// NETWORK 20
//   fb_gearinPos_el: add 2011 06 09 to delete 1sec delay
//   v_elevation: Virtual axis "v_elevation" with axis number 8
//   drive3: Real axis "Drive3" with axis number 3
// label: (*add ton between gearin and AF 2011_03_24*)
fb_gearinPos_el(
    Execute := test2 AND b_M_el_done,
    RatioNumerator := 1,
    RatioDenominator := 1,
    MasterFineadjust := 0,
    SyncMode := 0,
    StartMode := 0,
    Master := v_elevation,
    Slave := drive3); // MB_GearInPos
b_gearin_3_done := fb_gearinPos_el.InSync;

// NETWORK 21 (disabled)
//   v_elevation: Virtual axis "v_elevation" with axis number 8
//   drive4: Real axis "Drive4" with axis number 4
//   b_gearin_4_done: drive 3 and 4 are synchronous with v_elevation
// fb_gearin_4(
//     Execute := b_gearin_3_done,
//     RatioNumerator := 1,
//     RatioDenominator := 1,
//     MasterFineadjust := 0,
//     SyncMode := 0,
//     StartMode := 1,
//     Master := v_elevation,
//     Slave := drive4); // MB_GearInPos
// b_gearin_4_done := fb_gearin_4.InSync;

// NETWORK 22
//   b_local_on: in the local mode
//   axisdata[6].Axis_InAb: A-0-0021.14 -RD- Axis is ready for power to the engine (Ab)
//   axisdata[5].Axis_InAb: A-0-0021.14 -RD- Axis is ready for power to the engine (Ab)
//   b_enable_FI_6: the enable of drive 6
//   b_enable_FI_5: the enable of drive 5
// label: (*enable FeedIndexer axis with panel*)
fb_rtrig_FI(CLK := (b_local_on AND b_enable_FI OR b_remote_on AND b_activate_FI) AND axisdata[6].Axis_InAb AND axisdata[5].Axis_InAb); // R_TRIG
b_enable_FI_6 S= fb_rtrig_FI.Q;
b_enable_FI_5 S= fb_rtrig_FI.Q;

// NETWORK 23 (disabled)
//   b_enable_FI_5: the enable of drive 5
//   axisdata[5].Axis_InAb: A-0-0021.14 -RD- Axis is ready for power to the engine (Ab)
//   axisdata[5].Axis_Error: A-0-0021.09 -RD- Axis reports error
//   drive5: Real axis "Drive5" with axis number 5
// ton_en_5(IN := b_enable_FI_5 AND axisdata[5].Axis_InAb AND NOT axisdata[5].Axis_Error, PT := t#500ms); // TON
// fb_5_power(Enable := ton_en_5.Q, Axis := drive5); // MC_Power
// b_5_enable_on := fb_5_power.Status;

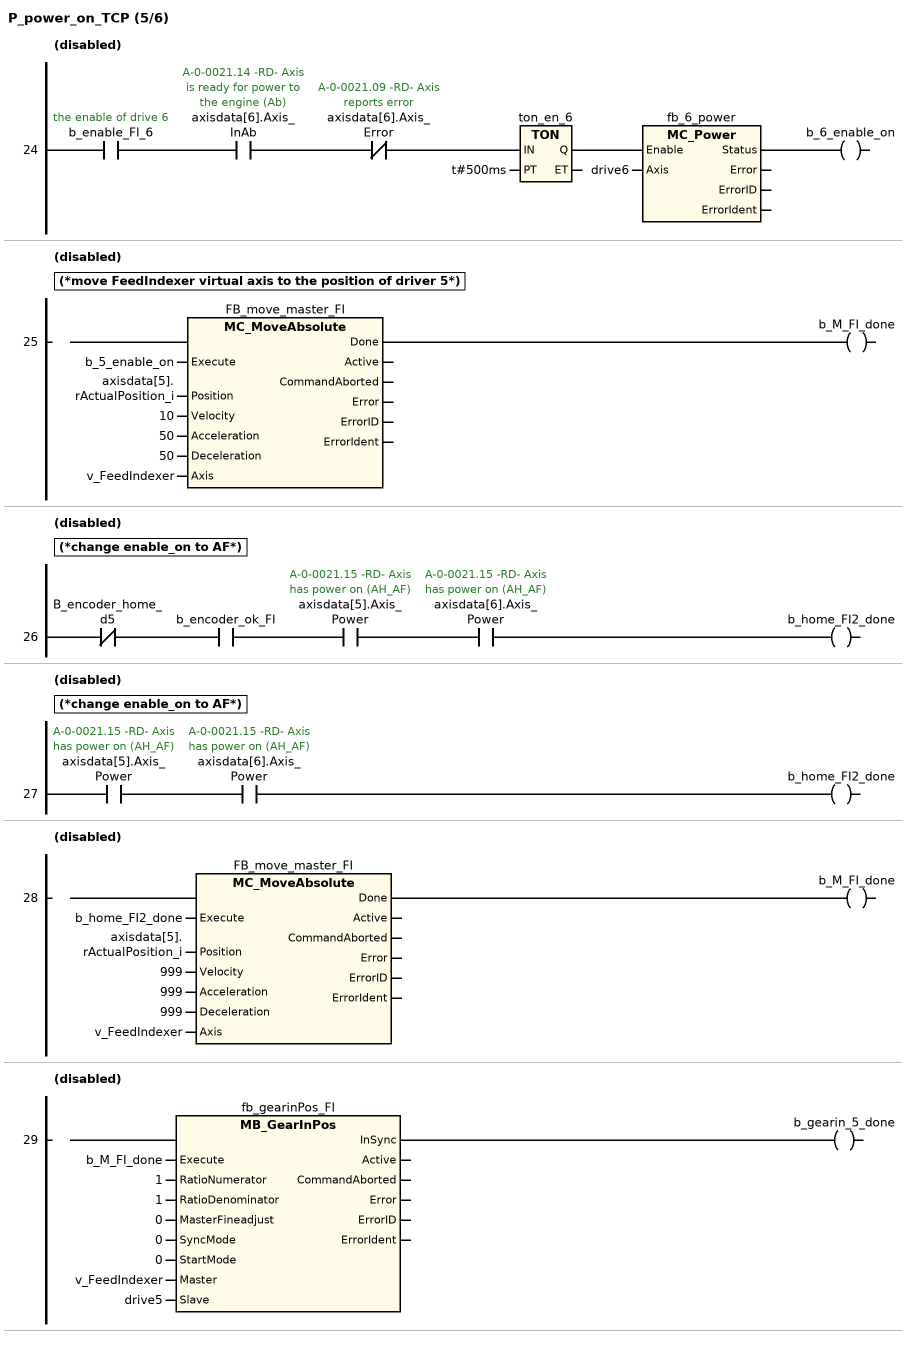
// NETWORK 24 (disabled)
//   b_enable_FI_6: the enable of drive 6
//   axisdata[6].Axis_InAb: A-0-0021.14 -RD- Axis is ready for power to the engine (Ab)
//   axisdata[6].Axis_Error: A-0-0021.09 -RD- Axis reports error
//   drive6: Real axis "Drive6" with axis number 6
// ton_en_6(IN := b_enable_FI_6 AND axisdata[6].Axis_InAb AND NOT axisdata[6].Axis_Error, PT := t#500ms); // TON
// fb_6_power(Enable := ton_en_6.Q, Axis := drive6); // MC_Power
// b_6_enable_on := fb_6_power.Status;

// NETWORK 25 (disabled)
//   axisdata[5].rActualPosition_i: A-0-0100 -RD- Actual position
//   v_FeedIndexer: Virtual axis "v_polarization" with axis number 9
// label: (*move FeedIndexer virtual axis to the position of driver 5*)
// FB_move_master_FI(
//     Execute := b_5_enable_on,
//     Position := axisdata[5].rActualPosition_i,
//     Velocity := 10,
//     Acceleration := 50,
//     Deceleration := 50,
//     Axis := v_FeedIndexer); // MC_MoveAbsolute
// b_M_FI_done := FB_move_master_FI.Done;

// NETWORK 26 (disabled)
//   axisdata[5].Axis_Power: A-0-0021.15 -RD- Axis has power on (AH_AF)
//   axisdata[6].Axis_Power: A-0-0021.15 -RD- Axis has power on (AH_AF)
// label: (*change enable_on to AF*)
// b_home_FI2_done := NOT B_encoder_home_d5 AND b_encoder_ok_FI AND axisdata[5].Axis_Power AND axisdata[6].Axis_Power;

// NETWORK 27 (disabled)
//   axisdata[5].Axis_Power: A-0-0021.15 -RD- Axis has power on (AH_AF)
//   axisdata[6].Axis_Power: A-0-0021.15 -RD- Axis has power on (AH_AF)
// label: (*change enable_on to AF*)
// b_home_FI2_done := axisdata[5].Axis_Power AND axisdata[6].Axis_Power;

// NETWORK 28 (disabled)
//   axisdata[5].rActualPosition_i: A-0-0100 -RD- Actual position
//   v_FeedIndexer: Virtual axis "v_polarization" with axis number 9
// FB_move_master_FI(
//     Execute := b_home_FI2_done,
//     Position := axisdata[5].rActualPosition_i,
//     Velocity := 999,
//     Acceleration := 999,
//     Deceleration := 999,
//     Axis := v_FeedIndexer); // MC_MoveAbsolute
// b_M_FI_done := FB_move_master_FI.Done;

// NETWORK 29 (disabled)
//   v_FeedIndexer: Virtual axis "v_polarization" with axis number 9
//   drive5: Real axis "Drive5" with axis number 5
// fb_gearinPos_FI(
//     Execute := b_M_FI_done,
//     RatioNumerator := 1,
//     RatioDenominator := 1,
//     MasterFineadjust := 0,
//     SyncMode := 0,
//     StartMode := 0,
//     Master := v_FeedIndexer,
//     Slave := drive5); // MB_GearInPos
// b_gearin_5_done := fb_gearinPos_FI.InSync;

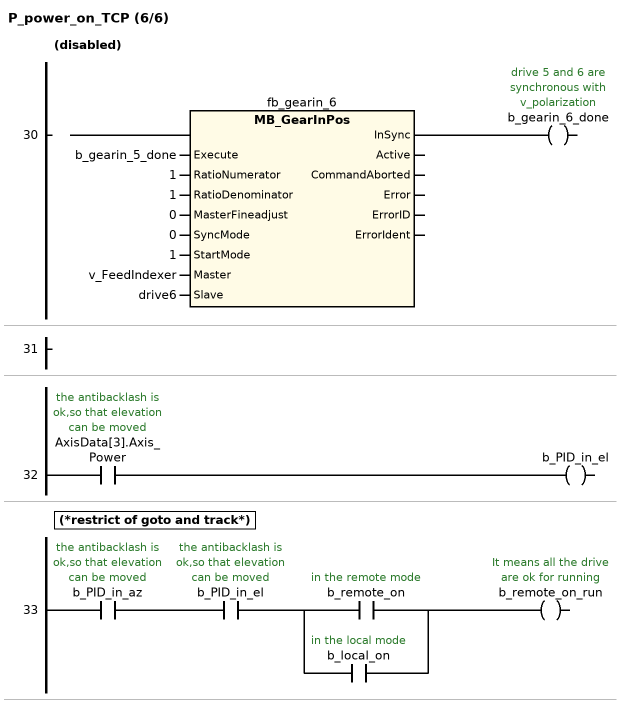
// NETWORK 30 (disabled)
//   v_FeedIndexer: Virtual axis "v_polarization" with axis number 9
//   drive6: Real axis "Drive6" with axis number 6
//   b_gearin_6_done: drive 5 and 6 are synchronous with v_polarization
// fb_gearin_6(
//     Execute := b_gearin_5_done,
//     RatioNumerator := 1,
//     RatioDenominator := 1,
//     MasterFineadjust := 0,
//     SyncMode := 0,
//     StartMode := 1,
//     Master := v_FeedIndexer,
//     Slave := drive6); // MB_GearInPos
// b_gearin_6_done := fb_gearin_6.InSync;

// NETWORK 31

// NETWORK 32
//   AxisData[3].Axis_Power: the antibacklash is ok,so that elevation can be moved
b_PID_in_el := AxisData[3].Axis_Power;

// NETWORK 33
//   b_PID_in_az: the antibacklash is ok,so that elevation can be moved
//   b_PID_in_el: the antibacklash is ok,so that elevation can be moved
//   b_remote_on: in the remote mode
//   b_local_on: in the local mode
//   b_remote_on_run: It means all the drive are ok for running
// label: (*restrict of goto and track*)
b_remote_on_run := b_PID_in_az AND b_PID_in_el AND (b_remote_on OR b_local_on);

END_PROGRAM

// IndraMotionMlc1/Application/POUs/Simulation/P_Simulation
PROGRAM P_Simulation
VAR
	//b_zone_az_sim:BOOL;  // simulate the zone switch 
	
	sim_HMV_warning : BOOL;(*the warning of HMV*)     
	sim_HMV_UD : BOOL;(*the UD of HMV*)              
	sim_stow_pin_limit_lock: BOOL:=1;(*locked*) // Stow pin deployed limit active
	sim_stow_pin_limit_unlock : BOOL;(*unlocked*) // Stow pin retracted limit active
	fb_rtrig_sim_stow_pin_retract: R_TRIG;
	fb_rtrig_sim_stow_pin_deploy: R_TRIG;
	sim_DriveCabinetDoor_Estop :BOOL;(*the estop of DriveCabinetDoor*)
	
	sim_PedDoor_Switch  :BOOL;(*the estop of DSDoor*)
	sim_PSCDoor_Switch :BOOL;(*the estop of DPSCDoor*)
	sim_EMISCDoor_Switch  :BOOL; (*the estop of EMISCDoor*)
	
	sim_AZ_Hatch  :BOOL;(*the estop of AZ_Hatch*)
	sim_Turnhead_Hatch  :BOOL;(*the estop of Turnhead_Hatch*)
	sim_DS_Estop  :BOOL;(*the estop of DS*)
	sim_Turnhead_Estop  :BOOL;(*the estop of Turnhead*)
	sim_FI_Estop  :BOOL;(*the estop of FI*)

	sim_HHP_Connected : BOOL;      
	sim_HHP_AZ : BOOL;
	sim_HHP_EL : BOOL;
	sim_HHP_Interlock : BOOL;
	sim_HHP_move_cw_slow : BOOL;
	sim_HHP_move_ccw_slow : BOOL;
	sim_HHP_move_cw_fast : BOOL;
	sim_HHP_move_ccw_fast : BOOL;
	
	sim_HHP_ENABLE  :BOOL;
	sim_HHP_STOW  :BOOL;
	sim_HHP_Motor_UNLOCK  :BOOL;
	sim_HHP_Disable  :BOOL;
	sim_HHP_Estop :BOOL;(*the estop of HHP*)
	sim_MAIN_PD_Compressor_breaker_on  :BOOL;
	sim_MAIN_PD_MAIN_lighting_on  :BOOL;
	
	sim_MAIN_PD_FI_Breaker_on :BOOL;
	sim_MAIN_PD_spare :BOOL;
	sim_PSC_PD_Light_Breaker_on :BOOL;
	sim_PSC_PD_EMISC_Breaker_on :BOOL;
	sim_PSC_PD_FAN_Breaker_on  :BOOL;
	sim_PSC_PD_spare :BOOL;
	
	sim_FI_PD_FI1_Breaker_on :BOOL;
	sim_FI_PD_FI2_Breaker_on  :BOOL;
	
	sim_Lock_Out_Az: BOOL;
	sim_Lock_Out_El: BOOL;
	sim_Lock_Out_Fi: BOOL;
	b_aztest: REAL;
	b_sector_sw: BOOL;
	
	
	
	b_escape: Bool;
	Az_lim_off: BOOL:=FALSE;
	El_lim_off: BOOL:=FALSE;
	Fi_lim_off: BOOL:=FALSE;
END_VAR

(* This piece of code is used to simulate the digital IO and drive IO when virtual axes are used *)
(*	r_limit_cw_az_sim:REAL:= 270 ;
	r_limit_ccw_az_sim:REAL:= -270;
	r_limit_final_cw_az_sim:REAL:= 271 ;
	r_limit_final_ccw_az_sim:REAL:=-271 ;
	// Elevation Limits
	r_limit_cw_az_sim:REAL:= 90;
	r_limit_ccw_az_sim:REAL:= 13.5 ;
	r_limit_final_cw_az_sim:REAL:=90.5 ;
	r_limit_final_ccw_az_sim:REAL:=13 ;
	// Feed Indexer Limits
	r_limit_cw_az_sim:REAL:= 110;
	r_limit_ccw_az_sim:REAL:= -140;
	r_limit_final_cw_az_sim:REAL:= 111 ;
	r_limit_final_ccw_az_sim:REAL:= -141; *)
	
IF gc_b_sim_on=1 THEN 
// Initial position 
    	

// Zone switch 
     b_aztest:=axisdata[1].rActualPosition_i;
	// There is a flash of llimits as AZ crosses over 0. I don't think this will be fixed in the simulator. 
	IF (axisdata[1].rActualPosition_i > 0.0 AND axisdata[1].rActualPosition_i < 90) THEN 
		b_zone_az_sim:=1;
	ELSIF axisdata[1].rActualPosition_i > 270 THEN
        b_zone_az_sim:=0;
	ELSE 
		b_zone_az_sim:=1;
	END_IF

// Azimuth limits
 IF NOT Az_lim_off THEN 
	IF r_pos_az_v >= gc_r_limit_cw_az_sim THEN 
		b_limit_cw_az:=1;
		b_stop_Az:=1;
	ELSE
		b_limit_cw_az:=0;
	END_IF
	
	IF r_pos_az_v <= gc_r_limit_ccw_az_sim THEN 
		b_limit_ccw_az:=1;
		b_stop_Az:=1;
		ELSE
		b_limit_ccw_az:=0;
	END_IF
	IF r_pos_az_v >= gc_r_limit_final_cw_az_sim THEN 
		b_limit_final_cw_az:=1;
		b_stop_Az:=1;
		ELSE
		b_limit_final_cw_az:=0;
	END_IF
	IF r_pos_az_v <= gc_r_limit_final_ccw_az_sim THEN 
		b_limit_final_ccw_az:=1;
		b_stop_Az:=1;
		ELSE
		b_limit_final_ccw_az:=0;
	END_IF
 ELSE
   b_limit_final_ccw_az:=0;
   b_limit_final_cw_az:=0;
	b_limit_ccw_az:=0;
	b_limit_cw_az:=0;
 END_IF;
	
	
	// Elevation limits
 IF NOT El_lim_off THEN
	IF r_pos_el_v >= gc_r_limit_cw_el_sim THEN 
		b_limit_cw_el:=1;
		
		IF b_enable_el_3=TRUE AND NOT(b_escape) THEN
			b_stop_El:=1;
			b_deactivate_el:=1;
			b_escape:=1;
		END_IF
	ELSE
		b_limit_cw_el:=0;
		b_escape:=0;
	END_IF
	IF r_pos_el_v <= gc_r_limit_ccw_el_sim THEN 
		b_limit_ccw_el:=1;
		
		//IF b_enable_el_3 THEN
		//	b_stop_El:=1;
		//	b_deactivate_el:=1;
		//END_IF
	ELSE
		b_limit_ccw_el:=0;
	END_IF
	IF r_pos_el_v >= gc_r_limit_final_cw_el_sim THEN 
		b_limit_final_cw_el:=1;
		//b_stop_El:=1;
		ELSE
		b_limit_final_cw_el:=0;
	END_IF
	IF r_pos_el_v <= gc_r_limit_final_ccw_el_sim THEN 
		b_limit_final_ccw_el:=1;
		//b_stop_El:=1;
		ELSE
		b_limit_final_ccw_el:=0;
	END_IF
 ELSE
	b_limit_final_ccw_el:=0;
	b_limit_final_cw_el:=0;
	b_limit_cw_el:=0;
	b_limit_ccw_el:=0;
 END_IF
 
	// Feed Indexer Limits
 IF NOT Fi_lim_off THEN
	IF r_pos_fi_v >= gc_r_limit_cw_fi_sim THEN 
		b_limit_cw_fi:=1;
		b_stop_Fi:=1;
	ELSE
		b_limit_cw_fi:=0;
	END_IF
	IF r_pos_fi_v <= gc_r_limit_ccw_fi_sim THEN 
		b_limit_ccw_fi:=1;
		b_stop_Fi:=1;
		ELSE
		b_limit_ccw_fi:=0;
	END_IF
	IF r_pos_fi_v >= gc_r_limit_final_cw_fi_sim THEN 
		b_limit_final_cw_fi:=1;
		b_stop_Fi:=1;
		ELSE
		b_limit_final_cw_fi:=0;
	END_IF
	IF r_pos_el_v <= gc_r_limit_final_ccw_fi_sim THEN 
		b_limit_final_ccw_fi:=1;
		b_stop_Fi:=1;
		ELSE
		b_limit_final_ccw_fi:=0;
	END_IF
ELSE 
	b_limit_final_ccw_fi:=0;
	b_limit_final_cw_fi:=0;
	b_limit_ccw_fi:=0;
	b_limit_cw_fi:=0;
END_IF
// Expose inputs to OPCUA

	b_HMV_warning:= sim_HMV_warning; 
	b_HMV_UD:=sim_HMV_UD ;         
	//b_stow_pin_limit_lock:= sim_stow_pin_limit_lock  ;
	fb_rtrig_sim_stow_pin_deploy(CLK:=sim_stow_pin_limit_lock);
	//b_stow_pin_limit_lock:=fb_rtrig_sim_stow_pin_deploy.Q;
	// simulate a retracted stow pin limit
	//fb_rtrig_sim_stow_pin_retract(CLK:=sim_stow_pin_limit_unlock);
	//b_stow_pin_limit_unlock:=fb_rtrig_sim_stow_pin_retract.Q;
	
	
	b_DriveCabinetDoor_Estop:= sim_DriveCabinetDoor_Estop ; 
	b_DSDoor_Estop:= sim_PedDoor_Switch ; 
	b_PSCDoor_Estop:= sim_PSCDoor_Switch ; 
	b_AZ_Hatch:= sim_AZ_Hatch ;  
	b_Turnhead_Hatch:= sim_Turnhead_Hatch ; 
	b_DS_Estop:= sim_DS_Estop;  
	b_Turnhead_Estop:= sim_Turnhead_Estop;  
	b_FI_Estop:=  sim_FI_Estop;

	b_HHP_Connected:=  sim_HHP_Connected; 
	b_HHP_AZ:= sim_HHP_AZ;
	b_HHP_EL:= sim_HHP_EL;
	b_HHP_Interlock:= sim_HHP_Interlock; 
	b_HHP_move_cw_slow:=  sim_HHP_move_cw_slow; 
	b_HHP_move_ccw_slow:= sim_HHP_move_ccw_slow ;
	b_HHP_move_cw_fast:= sim_HHP_move_cw_fast;
	b_HHP_move_ccw_fast:= sim_HHP_move_ccw_fast;
	
	b_HHP_ENABLE:= sim_HHP_ENABLE ;
	b_HHP_STOW:= sim_HHP_STOW ;
	b_HHP_Motor_UNLOCK:=  sim_HHP_Motor_UNLOCK; 
	b_HHP_Disable:=  sim_HHP_Disable;
	b_EMISCDoor_Estop:= sim_EMISCDoor_Switch;  
	b_HHP_Estop:= sim_HHP_Estop;
	b_MAIN_PD_Compressor_breaker_on:= sim_MAIN_PD_Compressor_breaker_on;
	b_MAIN_PD_MAIN_lighting_on:= sim_MAIN_PD_MAIN_lighting_on;  
	
	b_MAIN_PD_FI_Breaker_on:= sim_MAIN_PD_FI_Breaker_on;
	b_MAIN_PD_spare:=  sim_MAIN_PD_spare;
	b_PSC_PD_Light_Breaker_on:= sim_PSC_PD_Light_Breaker_on;
	b_PSC_PD_EMISC_Breaker_on:=  sim_PSC_PD_EMISC_Breaker_on;
	b_PSC_PD_FAN_Breaker_on:= sim_PSC_PD_FAN_Breaker_on ;
    b_PSC_PD_spare:= sim_PSC_PD_spare;
	b_FI_PD_FI1_Breaker_on:= sim_FI_PD_FI1_Breaker_on;
	b_FI_PD_FI2_Breaker_on := sim_FI_PD_FI2_Breaker_on ;
	
	b_Lock_Out_Az:= sim_Lock_Out_Az;
	b_Lock_Out_El:= sim_Lock_Out_El;
	b_Lock_Out_Fi:= sim_Lock_Out_Fi;
	

	
 END_IF //IF b_sim_on=1 THEN

END_PROGRAM

// IndraMotionMlc1/Application/POUs/Panel Function/P_remote_local
(*This program is built for switch the mode between local,remote and off.
In the local mode,the antenna can be controled only by the button on the
panelbox;In the remote mode,the antenna can be controled only by the command
that come from the ACU;In the off mode,all the motion will be stopped.
And every time the switch is off,there is a clear_error action*)
PROGRAM P_remote_local
VAR
(*clear all error when the switch is off*)
	FB_clear_all_error: MB_WriteParameter;
	b_clear_error: BOOL;
	b_clear_all_error: BOOL;
	b_clear_done: BOOL;
	rtrig_clear_error: R_TRIG;
	rtrig_reset_clear: R_TRIG;
	el_encoder_pos: LREAL;
	b_run_once: BOOL;
END_VAR

b_Alarm;
b_Horn;
b_HHP_Interlock;
b_HHP_ENABLE;
b_HHP_STOW;
b_HHP_Motor_UNLOCK;
b_HHP_Disable;
el_encoder_pos:=Motor_to_encoder(axisdata[3].rActualPosition_i);

IF b_HHP_AZ=FALSE AND b_HHP_FI=FALSE THEN
	b_HHP_EL := TRUE;
ELSE
	b_HHP_EL := FALSE;
END_IF

IF b_HHP_connected THEN
	b_remote_on:=FALSE;
	b_local_on:=TRUE;
	CommandArbiter.Status.DscCmdAuthority:= HHP; // Needsome code to change it to No Auth when HHP is dosconnected. 
	IF NOT b_run_once THEN 
     b_Horn_Start:= TRUE; 
	 b_run_once:=TRUE;
	END_IF
ELSE
	b_remote_on:=TRUE;
	b_local_on:=FALSE;
	b_run_once:=FALSE;
END_IF

IF b_local_on OR b_remote_on THEN
	b_clear_error:=FALSE;
END_IF;
(*when the switch is off,reset some command and stop all the motion*)
IF b_remote_on =FALSE AND b_local_on=FALSE THEN
	b_power_Az:=FALSE;
	b_power_el:=FALSE;
	b_power_FI:=FALSE;
	b_stow_pin_deploy:=FALSE;
	b_stow_pin_retract:=FALSE;
	b_scc_enable_on:=FALSE;
	b_scc_enable_off:=FALSE;
	b_scc_stow:=FALSE;
	b_track_on:=FALSE;
	b_clear_error:=TRUE;
	b_scc_goto:=FALSE;
	b_scc_goto_az:=FALSE;
	b_scc_goto_el:=FALSE;
	b_scc_goto_FI:=FALSE;
	b_scc_vel:=FALSE;
END_IF;
(*transfer the sub-program A_clear_error to clear all the error*)
P_remote_local.A_clear_error();

ACTION A_clear_error:
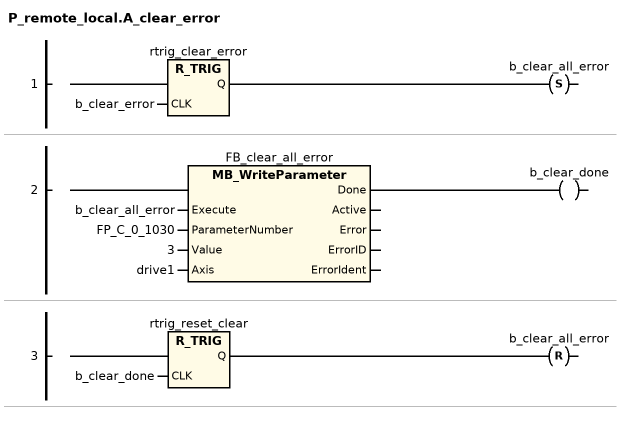
// NETWORK 1
rtrig_clear_error(CLK := b_clear_error); // R_TRIG
b_clear_all_error S= rtrig_clear_error.Q;

// NETWORK 2
FB_clear_all_error(Execute := b_clear_all_error, ParameterNumber := FP_C_0_1030, Value := 3, Axis := drive1); // MB_WriteParameter
b_clear_done := FB_clear_all_error.Done;

// NETWORK 3
rtrig_reset_clear(CLK := b_clear_done); // R_TRIG
b_clear_all_error R= rtrig_reset_clear.Q;
END_ACTION

END_PROGRAM

// IndraMotionMlc1/Application/POUs/TCP/Message/Motor_to_encoder
FUNCTION Motor_to_encoder : LREAL
VAR_INPUT
	motor_input:LREAL;
END_VAR
VAR
END_VAR

IF motor_input < 619748 THEN
	Motor_to_encoder:=AA1*(motor_input)-BB1;	
ELSIF (619748 <= motor_input) AND (motor_input < 676291) THEN
	Motor_to_encoder:=AA2*(motor_input)-BB2;
ELSIF (676291 <= motor_input) AND (motor_input < 735364) THEN
	Motor_to_encoder:=AA3*(motor_input)-BB3;
ELSIF (735364 <= motor_input) AND (motor_input < 796846) THEN
	Motor_to_encoder:=AA4*(motor_input)-BB4;
ELSIF (796846 <= motor_input) AND (motor_input < 860616) THEN
	Motor_to_encoder:=AA5*(motor_input)-BB5;
ELSIF (860616 <= motor_input) AND (motor_input < 926557) THEN
	Motor_to_encoder:=AA6*(motor_input)-BB6;
ELSIF (926557 <= motor_input) AND (motor_input < 994541) THEN
	Motor_to_encoder:=AA7*(motor_input)-BB7;
ELSIF (994541 <= motor_input) AND (motor_input < 1064438) THEN
	Motor_to_encoder:=AA8*(motor_input)-BB8;
ELSIF (1064438 <= motor_input) AND (motor_input < 1136109) THEN
	Motor_to_encoder:=AA9*(motor_input)-BB9;
ELSIF (1136109 <= motor_input) AND (motor_input < 1209420) THEN
	Motor_to_encoder:=AA10*(motor_input)-BB10;
ELSIF (1209420 <= motor_input) AND (motor_input < 1284232) THEN
	Motor_to_encoder:=AA11*(motor_input)-BB11;
ELSIF (1284232 <= motor_input) AND (motor_input < 1360400) THEN
	Motor_to_encoder:=AA12*(motor_input)-BB12;
ELSIF (1360400 <= motor_input) AND (motor_input < 1437759) THEN
	Motor_to_encoder:=AA13*(motor_input)-BB13;
ELSIF (1437759 <= motor_input) AND (motor_input < 1516147) THEN
	Motor_to_encoder:=AA14*(motor_input)-BB14;
ELSE
	Motor_to_encoder:=AA15*(motor_input)-BB15;
END_IF

END_FUNCTION

// IndraMotionMlc1/Application/POUs/Panel Function/P_read_drv_IO
(* The program is built for read the digital input value on X31 and X32,
and FP_P_0_0303 is Digital I/Os status display *)
PROGRAM P_read_drv_IO
VAR
(*With "MB_ReadParameter",it is possible to read the current value of a parameter. The return value is DINT. *)
	FB_1_read_P303: MB_ReadParameter;
	FB_2_read_P303: MB_ReadParameter;
	FB_3_read_P303: MB_ReadParameter;
	FB_4_read_P303: MB_ReadParameter;
	FB_5_read_P303: MB_ReadParameter;
	FB_6_read_P303: MB_ReadParameter;
	Dint_1_P303: DINT;
	Dint_2_P303: DINT;
	Dint_3_P303: DINT;
	Dint_4_P303: DINT;
	Dint_5_P303: DINT;
	Dint_6_P303: DINT;
(*change DINT to DWORD,so that the bit of DWORD can be read*)
	Dword_1_P303: DWORD;
	Dword_2_P303: DWORD;
	Dword_3_P303: DWORD;
	Dword_4_P303: DWORD;
	Dword_5_P303: DWORD;
	Dword_6_P303: DWORD;
	R_TRIG_0: R_TRIG;
	rtrig_stop_az1: R_TRIG;
	b_stop1_done: BOOL;
	b_stop_act_az: BOOL;
	R_TRIG_1: r_trig;
	b_zero_velocity: BOOL;
	fb_zero_velocity: MC_movevelocity;
	b_zero1_done: BOOL;
	b_zero_act_az: BOOL;
	TON_0: ton;
	FB_move_master_az1: MC_MoveAbsolute;
	fb_stop_AZ: MC_STOP;
END_VAR
VAR // added by the converter: edge detectors and wires of the graphical bodies
    _w1, _w2, _w3, _w4, _w5, _w6 : ANY;
    _w7 : BOOL;
END_VAR

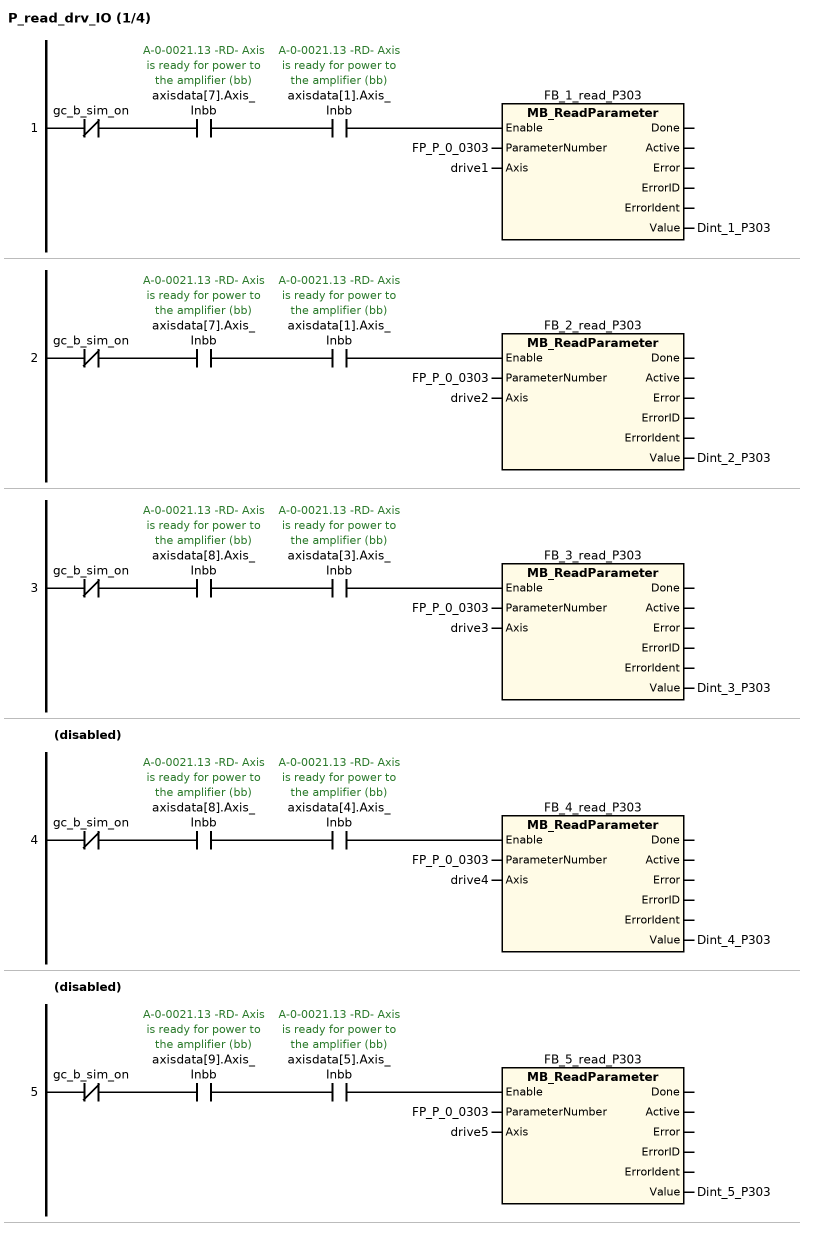
// NETWORK 1
//   FB_1_read_P303: With "MB_ReadParameter",it is possible to read the current value of a parameter. The return value is DINT.
//   axisdata[7].Axis_Inbb: A-0-0021.13 -RD- Axis is ready for power to the amplifier (bb)
//   axisdata[1].Axis_Inbb: A-0-0021.13 -RD- Axis is ready for power to the amplifier (bb)
//   FP_P_0_0303: Digital inputs, input image of device
//   drive1: Real axis "Drive1" with axis number 1
FB_1_read_P303(
    Enable := NOT gc_b_sim_on AND axisdata[7].Axis_Inbb AND axisdata[1].Axis_Inbb,
    ParameterNumber := FP_P_0_0303,
    Axis := drive1,
    Value => Dint_1_P303); // MB_ReadParameter

// NETWORK 2
//   axisdata[7].Axis_Inbb: A-0-0021.13 -RD- Axis is ready for power to the amplifier (bb)
//   axisdata[1].Axis_Inbb: A-0-0021.13 -RD- Axis is ready for power to the amplifier (bb)
//   FP_P_0_0303: Digital inputs, input image of device
//   drive2: Real axis "Drive2" with axis number 2
FB_2_read_P303(
    Enable := NOT gc_b_sim_on AND axisdata[7].Axis_Inbb AND axisdata[1].Axis_Inbb,
    ParameterNumber := FP_P_0_0303,
    Axis := drive2,
    Value => Dint_2_P303); // MB_ReadParameter

// NETWORK 3
//   axisdata[8].Axis_Inbb: A-0-0021.13 -RD- Axis is ready for power to the amplifier (bb)
//   axisdata[3].Axis_Inbb: A-0-0021.13 -RD- Axis is ready for power to the amplifier (bb)
//   FP_P_0_0303: Digital inputs, input image of device
//   drive3: Real axis "Drive3" with axis number 3
FB_3_read_P303(
    Enable := NOT gc_b_sim_on AND axisdata[8].Axis_Inbb AND axisdata[3].Axis_Inbb,
    ParameterNumber := FP_P_0_0303,
    Axis := drive3,
    Value => Dint_3_P303); // MB_ReadParameter

// NETWORK 4 (disabled)
//   axisdata[8].Axis_Inbb: A-0-0021.13 -RD- Axis is ready for power to the amplifier (bb)
//   axisdata[4].Axis_Inbb: A-0-0021.13 -RD- Axis is ready for power to the amplifier (bb)
//   FP_P_0_0303: Digital inputs, input image of device
//   drive4: Real axis "Drive4" with axis number 4
// FB_4_read_P303(
//     Enable := NOT gc_b_sim_on AND axisdata[8].Axis_Inbb AND axisdata[4].Axis_Inbb,
//     ParameterNumber := FP_P_0_0303,
//     Axis := drive4,
//     Value => Dint_4_P303); // MB_ReadParameter

// NETWORK 5 (disabled)
//   axisdata[9].Axis_Inbb: A-0-0021.13 -RD- Axis is ready for power to the amplifier (bb)
//   axisdata[5].Axis_Inbb: A-0-0021.13 -RD- Axis is ready for power to the amplifier (bb)
//   FP_P_0_0303: Digital inputs, input image of device
//   drive5: Real axis "Drive5" with axis number 5
// FB_5_read_P303(
//     Enable := NOT gc_b_sim_on AND axisdata[9].Axis_Inbb AND axisdata[5].Axis_Inbb,
//     ParameterNumber := FP_P_0_0303,
//     Axis := drive5,
//     Value => Dint_5_P303); // MB_ReadParameter

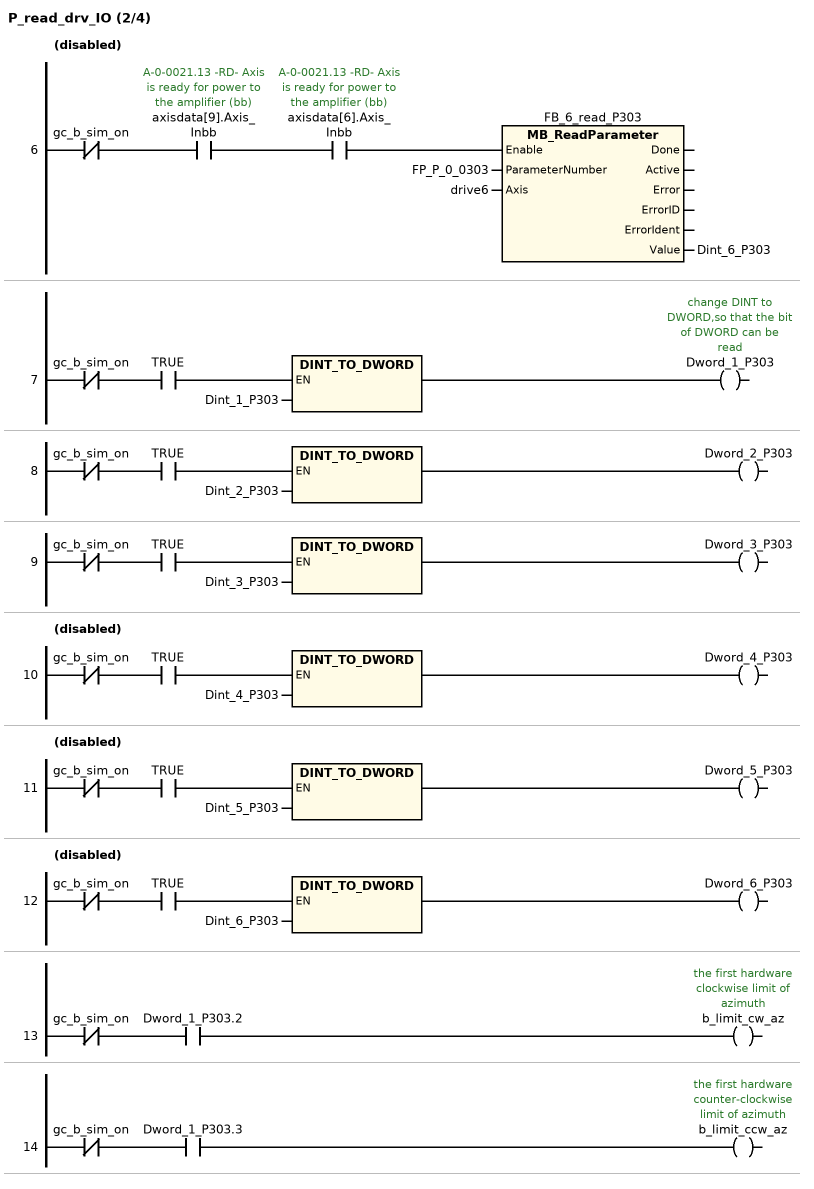
// NETWORK 6 (disabled)
//   axisdata[9].Axis_Inbb: A-0-0021.13 -RD- Axis is ready for power to the amplifier (bb)
//   axisdata[6].Axis_Inbb: A-0-0021.13 -RD- Axis is ready for power to the amplifier (bb)
//   FP_P_0_0303: Digital inputs, input image of device
//   drive6: Real axis "Drive6" with axis number 6
// FB_6_read_P303(
//     Enable := NOT gc_b_sim_on AND axisdata[9].Axis_Inbb AND axisdata[6].Axis_Inbb,
//     ParameterNumber := FP_P_0_0303,
//     Axis := drive6,
//     Value => Dint_6_P303); // MB_ReadParameter

// NETWORK 7
//   Dword_1_P303: change DINT to DWORD,so that the bit of DWORD can be read
IF NOT gc_b_sim_on AND TRUE THEN _w1 := DINT_TO_DWORD(Dint_1_P303); END_IF
Dword_1_P303 := _w1;

// NETWORK 8
IF NOT gc_b_sim_on AND TRUE THEN _w2 := DINT_TO_DWORD(Dint_2_P303); END_IF
Dword_2_P303 := _w2;

// NETWORK 9
IF NOT gc_b_sim_on AND TRUE THEN _w3 := DINT_TO_DWORD(Dint_3_P303); END_IF
Dword_3_P303 := _w3;

// NETWORK 10 (disabled)
// IF NOT gc_b_sim_on AND TRUE THEN _w4 := DINT_TO_DWORD(Dint_4_P303); END_IF
// Dword_4_P303 := _w4;

// NETWORK 11 (disabled)
// IF NOT gc_b_sim_on AND TRUE THEN _w5 := DINT_TO_DWORD(Dint_5_P303); END_IF
// Dword_5_P303 := _w5;

// NETWORK 12 (disabled)
// IF NOT gc_b_sim_on AND TRUE THEN _w6 := DINT_TO_DWORD(Dint_6_P303); END_IF
// Dword_6_P303 := _w6;

// NETWORK 13
//   b_limit_cw_az: the first hardware clockwise limit of azimuth
b_limit_cw_az := NOT gc_b_sim_on AND Dword_1_P303.2;

// NETWORK 14
//   b_limit_ccw_az: the first hardware counter-clockwise limit of azimuth
b_limit_ccw_az := NOT gc_b_sim_on AND Dword_1_P303.3;

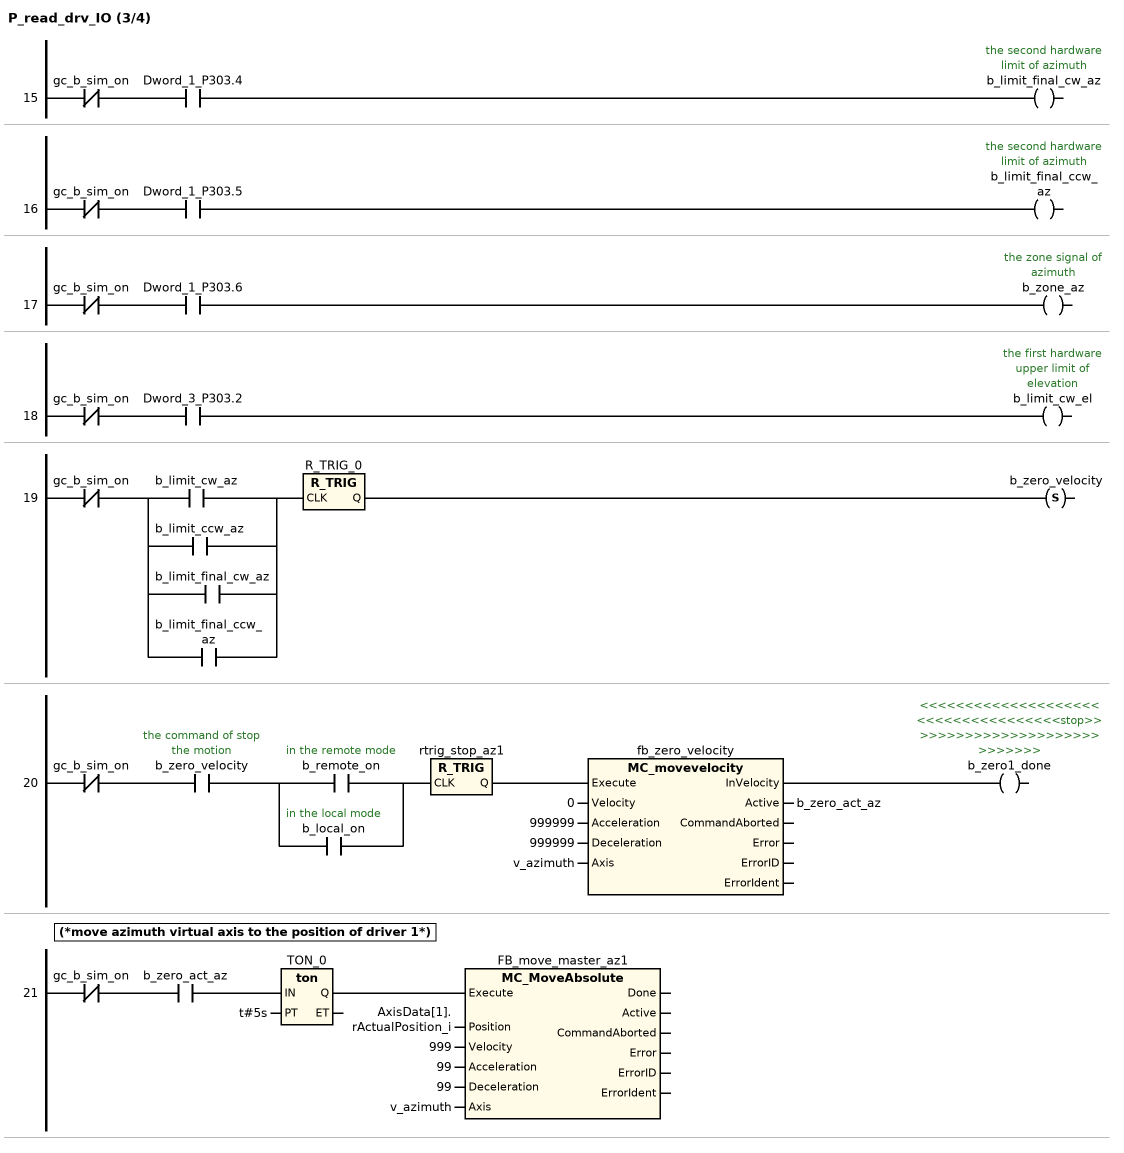
// NETWORK 15
//   b_limit_final_cw_az: the second hardware limit of azimuth
b_limit_final_cw_az := NOT gc_b_sim_on AND Dword_1_P303.4;

// NETWORK 16
//   b_limit_final_ccw_az: the second hardware limit of azimuth
b_limit_final_ccw_az := NOT gc_b_sim_on AND Dword_1_P303.5;

// NETWORK 17
//   b_zone_az: the zone signal of azimuth
b_zone_az := NOT gc_b_sim_on AND Dword_1_P303.6;

// NETWORK 18
//   b_limit_cw_el: the first hardware upper limit of elevation
b_limit_cw_el := NOT gc_b_sim_on AND Dword_3_P303.2;

// NETWORK 19
_w7 := NOT gc_b_sim_on;
R_TRIG_0(CLK := _w7 AND b_limit_cw_az OR _w7 AND b_limit_ccw_az OR _w7 AND b_limit_final_cw_az OR _w7 AND b_limit_final_ccw_az); // R_TRIG
b_zero_velocity S= R_TRIG_0.Q;

// NETWORK 20
//   b_zero_velocity: the command of stop the motion
//   b_remote_on: in the remote mode
//   b_local_on: in the local mode
//   999999: Virtual axis "v_azimuth" with axis number 7
//   b_zero1_done: <<<<<<<<<<<<<<<<<<<<<<<<<<<<<<<<<<<<stop>>>>>>>>>>>>>>>>>>>>>>>>>>>>>
rtrig_stop_az1(CLK := NOT gc_b_sim_on AND b_zero_velocity AND (b_remote_on OR b_local_on)); // R_TRIG
fb_zero_velocity(
    Execute := rtrig_stop_az1.Q,
    Velocity := 0,
    Acceleration := 999999,
    Deceleration := 999999,
    Axis := v_azimuth,
    Active => b_zero_act_az); // MC_movevelocity
b_zero1_done := fb_zero_velocity.InVelocity;

// NETWORK 21
//   FB_move_master_az1: "MC_MoveAbsolute" is used to move the drive to a preset absolute position.
//   AxisData[1].rActualPosition_i: A-0-0100 -RD- Actual position
//   v_azimuth: Virtual axis "v_azimuth" with axis number 7
// label: (*move azimuth virtual axis to the position of driver 1*)
TON_0(IN := NOT gc_b_sim_on AND b_zero_act_az, PT := t#5s); // ton
FB_move_master_az1(
    Execute := TON_0.Q,
    Position := AxisData[1].rActualPosition_i,
    Velocity := 999,
    Acceleration := 99,
    Deceleration := 99,
    Axis := v_azimuth); // MC_MoveAbsolute

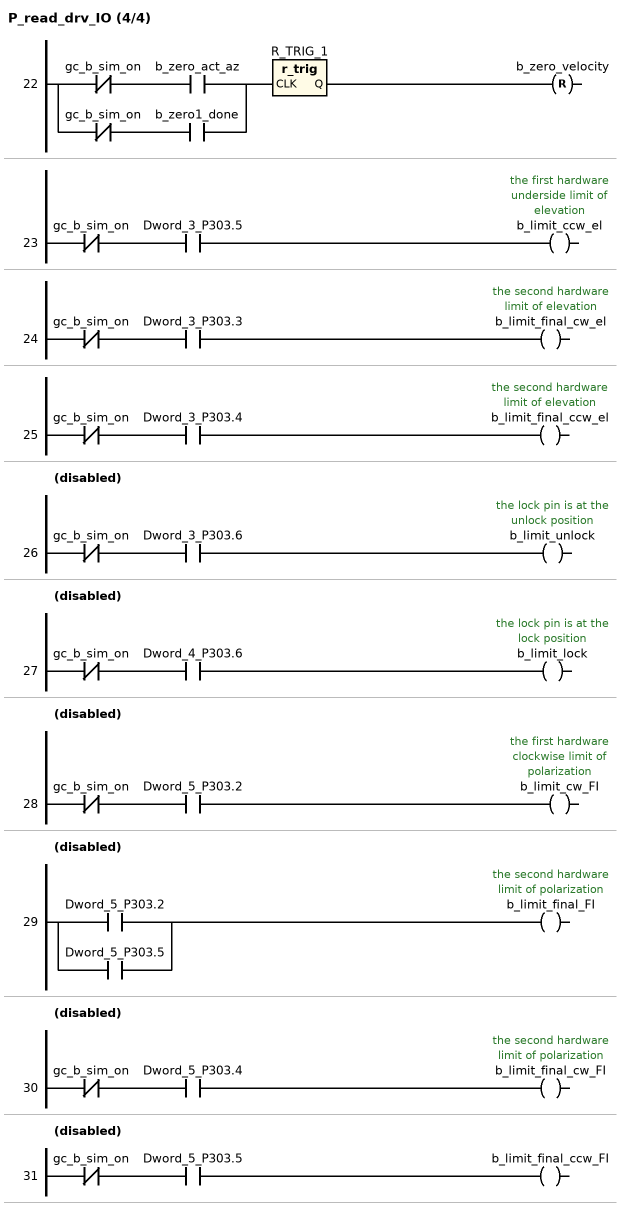
// NETWORK 22
R_TRIG_1(CLK := NOT gc_b_sim_on AND b_zero_act_az OR NOT gc_b_sim_on AND b_zero1_done); // r_trig
b_zero_velocity R= R_TRIG_1.Q;

// NETWORK 23
//   b_limit_ccw_el: the first hardware underside limit of elevation
b_limit_ccw_el := NOT gc_b_sim_on AND Dword_3_P303.5;

// NETWORK 24
//   b_limit_final_cw_el: the second hardware limit of elevation
b_limit_final_cw_el := NOT gc_b_sim_on AND Dword_3_P303.3;

// NETWORK 25
//   b_limit_final_ccw_el: the second hardware limit of elevation
b_limit_final_ccw_el := NOT gc_b_sim_on AND Dword_3_P303.4;

// NETWORK 26 (disabled)
//   b_limit_unlock: the lock pin is at the unlock position
// b_limit_unlock := NOT gc_b_sim_on AND Dword_3_P303.6;

// NETWORK 27 (disabled)
//   b_limit_lock: the lock pin is at the lock position
// b_limit_lock := NOT gc_b_sim_on AND Dword_4_P303.6;

// NETWORK 28 (disabled)
//   b_limit_cw_FI: the first hardware clockwise limit of polarization
// b_limit_cw_FI := NOT gc_b_sim_on AND Dword_5_P303.2;

// NETWORK 29 (disabled)
//   b_limit_final_FI: the second hardware limit of polarization
// b_limit_final_FI := Dword_5_P303.2 OR Dword_5_P303.5;

// NETWORK 30 (disabled)
//   b_limit_final_cw_FI: the second hardware limit of polarization
// b_limit_final_cw_FI := NOT gc_b_sim_on AND Dword_5_P303.4;

// NETWORK 31 (disabled)
// b_limit_final_ccw_FI := NOT gc_b_sim_on AND Dword_5_P303.5;

END_PROGRAM

// IndraMotionMlc1/Application/POUs/Motion/P_power_off_TCP
(*the program is built for power off the 3 axis under the contol of remote or local.
the elevation axis is the similar with the azimuth*)
PROGRAM P_power_off_TCP
VAR
(*The firmware function block "MC_Stop" is used to bring the drive to the status STOP.*)
	fb_stop_v_az: MC_Stop;
	fb_stop_d1: MC_Stop;
	fb_stop_d2: MC_Stop;
	fb_stop_v_el: MC_Stop;
	fb_stop_d3: MC_Stop;
	fb_stop_d4: MC_Stop;
	fb_stop_v_FI: MC_Stop;
	fb_stop_d5: MC_Stop;
	fb_stop_d6: MC_Stop;
(*The firmware function block "MC_GearOut" is used to terminate an active synchronization function block.*)
	fb_gearout_d1: MC_GearOut;
	fb_gearout_d2: MC_GearOut;
	fb_gearout_d3: MC_GearOut;
	fb_gearout_d4: MC_GearOut;
	fb_gearout_d5: MC_GearOut;
	fb_gearout_d6: MC_GearOut;
(*The function block R_TRIG detects a rising edge*)
	rtrig_stop_az: R_TRIG;
	rtrig_stop_el: R_TRIG;
	rtrig_stop_FI: R_TRIG;
	rtrig_stop_d1: R_TRIG;
	rtrig_stop_d2: R_TRIG;
	rtrig_stop_d3: R_TRIG;
	rtrig_stop_d4: R_TRIG;
	rtrig_stop_d5: R_TRIG;
	rtrig_stop_d6: R_TRIG;
	rtrig_d1: R_TRIG;
	rtrig_d2: R_TRIG;
	rtrig_d3: R_TRIG;
	rtrig_d4: R_TRIG;
	rtrig_d5: R_TRIG;
	rtrig_d6: R_TRIG;
	rtrig_en_off: R_TRIG;
(*The function block F_TRIG a falling edge*)
	ftrig_reset_az: F_TRIG;
	ftrig_reset_el: F_TRIG;
	ftrig_reset_FI: F_TRIG;
(*The function block Timer On Delay implements a turn-on delay..*)
	fb_ton_powoff_az: TON;
	fb_ton_powoff_el: TON;
	fb_ton_powoff_FI: TON;
	fb_ton_en_off: TON;
	fb_ton_error: TON;
	FB_clear_all_error: MB_WriteParameter;
	fb_f_enable_off: F_TRIG;
	fb_R_enable_off: R_TRIG;
	fb_ton_enable_off: TON;
	b_enable_start: BOOL;
	fb_blink_reset: BLINK;
	b_clear_error: BOOL;
	fb_r_clear_error: R_TRIG;
	FB_clear_error_1: MB_WriteParameter;
	rtrig_clr_deactivate: R_TRIG;
	rtrig_el_deactivate_clear: R_TRIG;
	rtrig_deactivate_clear_el: R_TRIG;
	rtrig_clr_deactivate_az: R_TRIG;
	rtrig_clr_deactivate_fi: R_TRIG;
	b_execute_goto_Az: INT;
	b_start_goto_Az: BOOL;
END_VAR

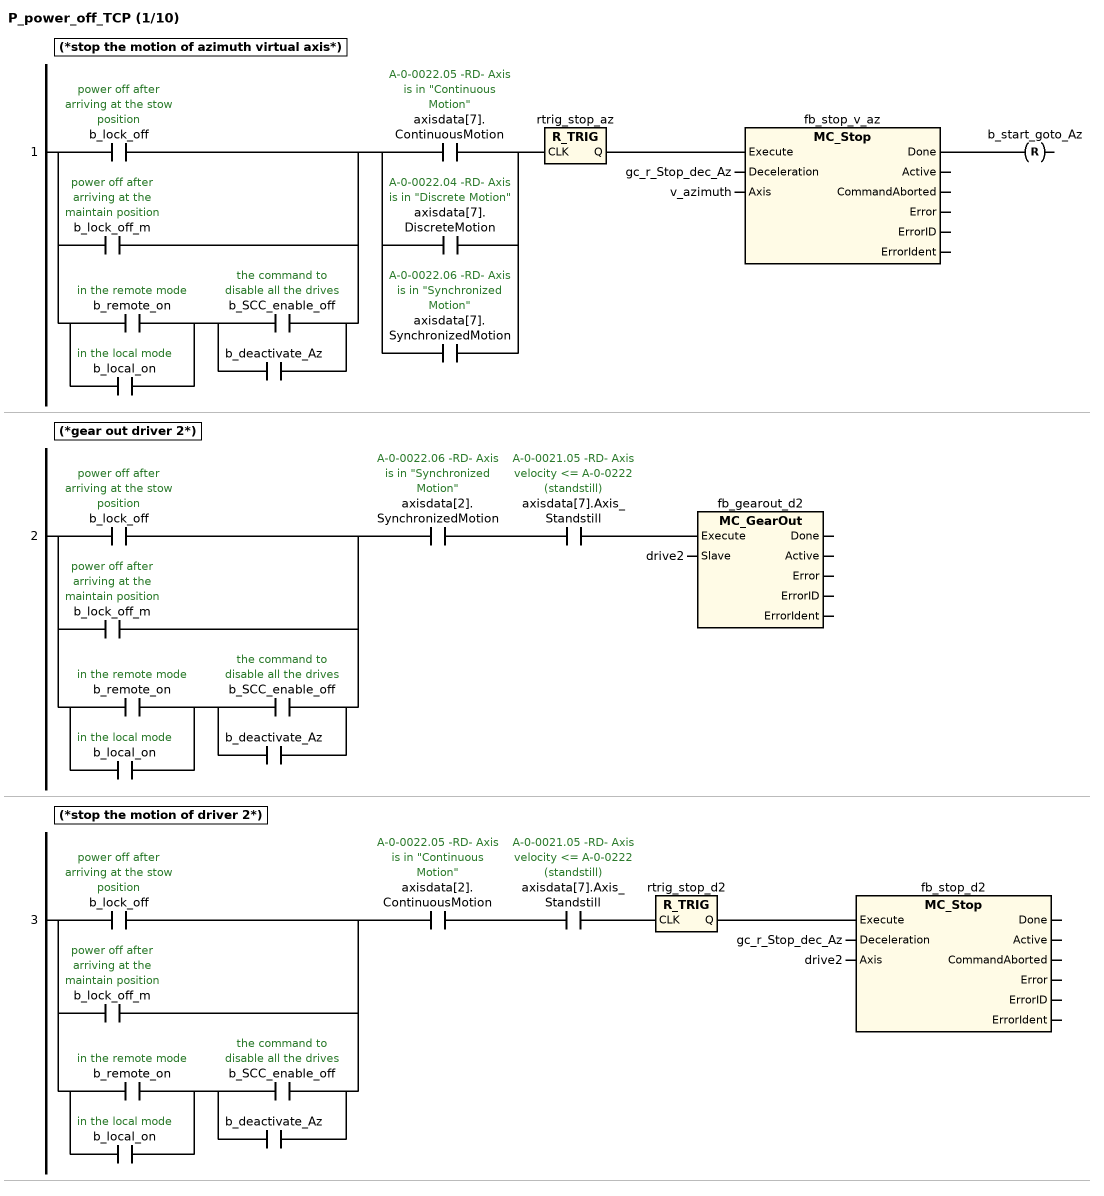
// NETWORK 1
//   fb_stop_v_az: The firmware function block "MC_Stop" is used to bring the drive to the status STOP.
//   rtrig_stop_az: The function block R_TRIG detects a rising edge
//   b_lock_off: power off after arriving at the stow position
//   b_lock_off_m: power off after arriving at the maintain position
//   b_remote_on: in the remote mode
//   b_local_on: in the local mode
//   b_SCC_enable_off: the command to disable all the drives
//   axisdata[7].ContinuousMotion: A-0-0022.05 -RD- Axis is in "Continuous Motion"
//   axisdata[7].DiscreteMotion: A-0-0022.04 -RD- Axis is in "Discrete Motion"
//   axisdata[7].SynchronizedMotion: A-0-0022.06 -RD- Axis is in "Synchronized Motion"
//   v_azimuth: Virtual axis "v_azimuth" with axis number 7
// label: (*stop the motion of azimuth virtual axis*)
rtrig_stop_az(CLK := (b_lock_off OR b_lock_off_m OR (b_remote_on OR b_local_on) AND (b_SCC_enable_off OR b_deactivate_Az)) AND (axisdata[7].ContinuousMotion OR axisdata[7].DiscreteMotion OR axisdata[7].SynchronizedMotion)); // R_TRIG
fb_stop_v_az(Execute := rtrig_stop_az.Q, Deceleration := gc_r_Stop_dec_Az, Axis := v_azimuth); // MC_Stop
b_start_goto_Az R= fb_stop_v_az.Done;

// NETWORK 2
//   b_lock_off: power off after arriving at the stow position
//   b_lock_off_m: power off after arriving at the maintain position
//   b_remote_on: in the remote mode
//   b_local_on: in the local mode
//   b_SCC_enable_off: the command to disable all the drives
//   axisdata[2].SynchronizedMotion: A-0-0022.06 -RD- Axis is in "Synchronized Motion"
//   axisdata[7].Axis_Standstill: A-0-0021.05 -RD- Axis velocity <= A-0-0222 (standstill)
//   drive2: Real axis "Drive2" with axis number 2
// label: (*gear out driver 2*)
fb_gearout_d2(Execute := (b_lock_off OR b_lock_off_m OR (b_remote_on OR b_local_on) AND (b_SCC_enable_off OR b_deactivate_Az)) AND axisdata[2].SynchronizedMotion AND axisdata[7].Axis_Standstill, Slave := drive2); // MC_GearOut

// NETWORK 3
//   b_lock_off: power off after arriving at the stow position
//   b_lock_off_m: power off after arriving at the maintain position
//   b_remote_on: in the remote mode
//   b_local_on: in the local mode
//   b_SCC_enable_off: the command to disable all the drives
//   axisdata[2].ContinuousMotion: A-0-0022.05 -RD- Axis is in "Continuous Motion"
//   axisdata[7].Axis_Standstill: A-0-0021.05 -RD- Axis velocity <= A-0-0222 (standstill)
//   drive2: Real axis "Drive2" with axis number 2
// label: (*stop the motion of driver 2*)
rtrig_stop_d2(CLK := (b_lock_off OR b_lock_off_m OR (b_remote_on OR b_local_on) AND (b_SCC_enable_off OR b_deactivate_Az)) AND axisdata[2].ContinuousMotion AND axisdata[7].Axis_Standstill); // R_TRIG
fb_stop_d2(Execute := rtrig_stop_d2.Q, Deceleration := gc_r_Stop_dec_Az, Axis := drive2); // MC_Stop

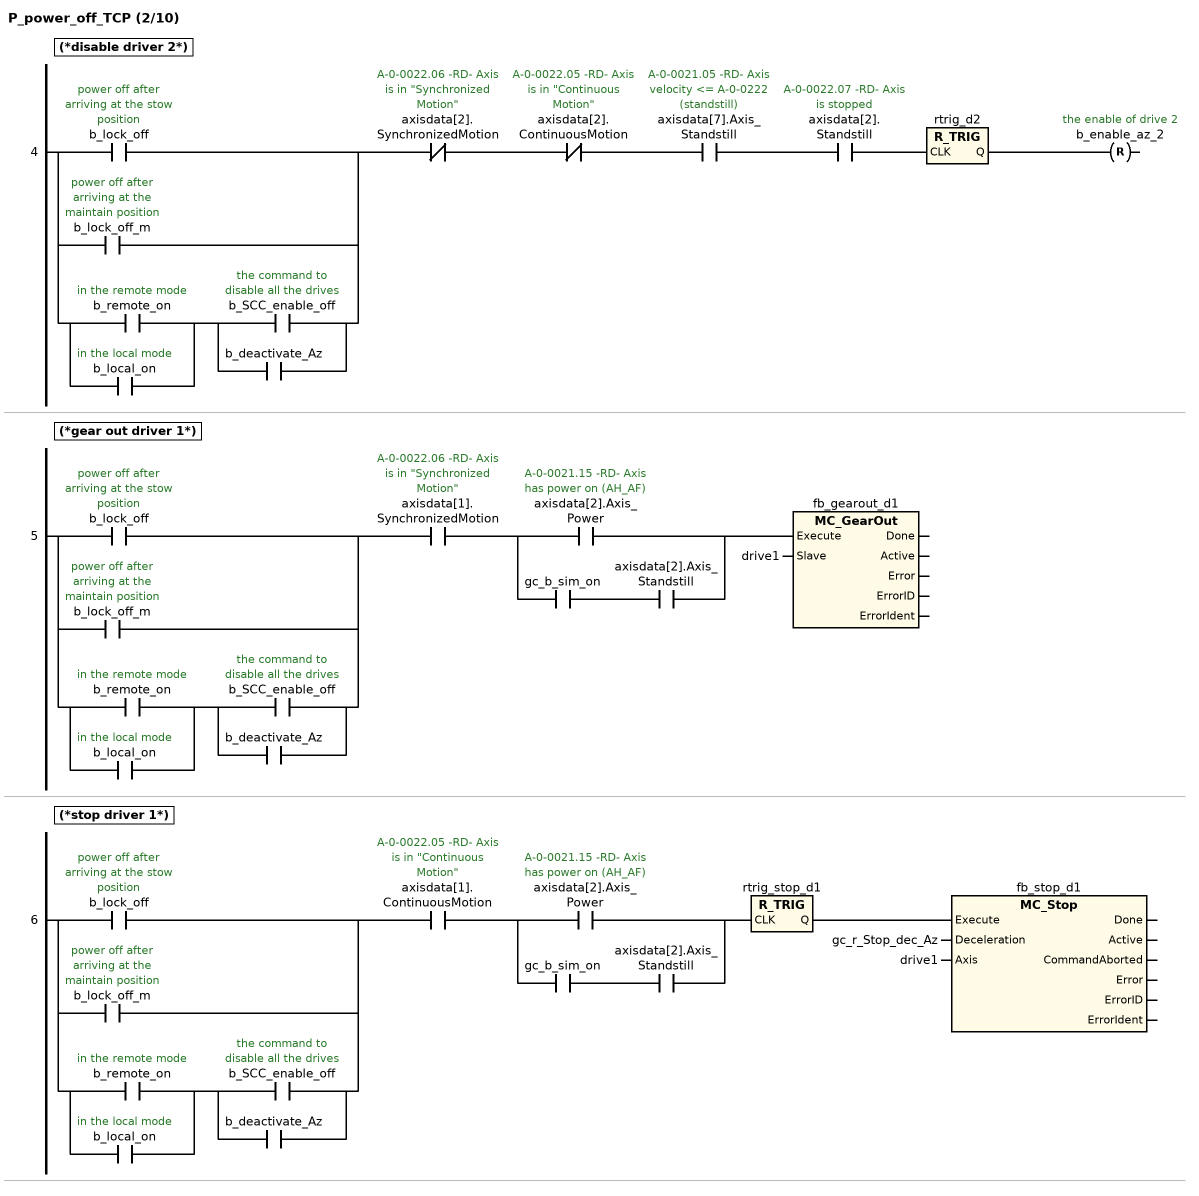
// NETWORK 4
//   b_lock_off: power off after arriving at the stow position
//   b_lock_off_m: power off after arriving at the maintain position
//   b_remote_on: in the remote mode
//   b_local_on: in the local mode
//   b_SCC_enable_off: the command to disable all the drives
//   axisdata[2].SynchronizedMotion: A-0-0022.06 -RD- Axis is in "Synchronized Motion"
//   axisdata[2].ContinuousMotion: A-0-0022.05 -RD- Axis is in "Continuous Motion"
//   axisdata[7].Axis_Standstill: A-0-0021.05 -RD- Axis velocity <= A-0-0222 (standstill)
//   axisdata[2].Standstill: A-0-0022.07 -RD- Axis is stopped
//   b_enable_az_2: the enable of drive 2
// label: (*disable driver 2*)
rtrig_d2(CLK := (b_lock_off OR b_lock_off_m OR (b_remote_on OR b_local_on) AND (b_SCC_enable_off OR b_deactivate_Az)) AND NOT axisdata[2].SynchronizedMotion AND NOT axisdata[2].ContinuousMotion AND axisdata[7].Axis_Standstill AND axisdata[2].Standstill); // R_TRIG
b_enable_az_2 R= rtrig_d2.Q;

// NETWORK 5
//   fb_gearout_d1: The firmware function block "MC_GearOut" is used to terminate an active synchronization function block.
//   b_lock_off: power off after arriving at the stow position
//   b_lock_off_m: power off after arriving at the maintain position
//   b_remote_on: in the remote mode
//   b_local_on: in the local mode
//   b_SCC_enable_off: the command to disable all the drives
//   axisdata[1].SynchronizedMotion: A-0-0022.06 -RD- Axis is in "Synchronized Motion"
//   axisdata[2].Axis_Power: A-0-0021.15 -RD- Axis has power on (AH_AF)
//   drive1: Real axis "Drive1" with axis number 1
// label: (*gear out driver 1*)
fb_gearout_d1(Execute := (b_lock_off OR b_lock_off_m OR (b_remote_on OR b_local_on) AND (b_SCC_enable_off OR b_deactivate_Az)) AND axisdata[1].SynchronizedMotion AND (axisdata[2].Axis_Power OR gc_b_sim_on AND axisdata[2].Axis_Standstill), Slave := drive1); // MC_GearOut

// NETWORK 6
//   b_lock_off: power off after arriving at the stow position
//   b_lock_off_m: power off after arriving at the maintain position
//   b_remote_on: in the remote mode
//   b_local_on: in the local mode
//   b_SCC_enable_off: the command to disable all the drives
//   axisdata[1].ContinuousMotion: A-0-0022.05 -RD- Axis is in "Continuous Motion"
//   axisdata[2].Axis_Power: A-0-0021.15 -RD- Axis has power on (AH_AF)
//   drive1: Real axis "Drive1" with axis number 1
// label: (*stop driver 1*)
rtrig_stop_d1(CLK := (b_lock_off OR b_lock_off_m OR (b_remote_on OR b_local_on) AND (b_SCC_enable_off OR b_deactivate_Az)) AND axisdata[1].ContinuousMotion AND (axisdata[2].Axis_Power OR gc_b_sim_on AND axisdata[2].Axis_Standstill)); // R_TRIG
fb_stop_d1(Execute := rtrig_stop_d1.Q, Deceleration := gc_r_Stop_dec_Az, Axis := drive1); // MC_Stop

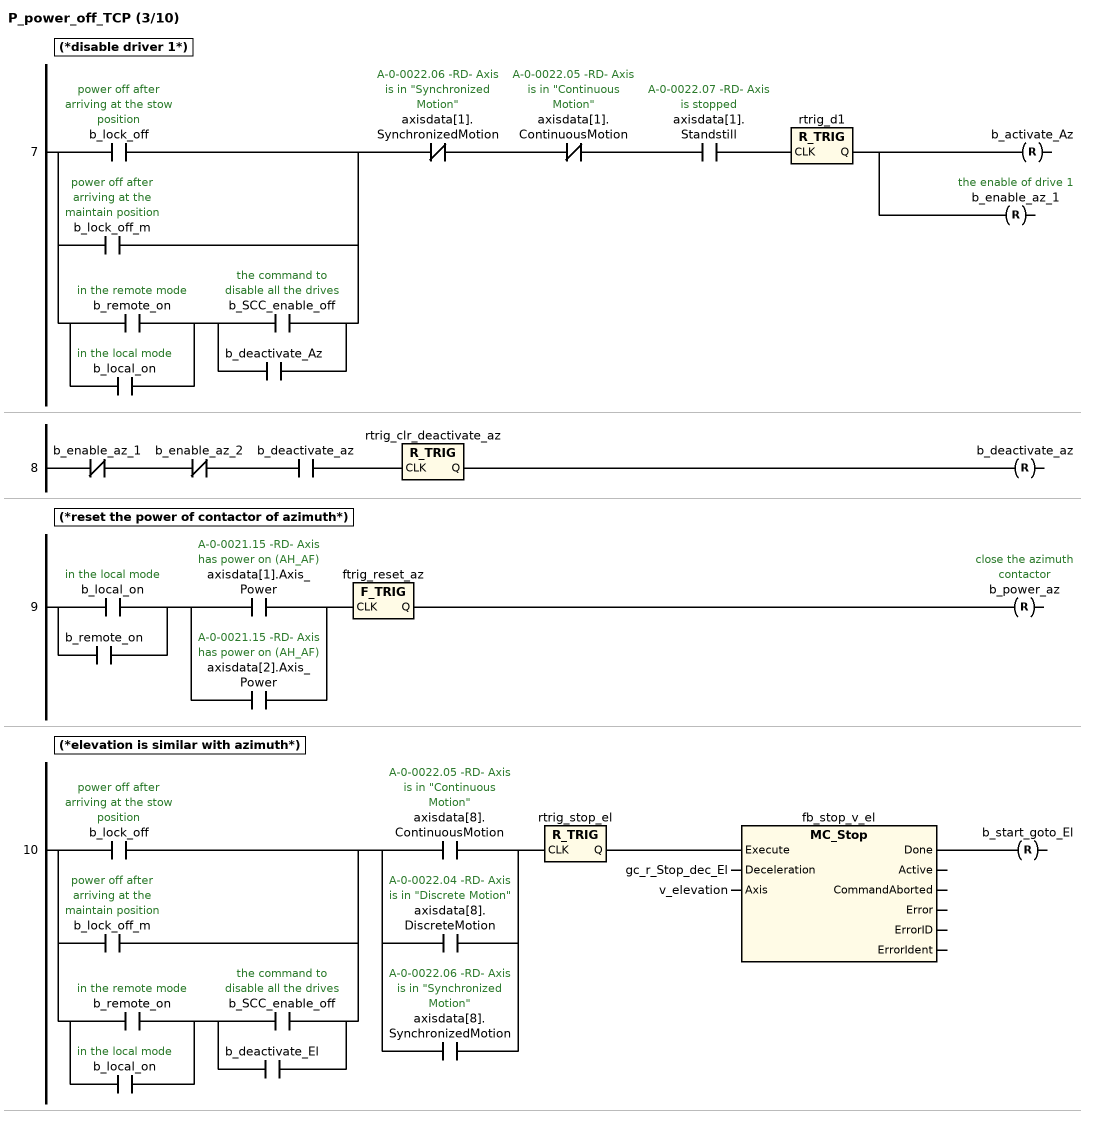
// NETWORK 7
//   b_lock_off: power off after arriving at the stow position
//   b_lock_off_m: power off after arriving at the maintain position
//   b_remote_on: in the remote mode
//   b_local_on: in the local mode
//   b_SCC_enable_off: the command to disable all the drives
//   axisdata[1].SynchronizedMotion: A-0-0022.06 -RD- Axis is in "Synchronized Motion"
//   axisdata[1].ContinuousMotion: A-0-0022.05 -RD- Axis is in "Continuous Motion"
//   axisdata[1].Standstill: A-0-0022.07 -RD- Axis is stopped
//   b_enable_az_1: the enable of drive 1
// label: (*disable driver 1*)
rtrig_d1(CLK := (b_lock_off OR b_lock_off_m OR (b_remote_on OR b_local_on) AND (b_SCC_enable_off OR b_deactivate_Az)) AND NOT axisdata[1].SynchronizedMotion AND NOT axisdata[1].ContinuousMotion AND axisdata[1].Standstill); // R_TRIG
b_activate_Az R= rtrig_d1.Q;
b_enable_az_1 R= rtrig_d1.Q;

// NETWORK 8
rtrig_clr_deactivate_az(CLK := NOT b_enable_az_1 AND NOT b_enable_az_2 AND b_deactivate_az); // R_TRIG
b_deactivate_az R= rtrig_clr_deactivate_az.Q;

// NETWORK 9
//   ftrig_reset_az: The function block F_TRIG a falling edge
//   b_local_on: in the local mode
//   axisdata[1].Axis_Power: A-0-0021.15 -RD- Axis has power on (AH_AF)
//   axisdata[2].Axis_Power: A-0-0021.15 -RD- Axis has power on (AH_AF)
//   b_power_az: close the azimuth contactor
// label: (*reset the power of contactor of azimuth*)
ftrig_reset_az(CLK := (b_local_on OR b_remote_on) AND (axisdata[1].Axis_Power OR axisdata[2].Axis_Power)); // F_TRIG
b_power_az R= ftrig_reset_az.Q;

// NETWORK 10
//   b_lock_off: power off after arriving at the stow position
//   b_lock_off_m: power off after arriving at the maintain position
//   b_remote_on: in the remote mode
//   b_local_on: in the local mode
//   b_SCC_enable_off: the command to disable all the drives
//   axisdata[8].ContinuousMotion: A-0-0022.05 -RD- Axis is in "Continuous Motion"
//   axisdata[8].DiscreteMotion: A-0-0022.04 -RD- Axis is in "Discrete Motion"
//   axisdata[8].SynchronizedMotion: A-0-0022.06 -RD- Axis is in "Synchronized Motion"
//   v_elevation: Virtual axis "v_elevation" with axis number 8
// label: (*elevation is similar with azimuth*)
rtrig_stop_el(CLK := (b_lock_off OR b_lock_off_m OR (b_remote_on OR b_local_on) AND (b_SCC_enable_off OR b_deactivate_El)) AND (axisdata[8].ContinuousMotion OR axisdata[8].DiscreteMotion OR axisdata[8].SynchronizedMotion)); // R_TRIG
fb_stop_v_el(Execute := rtrig_stop_el.Q, Deceleration := gc_r_Stop_dec_El, Axis := v_elevation); // MC_Stop
b_start_goto_El R= fb_stop_v_el.Done;

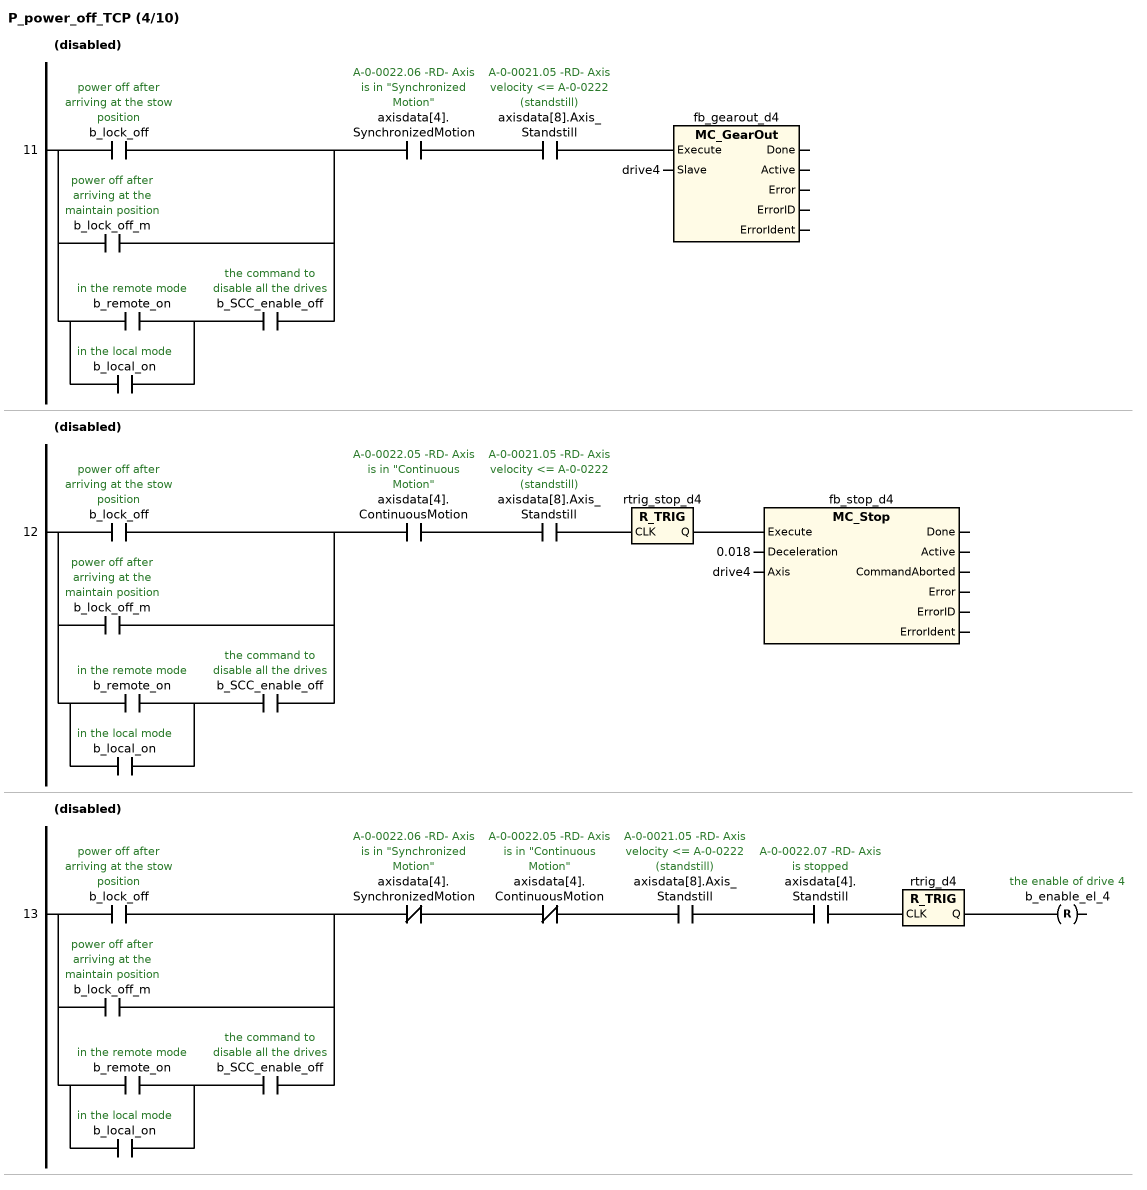
// NETWORK 11 (disabled)
//   b_lock_off: power off after arriving at the stow position
//   b_lock_off_m: power off after arriving at the maintain position
//   b_remote_on: in the remote mode
//   b_local_on: in the local mode
//   b_SCC_enable_off: the command to disable all the drives
//   axisdata[4].SynchronizedMotion: A-0-0022.06 -RD- Axis is in "Synchronized Motion"
//   axisdata[8].Axis_Standstill: A-0-0021.05 -RD- Axis velocity <= A-0-0222 (standstill)
//   drive4: Real axis "Drive4" with axis number 4
// fb_gearout_d4(Execute := (b_lock_off OR b_lock_off_m OR (b_remote_on OR b_local_on) AND b_SCC_enable_off) AND axisdata[4].SynchronizedMotion AND axisdata[8].Axis_Standstill, Slave := drive4); // MC_GearOut

// NETWORK 12 (disabled)
//   b_lock_off: power off after arriving at the stow position
//   b_lock_off_m: power off after arriving at the maintain position
//   b_remote_on: in the remote mode
//   b_local_on: in the local mode
//   b_SCC_enable_off: the command to disable all the drives
//   axisdata[4].ContinuousMotion: A-0-0022.05 -RD- Axis is in "Continuous Motion"
//   axisdata[8].Axis_Standstill: A-0-0021.05 -RD- Axis velocity <= A-0-0222 (standstill)
//   drive4: Real axis "Drive4" with axis number 4
// rtrig_stop_d4(CLK := (b_lock_off OR b_lock_off_m OR (b_remote_on OR b_local_on) AND b_SCC_enable_off) AND axisdata[4].ContinuousMotion AND axisdata[8].Axis_Standstill); // R_TRIG
// fb_stop_d4(Execute := rtrig_stop_d4.Q, Deceleration := 0.018, Axis := drive4); // MC_Stop

// NETWORK 13 (disabled)
//   b_lock_off: power off after arriving at the stow position
//   b_lock_off_m: power off after arriving at the maintain position
//   b_remote_on: in the remote mode
//   b_local_on: in the local mode
//   b_SCC_enable_off: the command to disable all the drives
//   axisdata[4].SynchronizedMotion: A-0-0022.06 -RD- Axis is in "Synchronized Motion"
//   axisdata[4].ContinuousMotion: A-0-0022.05 -RD- Axis is in "Continuous Motion"
//   axisdata[8].Axis_Standstill: A-0-0021.05 -RD- Axis velocity <= A-0-0222 (standstill)
//   axisdata[4].Standstill: A-0-0022.07 -RD- Axis is stopped
//   b_enable_el_4: the enable of drive 4
// rtrig_d4(CLK := (b_lock_off OR b_lock_off_m OR (b_remote_on OR b_local_on) AND b_SCC_enable_off) AND NOT axisdata[4].SynchronizedMotion AND NOT axisdata[4].ContinuousMotion AND axisdata[8].Axis_Standstill AND axisdata[4].Standstill); // R_TRIG
// b_enable_el_4 R= rtrig_d4.Q;

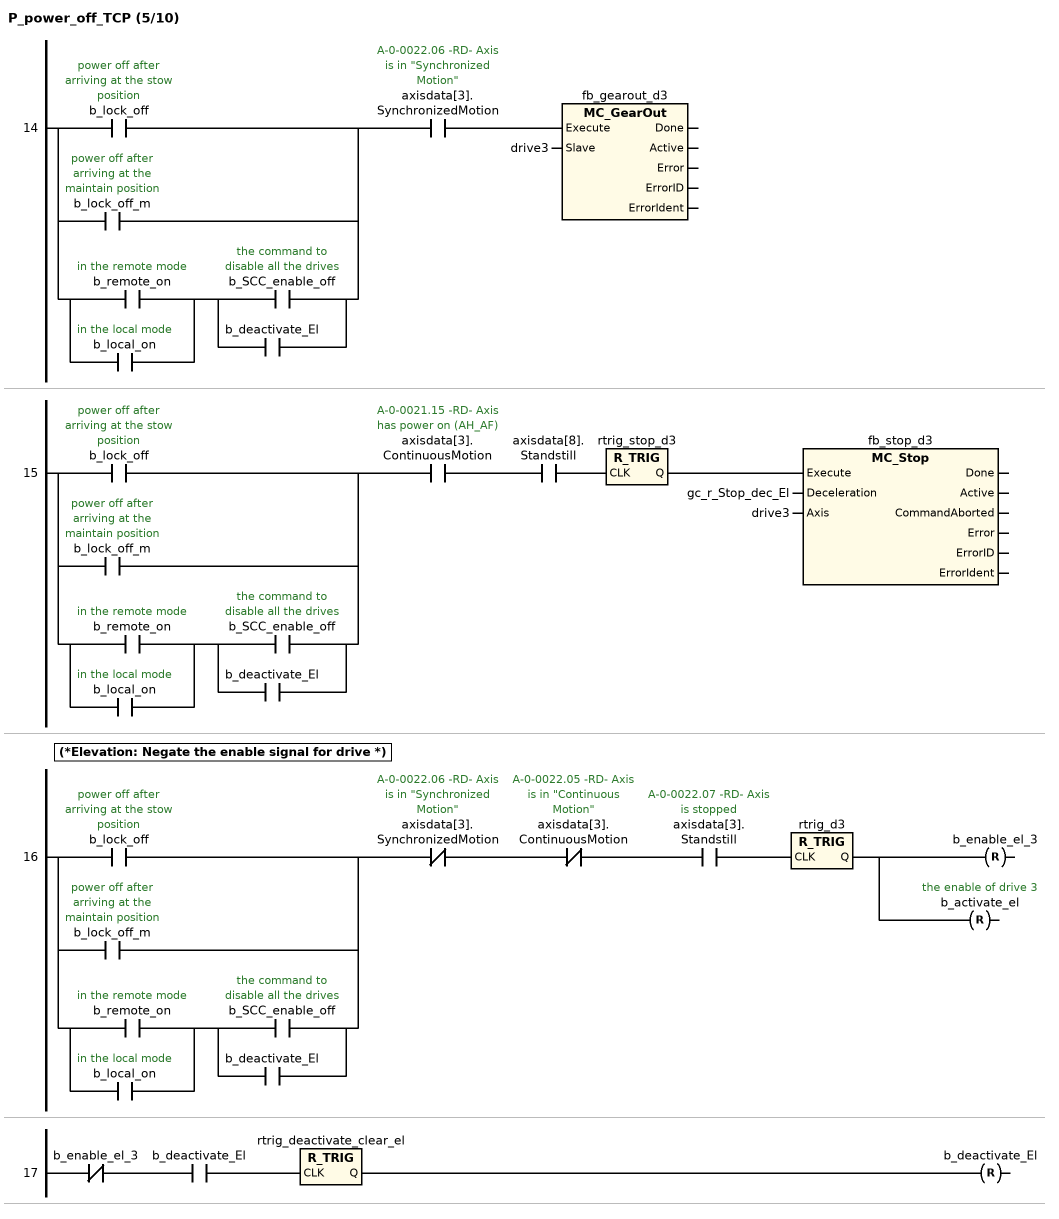
// NETWORK 14
//   b_lock_off: power off after arriving at the stow position
//   b_lock_off_m: power off after arriving at the maintain position
//   b_remote_on: in the remote mode
//   b_local_on: in the local mode
//   b_SCC_enable_off: the command to disable all the drives
//   axisdata[3].SynchronizedMotion: A-0-0022.06 -RD- Axis is in "Synchronized Motion"
//   drive3: Real axis "Drive3" with axis number 3
fb_gearout_d3(Execute := (b_lock_off OR b_lock_off_m OR (b_remote_on OR b_local_on) AND (b_SCC_enable_off OR b_deactivate_El)) AND axisdata[3].SynchronizedMotion, Slave := drive3); // MC_GearOut

// NETWORK 15
//   b_lock_off: power off after arriving at the stow position
//   b_lock_off_m: power off after arriving at the maintain position
//   b_remote_on: in the remote mode
//   b_local_on: in the local mode
//   b_SCC_enable_off: the command to disable all the drives
//   axisdata[3].ContinuousMotion: A-0-0021.15 -RD- Axis has power on (AH_AF)
//   drive3: Real axis "Drive3" with axis number 3
rtrig_stop_d3(CLK := (b_lock_off OR b_lock_off_m OR (b_remote_on OR b_local_on) AND (b_SCC_enable_off OR b_deactivate_El)) AND axisdata[3].ContinuousMotion AND axisdata[8].Standstill); // R_TRIG
fb_stop_d3(Execute := rtrig_stop_d3.Q, Deceleration := gc_r_Stop_dec_El, Axis := drive3); // MC_Stop

// NETWORK 16
//   b_lock_off: power off after arriving at the stow position
//   b_lock_off_m: power off after arriving at the maintain position
//   b_remote_on: in the remote mode
//   b_local_on: in the local mode
//   b_SCC_enable_off: the command to disable all the drives
//   axisdata[3].SynchronizedMotion: A-0-0022.06 -RD- Axis is in "Synchronized Motion"
//   axisdata[3].ContinuousMotion: A-0-0022.05 -RD- Axis is in "Continuous Motion"
//   axisdata[3].Standstill: A-0-0022.07 -RD- Axis is stopped
//   b_activate_el: the enable of drive 3
// label: (*Elevation: Negate the enable signal for drive *)
rtrig_d3(CLK := (b_lock_off OR b_lock_off_m OR (b_remote_on OR b_local_on) AND (b_SCC_enable_off OR b_deactivate_El)) AND NOT axisdata[3].SynchronizedMotion AND NOT axisdata[3].ContinuousMotion AND axisdata[3].Standstill); // R_TRIG
b_enable_el_3 R= rtrig_d3.Q;
b_activate_el R= rtrig_d3.Q;

// NETWORK 17
rtrig_deactivate_clear_el(CLK := NOT b_enable_el_3 AND b_deactivate_El); // R_TRIG
b_deactivate_El R= rtrig_deactivate_clear_el.Q;

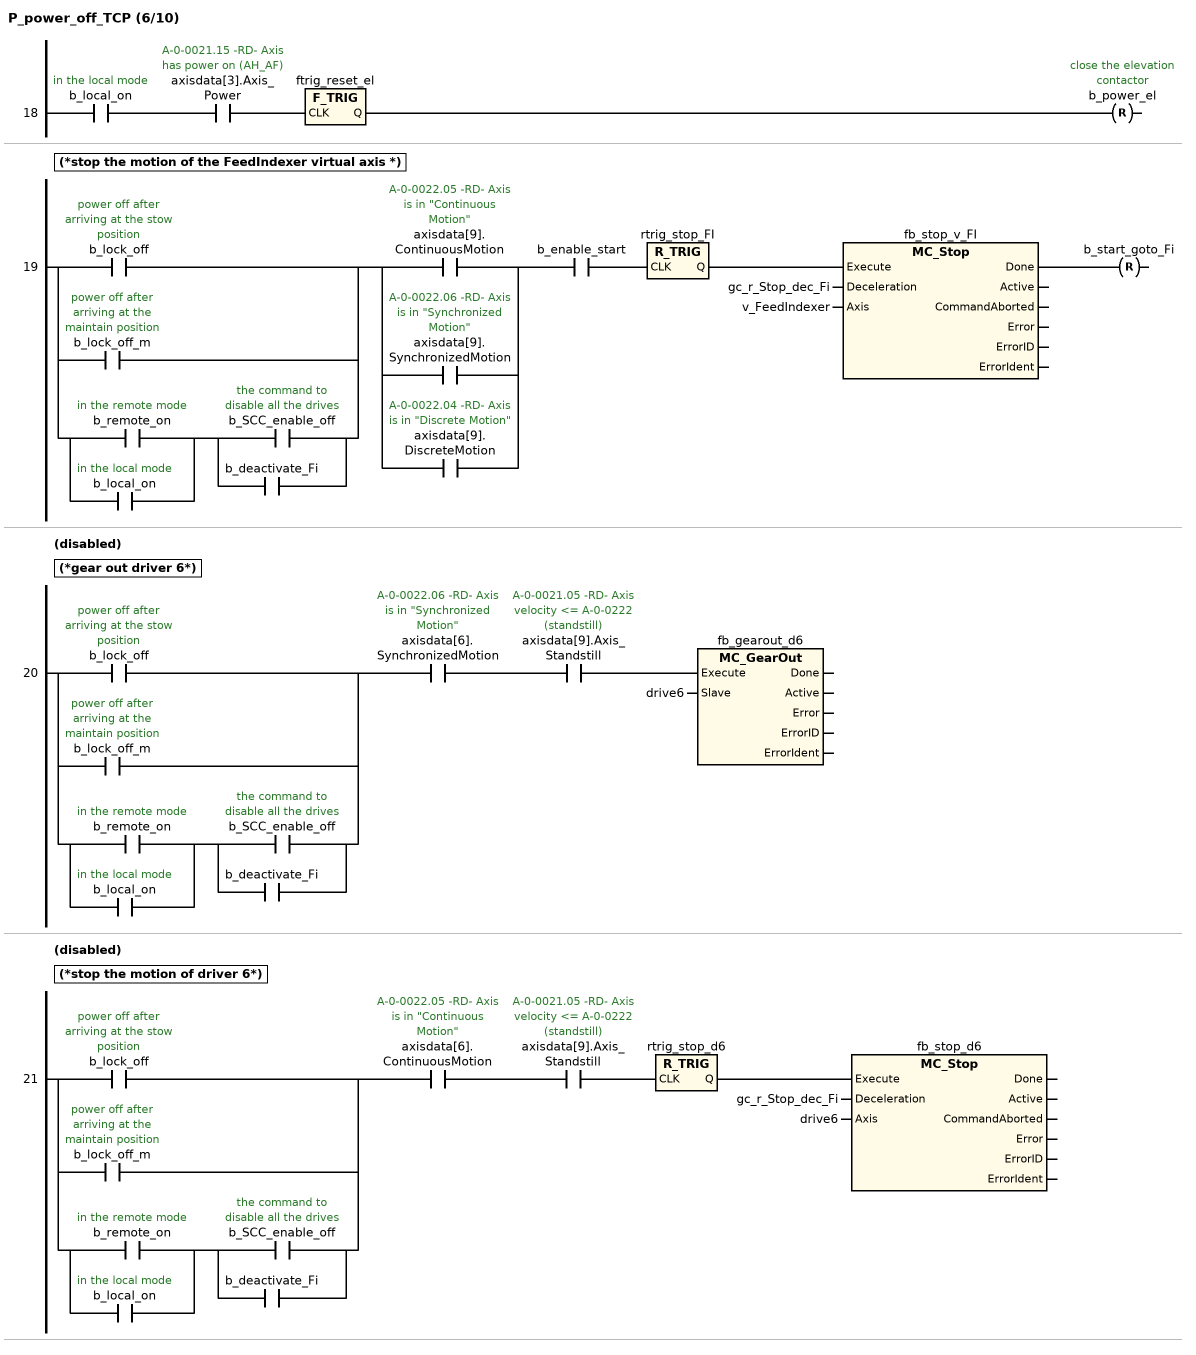
// NETWORK 18
//   b_local_on: in the local mode
//   axisdata[3].Axis_Power: A-0-0021.15 -RD- Axis has power on (AH_AF)
//   b_power_el: close the elevation contactor
ftrig_reset_el(CLK := b_local_on AND axisdata[3].Axis_Power); // F_TRIG
b_power_el R= ftrig_reset_el.Q;

// NETWORK 19
//   b_lock_off: power off after arriving at the stow position
//   b_lock_off_m: power off after arriving at the maintain position
//   b_remote_on: in the remote mode
//   b_local_on: in the local mode
//   b_SCC_enable_off: the command to disable all the drives
//   axisdata[9].ContinuousMotion: A-0-0022.05 -RD- Axis is in "Continuous Motion"
//   axisdata[9].SynchronizedMotion: A-0-0022.06 -RD- Axis is in "Synchronized Motion"
//   axisdata[9].DiscreteMotion: A-0-0022.04 -RD- Axis is in "Discrete Motion"
//   v_FeedIndexer: Virtual axis "v_polarization" with axis number 9
// label: (*stop the motion of the FeedIndexer virtual axis *)
rtrig_stop_FI(CLK := (b_lock_off OR b_lock_off_m OR (b_remote_on OR b_local_on) AND (b_SCC_enable_off OR b_deactivate_Fi)) AND (axisdata[9].ContinuousMotion OR axisdata[9].SynchronizedMotion OR axisdata[9].DiscreteMotion) AND b_enable_start); // R_TRIG
fb_stop_v_FI(Execute := rtrig_stop_FI.Q, Deceleration := gc_r_Stop_dec_Fi, Axis := v_FeedIndexer); // MC_Stop
b_start_goto_Fi R= fb_stop_v_FI.Done;

// NETWORK 20 (disabled)
//   b_lock_off: power off after arriving at the stow position
//   b_lock_off_m: power off after arriving at the maintain position
//   b_remote_on: in the remote mode
//   b_local_on: in the local mode
//   b_SCC_enable_off: the command to disable all the drives
//   axisdata[6].SynchronizedMotion: A-0-0022.06 -RD- Axis is in "Synchronized Motion"
//   axisdata[9].Axis_Standstill: A-0-0021.05 -RD- Axis velocity <= A-0-0222 (standstill)
//   drive6: Real axis "Drive6" with axis number 6
// label: (*gear out driver 6*)
// fb_gearout_d6(Execute := (b_lock_off OR b_lock_off_m OR (b_remote_on OR b_local_on) AND (b_SCC_enable_off OR b_deactivate_Fi)) AND axisdata[6].SynchronizedMotion AND axisdata[9].Axis_Standstill, Slave := drive6); // MC_GearOut

// NETWORK 21 (disabled)
//   b_lock_off: power off after arriving at the stow position
//   b_lock_off_m: power off after arriving at the maintain position
//   b_remote_on: in the remote mode
//   b_local_on: in the local mode
//   b_SCC_enable_off: the command to disable all the drives
//   axisdata[6].ContinuousMotion: A-0-0022.05 -RD- Axis is in "Continuous Motion"
//   axisdata[9].Axis_Standstill: A-0-0021.05 -RD- Axis velocity <= A-0-0222 (standstill)
//   drive6: Real axis "Drive6" with axis number 6
// label: (*stop the motion of driver 6*)
// rtrig_stop_d6(CLK := (b_lock_off OR b_lock_off_m OR (b_remote_on OR b_local_on) AND (b_SCC_enable_off OR b_deactivate_Fi)) AND axisdata[6].ContinuousMotion AND axisdata[9].Axis_Standstill); // R_TRIG
// fb_stop_d6(Execute := rtrig_stop_d6.Q, Deceleration := gc_r_Stop_dec_Fi, Axis := drive6); // MC_Stop

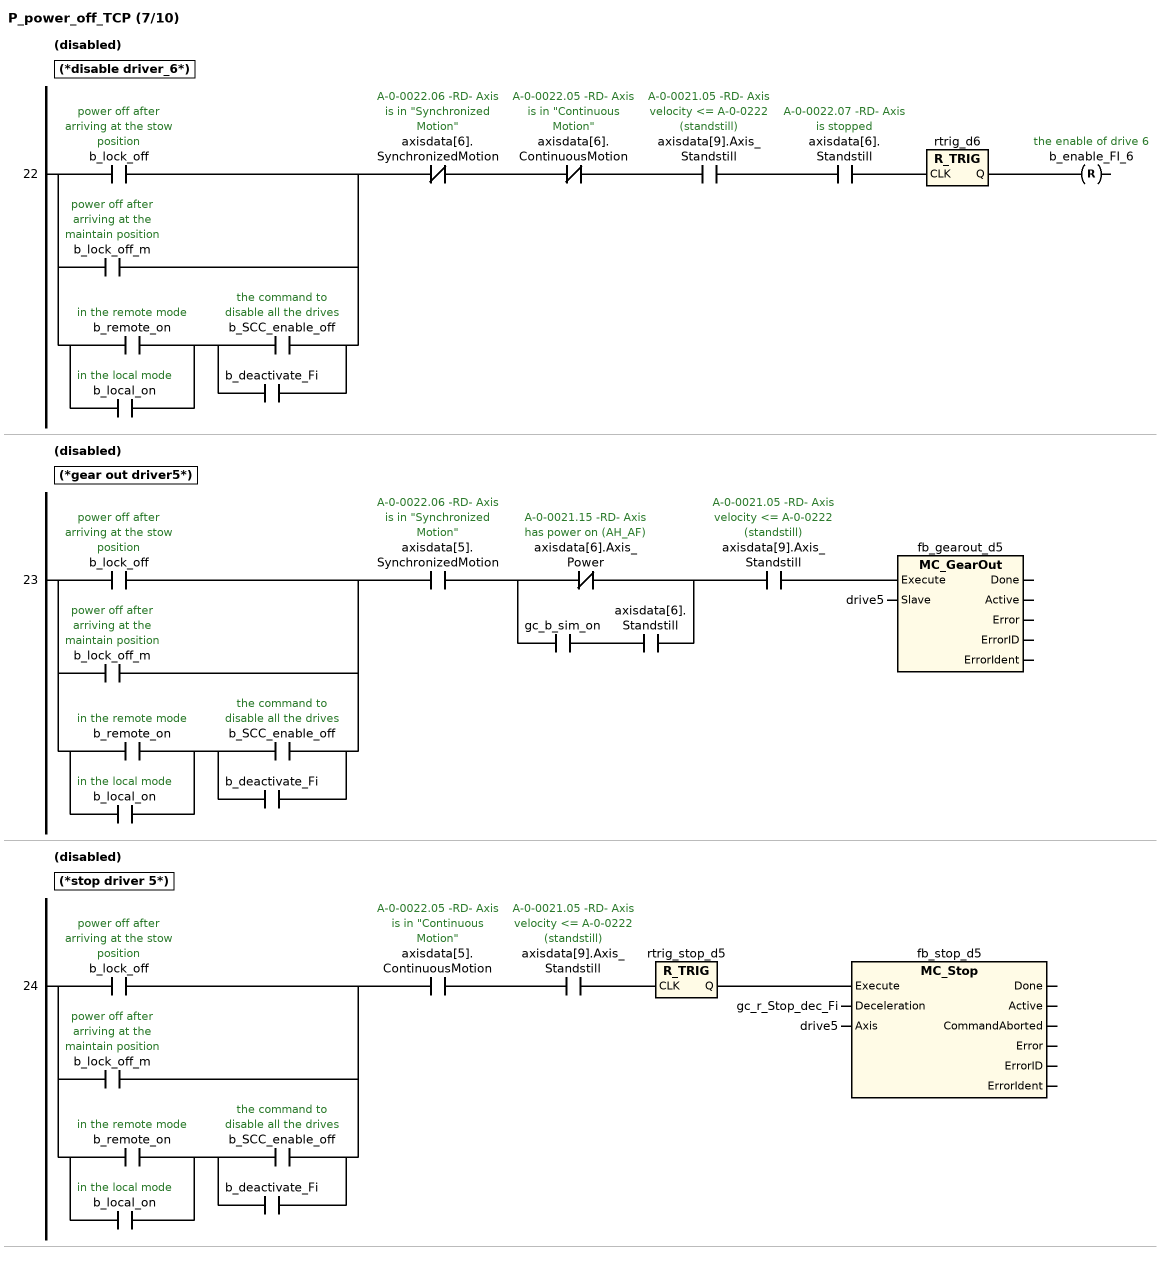
// NETWORK 22 (disabled)
//   b_lock_off: power off after arriving at the stow position
//   b_lock_off_m: power off after arriving at the maintain position
//   b_remote_on: in the remote mode
//   b_local_on: in the local mode
//   b_SCC_enable_off: the command to disable all the drives
//   axisdata[6].SynchronizedMotion: A-0-0022.06 -RD- Axis is in "Synchronized Motion"
//   axisdata[6].ContinuousMotion: A-0-0022.05 -RD- Axis is in "Continuous Motion"
//   axisdata[9].Axis_Standstill: A-0-0021.05 -RD- Axis velocity <= A-0-0222 (standstill)
//   axisdata[6].Standstill: A-0-0022.07 -RD- Axis is stopped
//   b_enable_FI_6: the enable of drive 6
// label: (*disable driver_6*)
// rtrig_d6(CLK := (b_lock_off OR b_lock_off_m OR (b_remote_on OR b_local_on) AND (b_SCC_enable_off OR b_deactivate_Fi)) AND NOT axisdata[6].SynchronizedMotion AND NOT axisdata[6].ContinuousMotion AND axisdata[9].Axis_Standstill AND axisdata[6].Standstill); // R_TRIG
// b_enable_FI_6 R= rtrig_d6.Q;

// NETWORK 23 (disabled)
//   b_lock_off: power off after arriving at the stow position
//   b_lock_off_m: power off after arriving at the maintain position
//   b_remote_on: in the remote mode
//   b_local_on: in the local mode
//   b_SCC_enable_off: the command to disable all the drives
//   axisdata[5].SynchronizedMotion: A-0-0022.06 -RD- Axis is in "Synchronized Motion"
//   axisdata[6].Axis_Power: A-0-0021.15 -RD- Axis has power on (AH_AF)
//   axisdata[9].Axis_Standstill: A-0-0021.05 -RD- Axis velocity <= A-0-0222 (standstill)
//   drive5: Real axis "Drive5" with axis number 5
// label: (*gear out driver5*)
// fb_gearout_d5(Execute := (b_lock_off OR b_lock_off_m OR (b_remote_on OR b_local_on) AND (b_SCC_enable_off OR b_deactivate_Fi)) AND axisdata[5].SynchronizedMotion AND (NOT axisdata[6].Axis_Power OR gc_b_sim_on AND axisdata[6].Standstill) AND axisdata[9].Axis_Standstill, Slave := drive5); // MC_GearOut

// NETWORK 24 (disabled)
//   b_lock_off: power off after arriving at the stow position
//   b_lock_off_m: power off after arriving at the maintain position
//   b_remote_on: in the remote mode
//   b_local_on: in the local mode
//   b_SCC_enable_off: the command to disable all the drives
//   axisdata[5].ContinuousMotion: A-0-0022.05 -RD- Axis is in "Continuous Motion"
//   axisdata[9].Axis_Standstill: A-0-0021.05 -RD- Axis velocity <= A-0-0222 (standstill)
//   drive5: Real axis "Drive5" with axis number 5
// label: (*stop driver 5*)
// rtrig_stop_d5(CLK := (b_lock_off OR b_lock_off_m OR (b_remote_on OR b_local_on) AND (b_SCC_enable_off OR b_deactivate_Fi)) AND axisdata[5].ContinuousMotion AND axisdata[9].Axis_Standstill); // R_TRIG
// fb_stop_d5(Execute := rtrig_stop_d5.Q, Deceleration := gc_r_Stop_dec_Fi, Axis := drive5); // MC_Stop

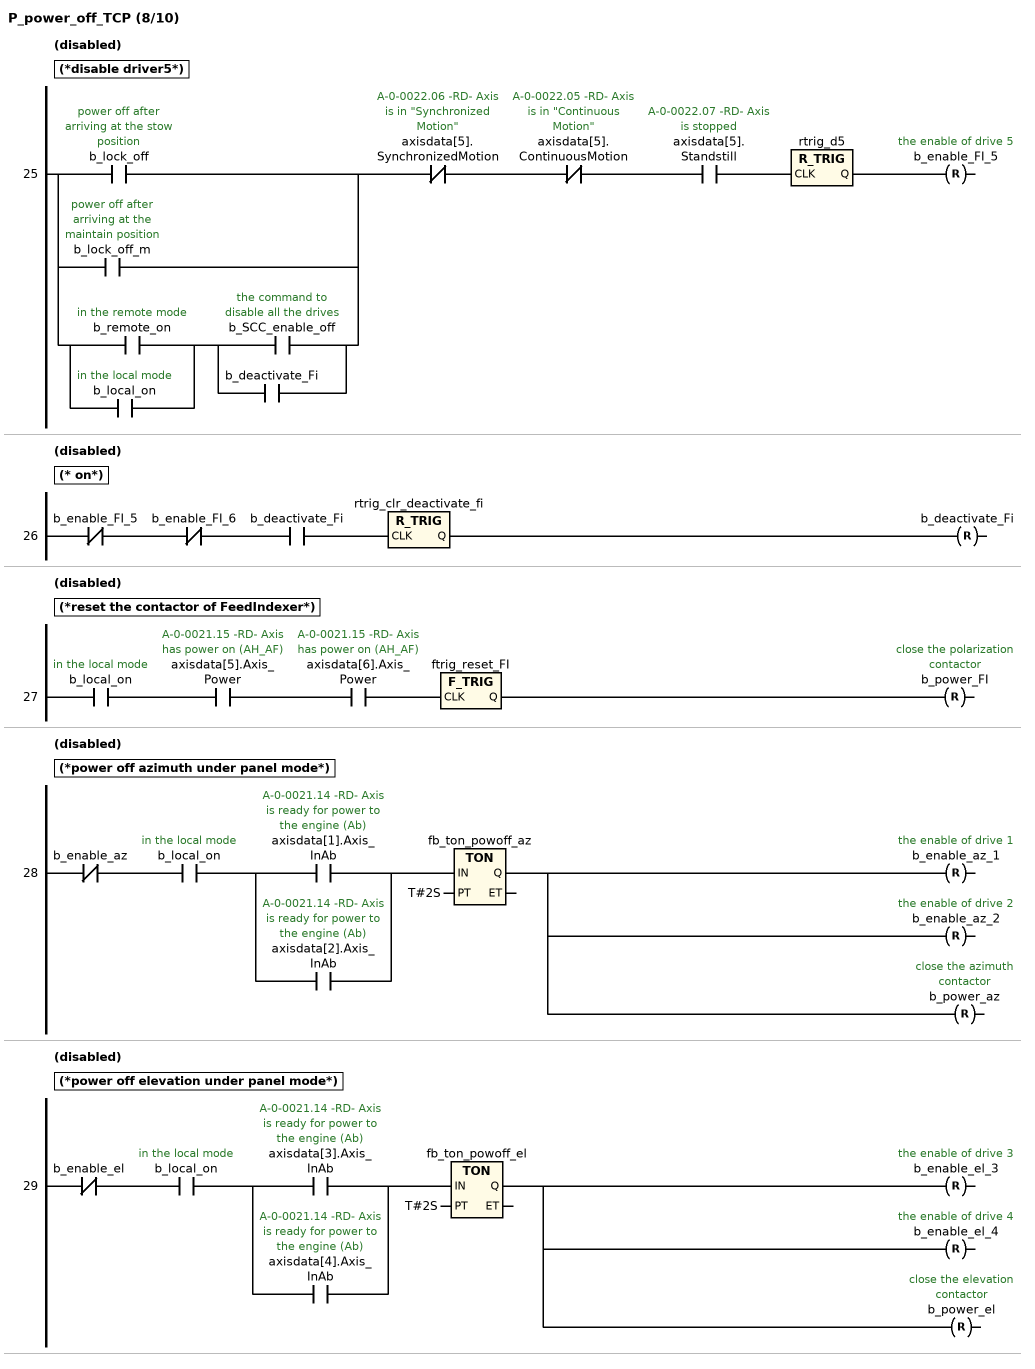
// NETWORK 25 (disabled)
//   b_lock_off: power off after arriving at the stow position
//   b_lock_off_m: power off after arriving at the maintain position
//   b_remote_on: in the remote mode
//   b_local_on: in the local mode
//   b_SCC_enable_off: the command to disable all the drives
//   axisdata[5].SynchronizedMotion: A-0-0022.06 -RD- Axis is in "Synchronized Motion"
//   axisdata[5].ContinuousMotion: A-0-0022.05 -RD- Axis is in "Continuous Motion"
//   axisdata[5].Standstill: A-0-0022.07 -RD- Axis is stopped
//   b_enable_FI_5: the enable of drive 5
// label: (*disable driver5*)
// rtrig_d5(CLK := (b_lock_off OR b_lock_off_m OR (b_remote_on OR b_local_on) AND (b_SCC_enable_off OR b_deactivate_Fi)) AND NOT axisdata[5].SynchronizedMotion AND NOT axisdata[5].ContinuousMotion AND axisdata[5].Standstill); // R_TRIG
// b_enable_FI_5 R= rtrig_d5.Q;

// NETWORK 26 (disabled)
// label: (* on*)
// rtrig_clr_deactivate_fi(CLK := NOT b_enable_FI_5 AND NOT b_enable_FI_6 AND b_deactivate_Fi); // R_TRIG
// b_deactivate_Fi R= rtrig_clr_deactivate_fi.Q;

// NETWORK 27 (disabled)
//   b_local_on: in the local mode
//   axisdata[5].Axis_Power: A-0-0021.15 -RD- Axis has power on (AH_AF)
//   axisdata[6].Axis_Power: A-0-0021.15 -RD- Axis has power on (AH_AF)
//   b_power_FI: close the polarization contactor
// label: (*reset the contactor of FeedIndexer*)
// ftrig_reset_FI(CLK := b_local_on AND axisdata[5].Axis_Power AND axisdata[6].Axis_Power); // F_TRIG
// b_power_FI R= ftrig_reset_FI.Q;

// NETWORK 28 (disabled)
//   fb_ton_powoff_az: The function block Timer On Delay implements a turn-on delay..
//   b_local_on: in the local mode
//   axisdata[1].Axis_InAb: A-0-0021.14 -RD- Axis is ready for power to the engine (Ab)
//   axisdata[2].Axis_InAb: A-0-0021.14 -RD- Axis is ready for power to the engine (Ab)
//   b_enable_az_1: the enable of drive 1
//   b_enable_az_2: the enable of drive 2
//   b_power_az: close the azimuth contactor
// label: (*power off azimuth under panel mode*)
// fb_ton_powoff_az(IN := NOT b_enable_az AND b_local_on AND (axisdata[1].Axis_InAb OR axisdata[2].Axis_InAb), PT := T#2S); // TON
// b_enable_az_1 R= fb_ton_powoff_az.Q;
// b_enable_az_2 R= fb_ton_powoff_az.Q;
// b_power_az R= fb_ton_powoff_az.Q;

// NETWORK 29 (disabled)
//   b_local_on: in the local mode
//   axisdata[3].Axis_InAb: A-0-0021.14 -RD- Axis is ready for power to the engine (Ab)
//   axisdata[4].Axis_InAb: A-0-0021.14 -RD- Axis is ready for power to the engine (Ab)
//   b_enable_el_3: the enable of drive 3
//   b_enable_el_4: the enable of drive 4
//   b_power_el: close the elevation contactor
// label: (*power off elevation under panel mode*)
// fb_ton_powoff_el(IN := NOT b_enable_el AND b_local_on AND (axisdata[3].Axis_InAb OR axisdata[4].Axis_InAb), PT := T#2S); // TON
// b_enable_el_3 R= fb_ton_powoff_el.Q;
// b_enable_el_4 R= fb_ton_powoff_el.Q;
// b_power_el R= fb_ton_powoff_el.Q;

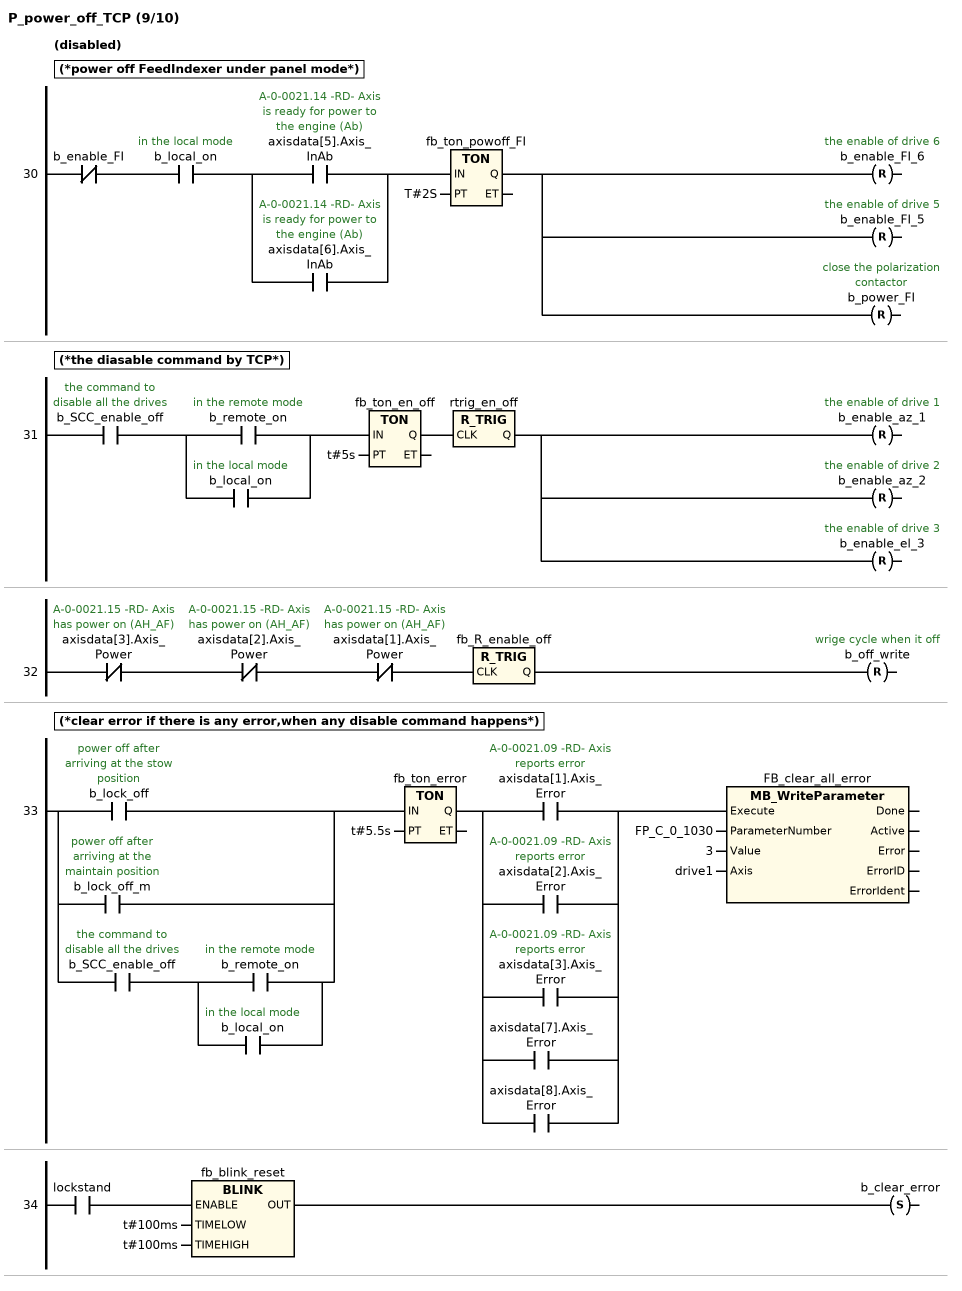
// NETWORK 30 (disabled)
//   b_local_on: in the local mode
//   axisdata[5].Axis_InAb: A-0-0021.14 -RD- Axis is ready for power to the engine (Ab)
//   axisdata[6].Axis_InAb: A-0-0021.14 -RD- Axis is ready for power to the engine (Ab)
//   b_enable_FI_6: the enable of drive 6
//   b_enable_FI_5: the enable of drive 5
//   b_power_FI: close the polarization contactor
// label: (*power off FeedIndexer under panel mode*)
// fb_ton_powoff_FI(IN := NOT b_enable_FI AND b_local_on AND (axisdata[5].Axis_InAb OR axisdata[6].Axis_InAb), PT := T#2S); // TON
// b_enable_FI_6 R= fb_ton_powoff_FI.Q;
// b_enable_FI_5 R= fb_ton_powoff_FI.Q;
// b_power_FI R= fb_ton_powoff_FI.Q;

// NETWORK 31
//   b_SCC_enable_off: the command to disable all the drives
//   b_remote_on: in the remote mode
//   b_local_on: in the local mode
//   b_enable_az_1: the enable of drive 1
//   b_enable_az_2: the enable of drive 2
//   b_enable_el_3: the enable of drive 3
// label: (*the diasable command by TCP*)
fb_ton_en_off(IN := b_SCC_enable_off AND (b_remote_on OR b_local_on), PT := t#5s); // TON
rtrig_en_off(CLK := fb_ton_en_off.Q); // R_TRIG
b_enable_az_1 R= rtrig_en_off.Q;
b_enable_az_2 R= rtrig_en_off.Q;
b_enable_el_3 R= rtrig_en_off.Q;

// NETWORK 32
//   axisdata[3].Axis_Power: A-0-0021.15 -RD- Axis has power on (AH_AF)
//   axisdata[2].Axis_Power: A-0-0021.15 -RD- Axis has power on (AH_AF)
//   axisdata[1].Axis_Power: A-0-0021.15 -RD- Axis has power on (AH_AF)
//   b_off_write: wrige cycle when it off
fb_R_enable_off(CLK := NOT axisdata[3].Axis_Power AND NOT axisdata[2].Axis_Power AND NOT axisdata[1].Axis_Power); // R_TRIG
b_off_write R= fb_R_enable_off.Q;

// NETWORK 33
//   b_lock_off: power off after arriving at the stow position
//   b_lock_off_m: power off after arriving at the maintain position
//   b_SCC_enable_off: the command to disable all the drives
//   b_remote_on: in the remote mode
//   b_local_on: in the local mode
//   axisdata[1].Axis_Error: A-0-0021.09 -RD- Axis reports error
//   axisdata[2].Axis_Error: A-0-0021.09 -RD- Axis reports error
//   axisdata[3].Axis_Error: A-0-0021.09 -RD- Axis reports error
//   FP_C_0_1030: Command: Clear all control errors
//   drive1: Real axis "Drive1" with axis number 1
// label: (*clear error if there is any error,when any disable command happens*)
fb_ton_error(IN := b_lock_off OR b_lock_off_m OR b_SCC_enable_off AND (b_remote_on OR b_local_on), PT := t#5.5s); // TON
FB_clear_all_error(
    Execute := fb_ton_error.Q AND (axisdata[1].Axis_Error OR axisdata[2].Axis_Error OR axisdata[3].Axis_Error OR axisdata[7].Axis_Error OR axisdata[8].Axis_Error),
    ParameterNumber := FP_C_0_1030,
    Value := 3,
    Axis := drive1); // MB_WriteParameter

// NETWORK 34
fb_blink_reset(ENABLE := lockstand, TIMELOW := t#100ms, TIMEHIGH := t#100ms); // BLINK
b_clear_error S= fb_blink_reset.OUT;

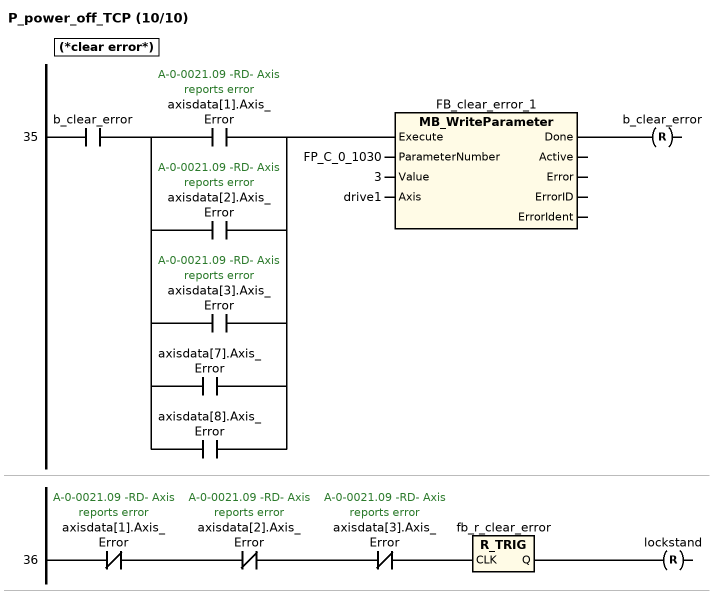
// NETWORK 35
//   axisdata[1].Axis_Error: A-0-0021.09 -RD- Axis reports error
//   axisdata[2].Axis_Error: A-0-0021.09 -RD- Axis reports error
//   axisdata[3].Axis_Error: A-0-0021.09 -RD- Axis reports error
//   FP_C_0_1030: Command: Clear all control errors
//   drive1: Real axis "Drive1" with axis number 1
// label: (*clear error*)
FB_clear_error_1(
    Execute := b_clear_error AND (axisdata[1].Axis_Error OR axisdata[2].Axis_Error OR axisdata[3].Axis_Error OR axisdata[7].Axis_Error OR axisdata[8].Axis_Error),
    ParameterNumber := FP_C_0_1030,
    Value := 3,
    Axis := drive1); // MB_WriteParameter
b_clear_error R= FB_clear_error_1.Done;

// NETWORK 36
//   axisdata[1].Axis_Error: A-0-0021.09 -RD- Axis reports error
//   axisdata[2].Axis_Error: A-0-0021.09 -RD- Axis reports error
//   axisdata[3].Axis_Error: A-0-0021.09 -RD- Axis reports error
fb_r_clear_error(CLK := NOT axisdata[1].Axis_Error AND NOT axisdata[2].Axis_Error AND NOT axisdata[3].Axis_Error); // R_TRIG
lockstand R= fb_r_clear_error.Q;

END_PROGRAM

// IndraMotionMlc1/Application/POUs/TCP/P_UDP_with_DAM
(*This program is built for UDP communication, receive the message from CSIRO,deal with the commands,and send the reply to CSIRO*)
PROGRAM P_UDP_with_DAM
VAR
(*<<<<<<<<<<<<<<<<<<<<<<<<<<<<<<<<<<<<<<<<<<<>>>>>>>>>>>>>>>>>>>>>>>>>>>>>>>>>>>>>*)
	b_receiving :BOOL;
	b_receiving_1 :BOOL;
	b_receiving_2 :BOOL;
	b_receiving_3 :BOOL;
	b_commanding: BOOL;
	b_commanding_1: BOOL;
	b_commanding_2: BOOL;
	b_commanding_3: BOOL;
	b_sending: BOOL;
	b_sending_1: BOOL;
	b_sending_2: BOOL;
	b_sending_3: BOOL;
	
(*<<<<<<<<<<<<<<<<<<<<<<<<<<<<<<<<<<<<<<<<<<<CONNECTION>>>>>>>>>>>>>>>>>>>>>>>>>>>>>>>>>>>>>*)
	UDPConnection_1: IL_UDPSocketAsync;
	UDPConnection_2: IL_UDPSocketAsync;
	UDPConnection_3: IL_UDPSocketAsync;
	b_Server_Enable: BOOL:=TRUE;(*the enable of IL_TCPConnectionAsync*)
	b_Server_Enable_1: BOOL:=TRUE;(*the enable of IL_TCPConnectionAsync*)
	b_Server_Enable_2: BOOL:=TRUE;(*the enable of IL_TCPConnectionAsync*)
	b_Server_Enable_3: BOOL:=TRUE;(*the enable of IL_TCPConnectionAsync*)
	di_Socket: DINT;(*the socket number*)
	di_Socket_1: DINT;(*the socket number*)
	di_Socket_2: DINT;(*the socket number*)
	di_Socket_3: DINT;(*the socket number*)
	strIP: STRING;
	b_Connection_done: BOOL;
	b_Connection_done_1: BOOL;
	b_Connection_done_2: BOOL;
	b_Connection_done_3: BOOL;
(*<<<<<<<<<<<<<<<<<<<<<<<<<<<<<<<<<<<<<<<<<<<RECEIVE>>>>>>>>>>>>>>>>>>>>>>>>>>>>>>>>>>>>>*)
	UDPRecv_1: IL_UDPRecvfromAsync;
	UDPRecv_2: IL_UDPRecvfromAsync;
	UDPRecv_3: IL_UDPRecvfromAsync;
	b_Recv_enable: BOOL;
	b_Recv_enable_1: BOOL;
	b_Recv_enable_2: BOOL;
	b_Recv_enable_3: BOOL;
	b_Recv_done: BOOL;
	b_Recv_done_1: BOOL;
	b_Recv_done_2: BOOL;
	b_Recv_done_3: BOOL;
	str_Recv: STRING(255);
	str_Recv_1: ARRAY [1..200] OF BYTE;
	str_Recv_2: ARRAY [1..200] OF BYTE;
	str_Recv_3: ARRAY [1..200] OF BYTE;
	//fb_crc16 : CRC16_MODBUS;
	di_ReceivedBytes: DINT;
	di_ReceivedBytes_1: DINT;
	di_ReceivedBytes_2: DINT;
	di_ReceivedBytes_3: DINT;
(*<<<<<<<<<<<<<<<<<<<<<<<<<<<<<<<<<<<<<<<<<<<<SEND>>>>>>>>>>>>>>>>>>>>>>>>>>>>>>>>>>>>>*)
	UDPSend_1: IL_UDPSendtoAsync;
	UDPSend_2: IL_UDPSendtoAsync;
	UDPSend_3: IL_UDPSendtoAsync;
	b_Send_enable: BOOL;
	b_Send_enable_1: BOOL;
	b_Send_enable_2: BOOL;
	b_Send_enable_3: BOOL;
	b_Send_done: BOOL;
	b_Send_done_1: BOOL;
	b_Send_done_2: BOOL;
	b_Send_done_3: BOOL;
	str_Send: STRING(1000);
	str_Send_1: ARRAY [1..8] OF BYTE;
	str_Send_2: ARRAY [1..8] OF BYTE;
	str_Send_3: ARRAY [1..8] OF BYTE;
	di_SentBytes: DINT;
	di_SentBytes_1: DINT;
	di_SentBytes_2: DINT;
	di_SentBytes_3: DINT;
	
	di_SentBytesLen_1: UINT;
	di_SentBytesLen_2: UINT;
	di_SentBytesLen_3: UINT;

(*add the function of close TCP function*)
	fb_tcp_close: IL_UDPCloseAsync;
	fb_udp_close_1: IL_UDPCloseAsync;
	fb_udp_close_2: IL_UDPCloseAsync;
	fb_udp_close_3: IL_UDPCloseAsync;
	B_TCP_close: BOOL;
	B_TCP_close_1: BOOL;
	B_TCP_close_2: BOOL;
	B_TCP_close_3: BOOL;
	b_TCP_close_done: BOOL;
	b_TCP_close_done_1: BOOL;
	b_TCP_close_done_2: BOOL;
	b_TCP_close_done_3: BOOL;
	b_Recv_active: BOOL;
	b_Recv_active_1: BOOL;
	b_Recv_active_2: BOOL;
	b_Recv_active_3: BOOL;
	i_counter_udp1:INT;
	i_counter_udp2:INT;
	i_counter_udp3:INT;

	str_concat: ARRAY[1..40] OF STRING(1000);(*数组及其类型的定义*)	
	str_concat_1: ARRAY[1..40] OF BYTE;(*数组及其类型的定义*)
	str_concat_2: ARRAY[1..40] OF BYTE;(*数组及其类型的定义*)
	str_concat_3: ARRAY[1..40] OF BYTE;(*数组及其类型的定义*)
	Counter: INT;
	bWaiting4Connection: BOOL;
	bWaiting4Connection_1: BOOL;
	bWaiting4Connection_2: BOOL;
	bWaiting4Connection_3: BOOL;
	bConnError: BOOL;
	bConnError_1: BOOL;
	bConnError_2: BOOL;
	bConnError_3: BOOL;
	diConnError: ERROR_CODE;
	diConnError_1: ERROR_CODE;
	diConnError_2: ERROR_CODE;
	diConnError_3: ERROR_CODE;
	ConnectError: ERROR_STRUCT;
	ConnectError_1: ERROR_STRUCT;
	ConnectError_2: ERROR_STRUCT;
	ConnectError_3: ERROR_STRUCT;
	i_counter_1s: INT:=0;	
	i_count:INT;
	
	reply_count: DINT;
	index: BYTE;
	
	dam1_data1 : LREAL;
	dam1_data2 : LREAL;
	dam1_data3 : LREAL;
	dam1_data4 : LREAL;
	dam1_data5 : LREAL;
	dam1_data6 : LREAL;
	dam1_data7 : LREAL;
	dam1_data8 : LREAL;
	dam1_data9 : LREAL;
	dam1_data10 : LREAL;
	dam1_data11 : LREAL;
	dam1_data12 : LREAL;
	

	
	dam3_data1 : REAL;
	dam3_data2 : REAL;
	dam3_data3 : REAL;
	dam3_data4 : REAL;
	dam3_data5 : REAL;
	dam3_data6 : REAL;
	dam3_data7 : REAL;
	dam3_data8 : REAL;
	dam3_data9 : REAL;
	dam3_data10 : REAL;
	dam3_data11 : REAL;
	dam3_data12 : REAL;
	dam3_data13 : REAL;
	dam3_data14 : REAL;
	dam3_data15 : REAL;
	dam3_data16 : REAL;
	dam3_data17 : REAL;
	dam3_data18 : REAL;
	dam3_data19 : REAL;
	dam3_data20 : REAL;
	dam3_data21 : REAL;
	dam3_data22 : REAL;
	dam3_data23 : REAL;
	dam3_data24 : REAL;
	dam3_data25 : REAL;
	dam3_data26 : REAL;
	dam3_data27 : REAL;
	dam3_data28 : REAL;
	fb_crc16_modbus: CRC16_MODBUS;
	
	a_phase_current : REAL;
	b_phase_current : REAL;
	c_phase_current : REAL;
	a_phase_voltage : REAL;
	b_phase_voltage : REAL;
	c_phase_voltage : REAL;
	ab_line_voltage : REAL;
	bc_line_voltage : REAL;
	ca_line_voltage : REAL;
	a_phase_activepower : REAL;
	b_phase_activepower : REAL;
	c_phase_activepower : REAL;
	a_phase_reactivepower : REAL;
	b_phase_reactivepower : REAL;
	c_phase_reactivepower : REAL;
	a_phase_apparentpower : REAL;
	b_phase_apparentpower : REAL;
	c_phase_apparentpower : REAL;
	a_phase_powerfactor : REAL;
	b_phase_powerfactor : REAL;
	c_phase_powerfactor : REAL;
	a_phase_frequency : REAL;
	b_phase_frequency : REAL;
	c_phase_frequency : REAL;
	total_activepower : REAL;
	total_reactivepower : REAL;
	total_apparentpower : REAL;
	total_powerfactor : REAL;
	
	
	X_Axis_Tile_Monitor : LREAL;
	Y_Axis_Tile_Monitor : LREAL;
	Temp_Tile_Monitor : LREAL;
	
	HumidEMISC_Outlet: LREAL;
END_VAR


reply_count:=reply_count+1;

IF reply_count < 0 OR reply_count >= 40 THEN	
	reply_count:=0;
END_IF

IF reply_count >= 0 AND reply_count < 10 THEN 
(*<<<<<<<<<<<<<<<<<<<<<<<<<<<<<concatenate STR_DAM1>>>>>>>>>>>>>>>>>>>>>>>>>>>>>>>>>>>>>>>>>>>>>>>>>>>>>>>*)
	str_concat_1[1] := 16#01;	//设备地址1
	str_concat_1[2] := 16#04;	//功能码
	str_concat_1[3] := 16#00;	//寄存器地址1
	str_concat_1[4] := 16#00;	//寄存器地址2
	str_concat_1[5] := 16#00;	//寄存器数量1
	str_concat_1[6] := 16#10;	//寄存器地址2
	fb_crc16_modbus(str_Message:= str_concat_1, str_Len:= 6, crc16=> );		//计算CRC校验
	str_concat_1[7] := WORD_TO_BYTE(fb_crc16_modbus.crc16 AND 16#00FF);
	str_concat_1[8] := WORD_TO_BYTE(SHR(fb_crc16_modbus.crc16,8) AND 16#00FF);
	FOR index:=1 TO 8 BY 1 DO
		str_send_1[index] := 16#00;
	END_FOR
	FOR index:=1 TO 8 BY 1 DO
		str_send_1[index] := str_concat_1[index];
	END_FOR
	di_SentBytesLen_1 := 8;
ELSIF reply_count >= 10 AND reply_count < 20 THEN
(*<<<<<<<<<<<<<<<<<<<<<<<<<<<<<concatenate STR_DAM2>>>>>>>>>>>>>>>>>>>>>>>>>>>>>>>>>>>>>>>>>>>>>>>>>>>>>>>*)
	str_concat_1[1] := 16#02;	//设备地址1
	str_concat_1[2] := 16#04;	//功能码
	str_concat_1[3] := 16#00;	//寄存器地址1
	str_concat_1[4] := 16#00;	//寄存器地址2
	str_concat_1[5] := 16#00;	//寄存器数量1
	str_concat_1[6] := 16#03;	//寄存器地址2
	fb_crc16_modbus(str_Message:= str_concat_1, str_Len:= 6, crc16=> );		//计算CRC校验
	str_concat_1[7] := WORD_TO_BYTE(fb_crc16_modbus.crc16 AND 16#00FF);
	str_concat_1[8] := WORD_TO_BYTE(SHR(fb_crc16_modbus.crc16,8) AND 16#00FF);
	FOR index:=1 TO 8 BY 1 DO
		str_send_1[index] := 16#00;
	END_FOR
	FOR index:=1 TO 8 BY 1 DO
		str_send_1[index] := str_concat_1[index];
	END_FOR
	di_SentBytesLen_1 := 8;
ELSIF reply_count >= 20 AND reply_count < 30 THEN
(*<<<<<<<<<<<<<<<<<<<<<<<<<<<<<concatenate STR_DAM2>>>>>>>>>>>>>>>>>>>>>>>>>>>>>>>>>>>>>>>>>>>>>>>>>>>>>>>*)
	str_concat_1[1] := 16#03;	//设备地址1
	str_concat_1[2] := 16#04;	//功能码
	str_concat_1[3] := 16#00;	//寄存器地址1
	str_concat_1[4] := 16#00;	//寄存器地址2
	str_concat_1[5] := 16#00;	//寄存器数量1
	str_concat_1[6] := 16#06;	//寄存器地址2
	fb_crc16_modbus(str_Message:= str_concat_1, str_Len:= 6, crc16=> );		//计算CRC校验
	str_concat_1[7] := WORD_TO_BYTE(fb_crc16_modbus.crc16 AND 16#00FF);
	str_concat_1[8] := WORD_TO_BYTE(SHR(fb_crc16_modbus.crc16,8) AND 16#00FF);
	FOR index:=1 TO 8 BY 1 DO
		str_send_1[index] := 16#00;
	END_FOR
	FOR index:=1 TO 8 BY 1 DO
		str_send_1[index] := str_concat_1[index];
	END_FOR
	di_SentBytesLen_1 := 8;
ELSE
(*<<<<<<<<<<<<<<<<<<<<<<<<<<<<<concatenate STR_DAM3>>>>>>>>>>>>>>>>>>>>>>>>>>>>>>>>>>>>>>>>>>>>>>>>>>>>>>>*)
	str_concat_1[1] := 16#03;	//设备地址1
	str_concat_1[2] := 16#04;	//功能码
	str_concat_1[3] := 16#00;	//寄存器地址1
	str_concat_1[4] := 16#27;	//寄存器地址2
	str_concat_1[5] := 16#00;	//寄存器数量1
	str_concat_1[6] := 16#0D;	//寄存器地址2
	fb_crc16_modbus(str_Message:= str_concat_1, str_Len:= 6, crc16=> );		//计算CRC校验
	str_concat_1[7] := WORD_TO_BYTE(fb_crc16_modbus.crc16 AND 16#00FF);
	str_concat_1[8] := WORD_TO_BYTE(SHR(fb_crc16_modbus.crc16,8) AND 16#00FF);
	FOR index:=1 TO 8 BY 1 DO
		str_send_1[index] := 16#00;
	END_FOR
	FOR index:=1 TO 8 BY 1 DO
		str_send_1[index] := str_concat_1[index];
	END_FOR	
	di_SentBytesLen_1 := 8;
END_IF
				
(*<<<<<<<<<<<<<<<<<<<<<<<<<<<if TCP is wrong,reset the TCP serve>>>>>>>>>>>>>>>>>>>>>>>>>>>>*)
IF UDPConnection_1.Error=TRUE OR UDPRecv_1.Error=TRUE OR UDPSend_1.Error=TRUE THEN
	b_Server_Enable_1:=FALSE;
	b_Recv_enable_1:=FALSE;
	b_Send_enable_1:=FALSE;
ELSE
	b_Server_Enable_1:=TRUE;
END_IF

IF UDPConnection_2.Error=TRUE OR UDPRecv_2.Error=TRUE OR UDPSend_2.Error=TRUE THEN
	b_Server_Enable_2:=FALSE;
	b_Recv_enable_2:=FALSE;
	b_Send_enable_2:=FALSE;
ELSE
	b_Server_Enable_2:=TRUE;
END_IF

P_UDP_with_DAM.Async_TCP();
P_UDP_with_DAM.A_RECV();
P_UDP_with_DAM.A_SEND();
(*<<<<<<<<<<<<<<<<<<<<<<<<<<<if TCP server is connected,a cycle is executed>>>>>>>>>>>>>>>>>>>>>>>>>>>>>>>>>>>>>>>>>>>>>*)
IF b_Connection_done_1=TRUE THEN
	IF  b_receiving_1=FALSE AND b_sending_1=FALSE AND b_Send_enable_1=FALSE THEN
		b_Send_enable_1:=TRUE;(*open send fuction*)
		P_UDP_with_DAM.A_SEND();
		b_sending_1:=TRUE;
	END_IF;
	
(*<<<<<<<<<<<<<<<<<<<<<<<<<<<send message>>>>>>>>>>>>>>>>>>>>>>>>>>>>>>>>>>>>>>>>>>>>>>>>>*)
	IF b_Send_done_1=TRUE AND b_sending_1=TRUE AND b_receiving_1=FALSE THEN
		b_Send_enable_1:=FALSE;
		P_UDP_with_DAM.A_SEND();
		b_sending_1:=FALSE;
		b_receiving_1:=TRUE;
		i_counter_udp1 := 0;
	END_IF;
	
(*<<<<<<<<<<<<<<<<<<<<<<<<<<<<<<<<<<<<<<<<<<<<<<<<<receive message>>>>>>>>>>>>>>>>>>>>>>>>>>>>>>>>>>>>>>>>>>>>>>>>>>>>>>>*)
	IF b_sending_1=FALSE AND b_receiving_1=TRUE THEN
		b_Recv_enable_1:=TRUE;
		P_UDP_with_DAM.A_RECV();
		i_counter_udp1 := i_counter_udp1 + 1;
	END_IF;
	
(*<<<<<<<<<<<<<<<<<<<<<<<<<<<<<<<<<<<<<<<<<<<<<<<<<not receive message>>>>>>>>>>>>>>>>>>>>>>>>>>>>>>>>>>>>>>>>>>>>>>>>>>>>>>>*)	
	IF b_sending_1=FALSE AND b_receiving_1=TRUE AND i_counter_udp1>10 THEN
		b_Recv_enable_1:=FALSE;
		b_receiving_1:=FALSE;
		i_counter_udp1 := 0;
	END_IF;
	
(*<<<<<<<<<<<<<<<<<<<<<<<<<<<recieveing message>>>>>>>>>>>>>>>>>>>>>>>>>>>>>>>>>>>>>>>>>>>>>>>>>*)
	IF b_Recv_done_1=TRUE AND b_receiving_1=TRUE THEN
		
		IF str_Recv_1[1] = 16#01 AND str_Recv_1[3] = 16#20 THEN
			
			TempEMISC_Outlet := WORD_TO_LREAL(BYTE_TO_WORD(str_Recv_1[16]) * 256 + BYTE_TO_WORD(str_Recv_1[17])) / 65535 * 165 - 40;
			HumidEMISC_Outlet := WORD_TO_LREAL(BYTE_TO_WORD(str_Recv_1[18]) * 256 + BYTE_TO_WORD(str_Recv_1[19])) / 65535 * 100;
			TempPSC_Inlet := WORD_TO_LREAL(BYTE_TO_WORD(str_Recv_1[20]) * 256 + BYTE_TO_WORD(str_Recv_1[21])) / 65535 * 165 - 40;
			HumidPSC_Inlet := WORD_TO_LREAL(BYTE_TO_WORD(str_Recv_1[22]) * 256 + BYTE_TO_WORD(str_Recv_1[23])) / 65535 * 100;
			TempPSC_Outlet := WORD_TO_LREAL(BYTE_TO_WORD(str_Recv_1[24]) * 256 + BYTE_TO_WORD(str_Recv_1[25])) / 65535 * 165 - 40;
			HumidPSC_Outlet := WORD_TO_LREAL(BYTE_TO_WORD(str_Recv_1[26]) * 256 + BYTE_TO_WORD(str_Recv_1[27])) / 65535 * 100;
			TempDriveCab := WORD_TO_LREAL(BYTE_TO_WORD(str_Recv_1[28]) * 256 + BYTE_TO_WORD(str_Recv_1[29])) / 65535 * 100 - 20;
			HumidDriveCab := WORD_TO_LREAL(BYTE_TO_WORD(str_Recv_1[30]) * 256 + BYTE_TO_WORD(str_Recv_1[31])) / 65535 * 100;
			TempDriveCab_Up := WORD_TO_LREAL(BYTE_TO_WORD(str_Recv_1[32]) * 256 + BYTE_TO_WORD(str_Recv_1[33])) / 65535 * 100 - 20;
			HumidDriveCab_Up := WORD_TO_LREAL(BYTE_TO_WORD(str_Recv_1[34]) * 256 + BYTE_TO_WORD(str_Recv_1[35])) / 65535 * 100;			 

			
		ELSIF str_Recv_1[1] = 16#02 AND str_Recv_1[3] = 16#06 THEN
			
			Pedestal_temp_1 := WORD_TO_REAL(BYTE_TO_WORD(str_Recv_1[4]) * 256 + BYTE_TO_WORD(str_Recv_1[5])) / 65535 * 200 - 50;
			Pedestal_temp_2 := WORD_TO_REAL(BYTE_TO_WORD(str_Recv_1[6]) * 256 + BYTE_TO_WORD(str_Recv_1[7])) / 65535 * 200 - 50;
			Pedestal_temp_3 := WORD_TO_REAL(BYTE_TO_WORD(str_Recv_1[8]) * 256 + BYTE_TO_WORD(str_Recv_1[9])) / 65535 * 200 - 50;
			
		ELSIF str_Recv_1[1] = 16#03 AND str_Recv_1[3] =16#0C THEN
			
			CurrentPh1 := WORD_TO_LREAL(BYTE_TO_WORD(str_Recv_1[4]) * 256 + BYTE_TO_WORD(str_Recv_1[5])) / 65535 * 100;
			CurrentPh2 := WORD_TO_LREAL(BYTE_TO_WORD(str_Recv_1[6]) * 256 + BYTE_TO_WORD(str_Recv_1[7])) / 65535 * 100;
			CurrentPh3 := WORD_TO_LREAL(BYTE_TO_WORD(str_Recv_1[8]) * 256 + BYTE_TO_WORD(str_Recv_1[9])) / 65535 * 100;
			VoltagePh1 := WORD_TO_LREAL(BYTE_TO_WORD(str_Recv_1[10]) * 256 + BYTE_TO_WORD(str_Recv_1[11])) / 65535 * 1000;
			VoltagePh2 := WORD_TO_LREAL(BYTE_TO_WORD(str_Recv_1[12]) * 256 + BYTE_TO_WORD(str_Recv_1[13])) / 65535 * 1000;
			VoltagePh3 := WORD_TO_LREAL(BYTE_TO_WORD(str_Recv_1[14]) * 256 + BYTE_TO_WORD(str_Recv_1[15])) / 65535 * 1000;
		
		ELSIF str_Recv_1[1] = 16#03 AND str_Recv_1[3] =16#1A THEN
		
			FrequencyPh1 := WORD_TO_LREAL(BYTE_TO_WORD(str_Recv_1[4]) * 256 + BYTE_TO_WORD(str_Recv_1[5])) / 65535 * 65;
			FrequencyPh2 := WORD_TO_LREAL(BYTE_TO_WORD(str_Recv_1[6]) * 256 + BYTE_TO_WORD(str_Recv_1[7])) / 65535 * 65;
			FrequencyPh3 := WORD_TO_LREAL(BYTE_TO_WORD(str_Recv_1[8]) * 256 + BYTE_TO_WORD(str_Recv_1[9])) / 65535 * 65;
			
			ActivePowerConsumption := WORD_TO_LREAL(BYTE_TO_WORD(str_Recv_1[10]) * 256 + BYTE_TO_WORD(str_Recv_1[11])) / 65535 * 600000 - 300000;
			ReactivePowerConsumption := WORD_TO_LREAL(BYTE_TO_WORD(str_Recv_1[12]) * 256 + BYTE_TO_WORD(str_Recv_1[13])) / 65535 * 600000 - 300000;
			ApparentPowerConsumption := WORD_TO_LREAL(BYTE_TO_WORD(str_Recv_1[14]) * 256 + BYTE_TO_WORD(str_Recv_1[15])) / 65535 * 600000 - 300000;

		
			PowerFactor := WORD_TO_LREAL(BYTE_TO_WORD(str_Recv_1[28]) * 256 + BYTE_TO_WORD(str_Recv_1[29])) / 65535 * 2 - 1;
	
		END_IF;

		b_Recv_enable_1:=FALSE;
		P_UDP_with_DAM.A_RECV();
		b_receiving_1:=FALSE;
		i_counter_udp1 := 0;
	END_IF;
	
	IF b_Recv_done_1=TRUE  THEN
		b_Recv_enable_1:=FALSE;
		P_UDP_with_DAM.A_RECV();
	END_IF;
(*<<<<<<<<<<<<<<<<<<<<<<<<<<<<<<<<<<<<<<<<<<<<<If not conected,then reset receive and send function>>>>>>>>>>>>>>>>>>>>>>>>>>>>>>>>>>>>>>>>>>>>>>>>>>>>>>>*)
ELSE
	b_receiving_1:=FALSE;
	b_sending_1:=FALSE;
	b_Recv_enable_1:=FALSE;
	b_send_enable_1:=FALSE;
END_IF;

(*Tilt Sensor Receiving Data*)
IF b_Connection_done_2=TRUE THEN
	IF  b_receiving_2=FALSE AND b_sending_2=FALSE AND b_Recv_enable_2=FALSE THEN
		b_Recv_enable_2:=TRUE;(*open receive fuction*)
		P_UDP_with_DAM.A_RECV();
		b_receiving_2:=TRUE;
	END_IF;
	
	IF b_Recv_done_2=TRUE AND b_receiving_2=TRUE THEN
		Pointing.Status.TiltXRaw_mV_One:= WORD_TO_LREAL(BYTE_TO_WORD(str_Recv_2[22]) * 256 + BYTE_TO_WORD(str_Recv_2[23]));
		Pointing.Status.TiltYRaw_mV_One := WORD_TO_LREAL(BYTE_TO_WORD(str_Recv_2[24]) * 256 + BYTE_TO_WORD(str_Recv_2[25]));
		Pointing.Status.TiltTemp_One := WORD_TO_LREAL(BYTE_TO_WORD(str_Recv_2[26]) * 256 + BYTE_TO_WORD(str_Recv_2[27]));
		X_Axis_Tile_Monitor := WORD_TO_LREAL(BYTE_TO_WORD(str_Recv_2[30]) * 256 + BYTE_TO_WORD(str_Recv_2[31]));
		Y_Axis_Tile_Monitor := WORD_TO_LREAL(BYTE_TO_WORD(str_Recv_2[32]) * 256 + BYTE_TO_WORD(str_Recv_2[33]));
		Temp_Tile_Monitor := WORD_TO_LREAL(BYTE_TO_WORD(str_Recv_2[34]) * 256 + BYTE_TO_WORD(str_Recv_2[35]));
	
		b_Recv_enable_2:=FALSE;
		P_UDP_with_DAM.A_RECV();
		b_receiving_2:=FALSE;
	END_IF;
ELSE
	b_receiving_2:=FALSE;
	b_sending_2:=FALSE;
	b_Recv_enable_2:=FALSE;
	b_send_enable_2:=FALSE;
END_IF;

ACTION Async_TCP:
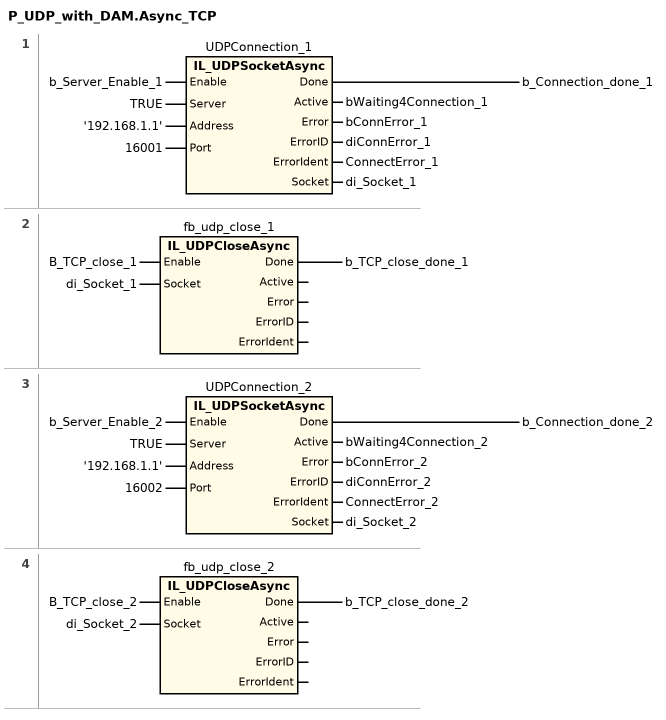
// NETWORK 1
UDPConnection_1(
    Enable := b_Server_Enable_1,
    Server := TRUE,
    Address := '192.168.1.1',
    Port := 16001,
    Active => bWaiting4Connection_1,
    Error => bConnError_1,
    ErrorID => diConnError_1,
    ErrorIdent => ConnectError_1,
    Socket => di_Socket_1); // IL_UDPSocketAsync
b_Connection_done_1 := UDPConnection_1.Done;

// NETWORK 2
fb_udp_close_1(Enable := B_TCP_close_1, Socket := di_Socket_1); // IL_UDPCloseAsync
b_TCP_close_done_1 := fb_udp_close_1.Done;

// NETWORK 3
UDPConnection_2(
    Enable := b_Server_Enable_2,
    Server := TRUE,
    Address := '192.168.1.1',
    Port := 16002,
    Active => bWaiting4Connection_2,
    Error => bConnError_2,
    ErrorID => diConnError_2,
    ErrorIdent => ConnectError_2,
    Socket => di_Socket_2); // IL_UDPSocketAsync
b_Connection_done_2 := UDPConnection_2.Done;

// NETWORK 4
fb_udp_close_2(Enable := B_TCP_close_2, Socket := di_Socket_2); // IL_UDPCloseAsync
b_TCP_close_done_2 := fb_udp_close_2.Done;
END_ACTION

ACTION A_RECV:
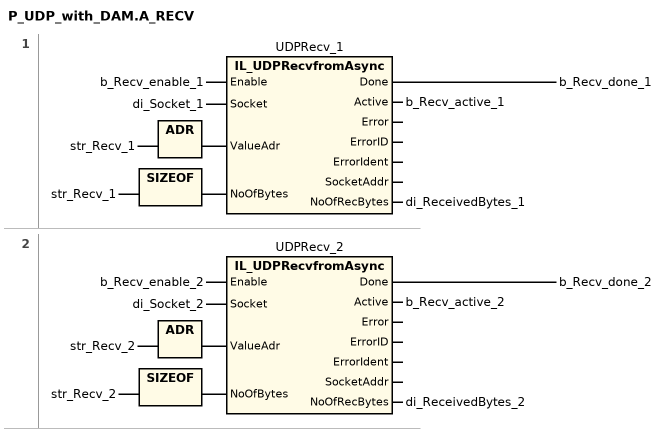
// NETWORK 1
UDPRecv_1(
    Enable := b_Recv_enable_1,
    Socket := di_Socket_1,
    ValueAdr := ADR(str_Recv_1),
    NoOfBytes := SIZEOF(str_Recv_1),
    Active => b_Recv_active_1,
    NoOfRecBytes => di_ReceivedBytes_1); // IL_UDPRecvfromAsync
b_Recv_done_1 := UDPRecv_1.Done;

// NETWORK 2
UDPRecv_2(
    Enable := b_Recv_enable_2,
    Socket := di_Socket_2,
    ValueAdr := ADR(str_Recv_2),
    NoOfBytes := SIZEOF(str_Recv_2),
    Active => b_Recv_active_2,
    NoOfRecBytes => di_ReceivedBytes_2); // IL_UDPRecvfromAsync
b_Recv_done_2 := UDPRecv_2.Done;
END_ACTION

ACTION A_SEND:
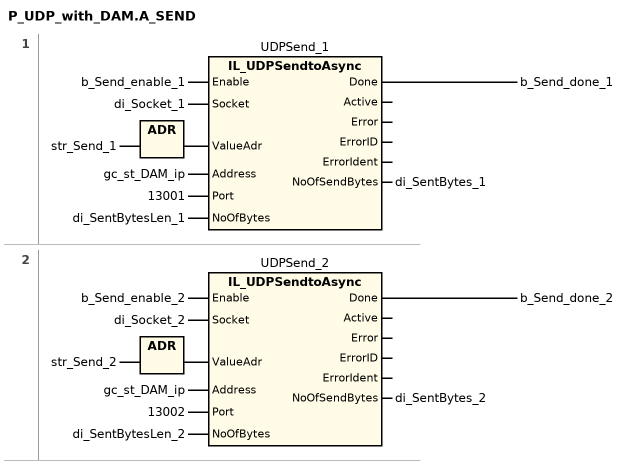
// NETWORK 1
UDPSend_1(
    Enable := b_Send_enable_1,
    Socket := di_Socket_1,
    ValueAdr := ADR(str_Send_1),
    Address := gc_st_DAM_ip,
    Port := 13001,
    NoOfBytes := di_SentBytesLen_1,
    NoOfSendBytes => di_SentBytes_1); // IL_UDPSendtoAsync
b_Send_done_1 := UDPSend_1.Done;

// NETWORK 2
UDPSend_2(
    Enable := b_Send_enable_2,
    Socket := di_Socket_2,
    ValueAdr := ADR(str_Send_2),
    Address := gc_st_DAM_ip,
    Port := 13002,
    NoOfBytes := di_SentBytesLen_2,
    NoOfSendBytes => di_SentBytes_2); // IL_UDPSendtoAsync
b_Send_done_2 := UDPSend_2.Done;
END_ACTION

END_PROGRAM

// IndraMotionMlc1/Application/POUs/TCP/Message/CRC16_MODBUS
FUNCTION_BLOCK CRC16_MODBUS
VAR_INPUT
	str_Message: ARRAY[1..40] OF BYTE;
	str_Len: BYTE;
END_VAR
VAR_OUTPUT
	crc16 : WORD;
END_VAR
VAR
	i : BYTE;
	j : BYTE;
	polynomial : WORD;
	curval : WORD;
	temp : WORD;
END_VAR


temp := 16#FFFF;
polynomial := 16#A001;
FOR i:=1 TO str_Len BY 1 DO
	curval := BYTE_TO_WORD(str_Message[i]);
	FOR j:=1 TO 8 BY 1 DO
		IF ((WORD_TO_BYTE(temp XOR curval) AND 16#01) = 16#01) THEN
			temp := (SHR(temp,1) XOR polynomial);
		ELSE
			temp := SHR(temp,1);			
		END_IF;
		curval := SHR(curval,1);
	END_FOR;
END_FOR;

crc16 := temp;

END_FUNCTION_BLOCK

// IndraMotionMlc1/Application/POUs/TCP/P_GSTAT_K2STAT
(*the program is built for GSTAT and KSTAT,according to ICD*)
PROGRAM P_GSTAT_K2STAT
VAR
(*the transitional variables for GSTAT and KSTAT*)
    STR_GSTAT: STRING(1500);
	STR_K2STAT: STRING(255);
	STR_K4STAT: STRING(255);

(*The function block BLINK generates a pulsating signal.The input consists of ENABLE of the type BOOL, as well as TIMELOW and TIMEHIGH of the type TIME.*)
	fb_blink_diagnos_1: BLINK;
	fb_blink_diagnos_2: BLINK;
	fb_blink_diagnos_3: BLINK;
	fb_blink_diagnos_4: BLINK;
	fb_blink_diagnos_5: BLINK;
	fb_blink_diagnos_6: BLINK;
	fb_blink_diagnos_MLC: BLINK;
(*With the function block "MB_ReadParameter" it is possible to read the current value of a parameter. The return value is DINT*)
	fb_read_brake_1: MB_ReadParameter;
	fb_read_brake_2: MB_ReadParameter;
	fb_read_brake_3: MB_ReadParameter;
	fb_read_brake_4: MB_ReadParameter;
	fb_read_brake_5: MB_ReadParameter;
	fb_read_brake_6: MB_ReadParameter;
(*With the function block "MB_ReadStringParameter" it is possible to read a parameter the operating data of which has the ASCII format (string).*)
	fb_diagnose_1: MB_ReadStringParameter;
	fb_diagnose_2: MB_ReadStringParameter;
	fb_diagnose_3: MB_ReadStringParameter;
	fb_diagnose_4: MB_ReadStringParameter;
	fb_diagnose_5: MB_ReadStringParameter;
	fb_diagnose_6: MB_ReadStringParameter;
	fb_diagnose_MLC: MB_ReadStringParameter;
(*With the function block "MB_ReadRealParameter" it is possible to read the current value of a parameter. The return value is REAL. *)
	FB_readcur1: MB_ReadRealParameter;
	FB_readcur2: MB_ReadRealParameter;
	FB_readcur3: MB_ReadRealParameter;
	FB_readcur4: MB_ReadRealParameter;
	FB_readcur5: MB_ReadRealParameter;
	FB_readcur6: MB_ReadRealParameter;
	fb_temp_1: MB_ReadRealParameter;
	fb_temp_2: MB_ReadRealParameter;
	fb_temp_3: MB_ReadRealParameter;
	fb_temp_4: MB_ReadRealParameter;
	fb_temp_5: MB_ReadRealParameter;
	fb_temp_6: MB_ReadRealParameter;
	fb_read_s189_1: MB_ReadRealParameter;
	fb_read_s189_3: MB_ReadRealParameter;
	fb_read_s189_5: MB_ReadRealParameter;
	FB_readtor1: MB_ReadRealParameter;
	FB_readtor2: MB_ReadRealParameter;
	FB_readtor3: MB_ReadRealParameter;
	FB_readtor4: MB_ReadRealParameter;
	FB_readtor5: MB_ReadRealParameter;
	FB_readtor6: MB_ReadRealParameter;
	FB_temp_1_a: MB_ReadRealParameter;
	FB_temp_2_a: MB_ReadRealParameter;
	FB_temp_3_a: MB_ReadRealParameter;
	FB_temp_4_a: MB_ReadRealParameter;
	FB_temp_5_a: MB_ReadRealParameter;
	FB_temp_6_a: MB_ReadRealParameter;
(*FP_P_0_0539,Holding brake status word *)
	dw_brake_1: DWORD;
	dw_brake_2: DWORD;
	dw_brake_3: DWORD;
	dw_brake_4: DWORD;
	dw_brake_5: DWORD;
	dw_brake_6: DWORD;
(*FP_P_0_0007,Display text of diagnostic message*)
	str_diagnose_MLC: STRING;
	str_diagnose_1: STRING;
	str_diagnose_2: STRING;
	str_diagnose_3: STRING;
	str_diagnose_4: STRING;
	str_diagnose_5: STRING;
	str_diagnose_6: STRING;

(*FP_S_0_0384,Amplifier temperature*)
	r_temp_amp1: REAL;
	r_temp_amp2: REAL;
	r_temp_amp3: REAL;
	r_temp_amp4: REAL;
	r_temp_amp5: REAL;
	r_temp_amp6: REAL;


(*<<<<<<<<<<<<<<<<<<<<<<<<<<<<<<<<<<<<<<<add MLC temperature and operation hour(20100708)>>>>>>>>>>>>>>>>>>>>>>>>>>>>>>>>>>>>>*)
	fb_temp_MLC: MB_ReadRealParameter;
	r_temp_MLC: REAL;(*FP_c_0_0070,Control unit temperature*)
	fb_read_system_status: MB_ReadParameter;
	dw_system_status: DWORD;(*FP_C_0_0023,MC system status,used for temperature warning*)
	fb_read_operation_hour: MB_ReadParameter;

(*the limit for judging whether azimuth following error is too big*)
	r_limit_track_az: REAL;
(*test for limit check*)
	fb_software_limit_1: MB_ReadParameter;
	fb_software_limit_5: MB_ReadParameter;
	fb_software_limit_3: MB_ReadParameter;
	fb_hardware_limit_1: MB_ReadParameter;
	fb_hardware_limit_3: MB_ReadParameter;
	fb_hardware_limit_5: MB_ReadParameter;
	fb_ESTOP_1: MB_ReadParameter;
	fb_ESTOP_3: MB_ReadParameter;
	fb_ESTOP_5: MB_ReadParameter;
	i_software_limit_1: DINT;
	i_software_limit_3: DINT;
	i_software_limit_5: DINT;
	i_hardware_limit_1: DINT;
	i_hardware_limit_3: DINT;
	i_hardware_limit_5: DINT;
	i_ESTOP_1: DINT;
	i_ESTOP_3: DINT;
	i_ESTOP_5: DINT;


	b_azimuth_limit: BOOL;
	b_elevation_limit: BOOL;
	b_FeedIndexer_limit: BOOL;
	fb_readpar_speed_1: MB_ReadRealParameter;
	fb_readpar_speed_3: MB_ReadRealParameter;
	fb_readpar_speed_5: MB_ReadRealParameter;
	
	str_concat: ARRAY[1..40] OF STRING(1500);(*数组及其类型的定义*)	
	Counter: INT;
	FB_readmotorencoder1: MB_ReadRealParameter;
	FB_readmotorencoder2: MB_ReadRealParameter;
	FB_readmotorencoder3: MB_ReadRealParameter;
	FB_readmotorencoder4: MB_ReadRealParameter;
	FB_readmotorencoder5: MB_ReadRealParameter;
	FB_readmotorencoder6: MB_ReadRealParameter;
	r_motorencoder_6: REAL;
	r_motorencoder_5: REAL;
	r_motorencoder_4: REAL;
	r_motorencoder_3: REAL;
	r_motorencoder_2: REAL;
	r_motorencoder_1: REAL;
	
	(*the status word for GSTAT*)
	
	status_1:DWORD;
	status_2:DWORD;
	status_3:DWORD;
	status_4:DWORD;
	status_5:DWORD;
	status_6:DWORD;
	fb_diagnose_111: MB_ReadParameter;
	str_diagnose_11: DWORD;
	fb_blink_diagnos_11: BLINK;
	fb_diagnose_11: MB_ReadrealParameter;
	str_diagnose_111: REAL;
	fb_readpar_speed_2: MB_ReadRealParameter;
	fb_readpar_speed_4: MB_ReadRealParameter;
	fb_readpar_speed_6: MB_ReadRealParameter;
	
	ReadAxisPshape: ARRAY[1..5] OF MB_ReadlrealParameter;
	ReadAxisVact: ARRAY[1..5] OF MB_ReadlrealParameter;
	ReadAxisVshape: ARRAY[1..5] OF MB_ReadlrealParameter;

	conut_i: INT;
	b_PID_in_FI: BOOL;
	b_limit_cw_FI: BOOL;
	b_limit_ccw_FI: BOOL;
	b_limit_final_FI: BOOL;
	fb_readpar_pos_cmd_1: MB_ReadRealParameter;
END_VAR

P_GSTAT_K2STAT.A_Read_Parameter();

status_code1:=LEFT(str_diagnose_1,5);
status_code2:=LEFT(str_diagnose_2,5);
status_code3:=LEFT(str_diagnose_3,5);
status_code4:=LEFT(str_diagnose_4,5);
status_code5:=LEFT(str_diagnose_5,5);
status_code6:=LEFT(str_diagnose_6,5);

FOR  conut_i:=1 TO 5 BY 1 DO
ReadAxisPshape[conut_i](
	Enable:=axisdata[1].Axis_Inbb , 
	Done=> , 
	Active=> , 
	Error=> , 
	ErrorID=> , 
	ErrorIdent=> , 
	ParameterNumber:=FP_P_0_0434 , 
	Value=>P_shape_value[conut_i] , 
	Axis:=AxRef[conut_i] );
	
ReadAxisVshape[conut_i](
	Enable:=axisdata[1].Axis_Inbb , 
	Done=> , 
	Active=> , 
	Error=> , 
	ErrorID=> , 
	ErrorIdent=> , 
	ParameterNumber:=FP_P_0_0434 , 
	Value=>V_shape_value[conut_i] , 
	Axis:=AxRef[conut_i] );
	
ReadAxisVact[conut_i](
	Enable:=axisdata[1].Axis_Inbb , 
	Done=> , 
	Active=> , 
	Error=> , 
	ErrorID=> , 
	ErrorIdent=> , 
	ParameterNumber:=FP_S_0_0040 , 
	Value=>V_act_value[conut_i] , 
	Axis:=AxRef[conut_i] );
END_FOR

(*<<<<<<<<<<<<<<<<<<<<<<<<<<<<<master_status>>>>>>>>>>>>>>>>>>>>>>>>>>>>>>>>>>>>>>>>>>>>>>>>>>>>>>>*)
master_status.0:=axisdata[1].Axis_InAb;
IF b_remote_on=TRUE THEN
	master_status.1:=0;
ELSE
	master_status.1:=1;
END_IF
IF b_DSdoor_Estop  THEN
	master_status.2:=1;
ELSE
	master_status.2:=0;
END_IF

IF ABS(axisdata[3].rActualPosition_i-90)<0.02 THEN
	master_status.3:=1;
ELSE
	master_status.3:=0;
END_IF
	master_status.4:=(axisdata[1].Axis_Error OR axisdata[2].Axis_Error OR axisdata[3].Axis_Error OR axisdata[4].Axis_Error OR axisdata[5].Axis_Error OR axisdata[6].Axis_Error);
	master_status.5:=b_stow_pin_limit_unlock;
	master_status.6:=b_stow_pin_limit_lock;
	
IF i_num_stack_left>9500 THEN
		master_status.7:=0;
	ELSE IF i_num_stack_left<1500 THEN
		master_status.7:=1;	
	END_IF
		
END_IF

IF b_remote_on_run AND b_track_on THEN
	master_status.9:=0;
	master_status.8:=1;
ELSIF b_remote_on_run AND b_Track_Pause = TRUE THEN
	master_status.9:=1;
	master_status.8:=0;
ELSIF b_remote_on_run AND b_Track_Pause = FALSE  AND b_track_on = FALSE THEN
	master_status.9:=0;
	master_status.8:=0;
ELSE
 	master_status.9:=1;
	master_status.8:=1;
END_IF

IF 	b_encoder_ok_az	AND b_encoder_ok_FI THEN
	master_status.10:=1;
	master_status.11:=1;
ELSIF b_encoder_ok_az =FALSE AND b_encoder_ok_FI THEN
	master_status.10:=0;
	master_status.11:=1;
ELSIF b_encoder_ok_az  AND b_encoder_ok_FI=FALSE THEN
	master_status.10:=1;
	master_status.11:=0;
ELSE
	master_status.10:=0;
	master_status.11:=0;		
END_IF

IF b_remote_on_run THEN
	master_status.12:=1;
ELSE
	master_status.12:=0;
END_IF
	
IF b_remote_on_run THEN
	master_status.12:=1;
ELSE
	master_status.12:=0;
END_IF

IF b_permit_new_file THEN
	master_status.13:=1;
ELSE
	master_status.13:=0;
END_IF

(*<<<<<<<<<<<<<<<<<<<<<<<<<<<<<status_1>>>>>>>>>>>>>>>>>>>>>>>>>>>>>>>>>>>>>>>>>>>>>>>>>>>>>>>*)
status_1.0:=axisdata[1].Axis_InAb;
status_1.1:=b_PID_in_az;
status_1.2:=dw_brake_1.0;
status_1.3:=b_limit_cw_az;
status_1.4:=b_limit_ccw_az;
status_1.5:=(b_limit_final_cw_az OR b_limit_final_ccw_az);
status_1.6:=axisdata[1].Axis_Error;

(*<<<<<<<<<<<<<<<<<<<<<<<<<<<<<status_2>>>>>>>>>>>>>>>>>>>>>>>>>>>>>>>>>>>>>>>>>>>>>>>>>>>>>>>*)
status_2.0:=axisdata[2].Axis_InAb;
status_2.1:=b_PID_in_az;
status_2.2:=dw_brake_2.0;
status_2.3:=b_limit_cw_az;
status_2.4:=b_limit_ccw_az;
status_2.5:=(b_limit_final_cw_az OR b_limit_final_ccw_az);
status_2.6:=axisdata[2].Axis_Error;

(*<<<<<<<<<<<<<<<<<<<<<<<<<<<<<status_3>>>>>>>>>>>>>>>>>>>>>>>>>>>>>>>>>>>>>>>>>>>>>>>>>>>>>>>*)
status_3.0:=axisdata[3].Axis_InAb;
status_3.1:=b_PID_in_el;
status_3.2:=dw_brake_3.0;
status_3.3:=b_limit_cw_el;
status_3.4:=b_limit_ccw_el;
status_3.5:=(b_limit_final_cw_el OR b_limit_final_ccw_el) ;
status_3.6:=axisdata[3].Axis_Error;

(*<<<<<<<<<<<<<<<<<<<<<<<<<<<<<status_4>>>>>>>>>>>>>>>>>>>>>>>>>>>>>>>>>>>>>>>>>>>>>>>>>>>>>>>*)
status_4.0:=axisdata[4].Axis_InAb;
status_4.1:=b_PID_in_el;
status_4.2:=dw_brake_4.0;
status_4.3:=b_limit_cw_el;
status_4.4:=b_limit_ccw_el;
status_4.5:=(b_limit_final_cw_el OR b_limit_final_ccw_el); 
status_4.6:=axisdata[4].Axis_Error;

(*<<<<<<<<<<<<<<<<<<<<<<<<<<<<<status_5>>>>>>>>>>>>>>>>>>>>>>>>>>>>>>>>>>>>>>>>>>>>>>>>>>>>>>>*)
status_5.0:=axisdata[5].Axis_InAb;
status_5.1:=b_PID_in_FI;
status_5.2:=dw_brake_5.0;
status_5.3:=b_limit_cw_FI;
status_5.4:=b_limit_ccw_FI;
status_5.5:=b_limit_final_FI;
status_5.6:=axisdata[5].Axis_Error;

(*<<<<<<<<<<<<<<<<<<<<<<<<<<<<<status_6>>>>>>>>>>>>>>>>>>>>>>>>>>>>>>>>>>>>>>>>>>>>>>>>>>>>>>>*)
status_6.0:=axisdata[6].Axis_InAb;
status_6.1:=b_PID_in_FI;
status_6.2:=dw_brake_6.0;
status_6.3:=b_limit_cw_FI;
status_6.4:=b_limit_ccw_FI;
status_6.5:=b_limit_final_FI;
status_6.6:=axisdata[6].Axis_Error;


(*
(*<<<<<<<<<<<<<<<<<<<<<<<<<<<<<status_2>>>>>>>>>>>>>>>>>>>>>>>>>>>>>>>>>>>>>>>>>>>>>>>>>>>>>>>*)
status_2.0:=NOT(axisdata[2].Axis_InAb);
status_2.1:=axisdata[2].Axis_Error;
status_2.2:=NOT(dw_brake_2.0);
IF r_temp_motor2>120 THEN
status_2.3:=1;
b_power_Az:=FALSE;
b_enable_az_1:=FALSE;
b_enable_az_2:=FALSE;
ELSE
status_2.3:=0;
END_IF
IF r_current_2>5 THEN
status_2.4:=1;
ELSE
status_2.4:=0;
END_IF
(*<<<<<<<<<<<<<<<<<<<<<<<<<<<<<status_3>>>>>>>>>>>>>>>>>>>>>>>>>>>>>>>>>>>>>>>>>>>>>>>>>>>>>>>*)
status_3.0:=NOT(axisdata[3].Axis_InAb);
status_3.1:=axisdata[3].Axis_Error;
status_3.2:=NOT(dw_brake_3.0);
IF r_temp_motor3>120 THEN
status_3.3:=1;
b_power_El:=FALSE;
b_enable_el_3:=FALSE;
b_enable_el_4:=FALSE;
ELSE
status_3.3:=0;
END_IF
IF r_current_3>5 THEN
status_3.4:=1;
ELSE
status_3.4:=0;
END_IF
status_3.8:=NOT(b_PID_in_el);

IF (b_scc_goto=TRUE AND (b_goto_Az_done=FALSE OR b_goto_El_done=FALSE OR b_goto_FI_done=FALSE)) OR (b_track_on=TRUE AND i_num_stack_left<>0) THEN
status_3.9:=1;
END_IF;
IF (b_goto_Az_done=TRUE AND b_goto_El_done=TRUE AND b_goto_FI_done=TRUE) OR i_num_stack_left=0 THEN
status_3.9:=0;
END_IF;

status_3.10:=NOT(b_track_on);
IF ABS(r_track_error[2])<0.0034 THEN
	status_3.11:=0;
ELSE
	status_3.11:=1;
END_IF
status_3.12:=axisdata[3].Axis_Error;
IF ABS(r_following_3)>0.5 THEN
status_3.13:=1;
ELSE
status_3.13:=0;
END_IF
IF r_pos_el<14.6 THEN
	status_3.14:=1;
ELSE
	status_3.14:=0;
END_IF
IF r_pos_el>90.15 THEN
	status_3.15:=1;
ELSE
	status_3.15:=0;
END_IF
status_3.16:=b_limit_ccw_el;
status_3.17:=b_limit_cw_el;
status_3.18:=b_limit_final_el;
status_3.19:=b_track_overspeed_el;
(*<<<<<<<<<<<<<<<<<<<<<<<<<<<<<status_4>>>>>>>>>>>>>>>>>>>>>>>>>>>>>>>>>>>>>>>>>>>>>>>>>>>>>>>*)
status_4.0:=NOT(axisdata[4].Axis_InAb);
status_4.1:=axisdata[4].Axis_Error;
status_4.2:=NOT(dw_brake_4.0);
IF r_temp_motor4>120 THEN
status_4.3:=1;
b_power_El:=FALSE;
b_enable_el_3:=FALSE;
b_enable_el_4:=FALSE;
ELSE
status_4.3:=0;
END_IF
IF r_current_4>5 THEN
status_4.4:=1;
ELSE
status_4.4:=0;
END_IF
(*<<<<<<<<<<<<<<<<<<<<<<<<<<<<<status_5>>>>>>>>>>>>>>>>>>>>>>>>>>>>>>>>>>>>>>>>>>>>>>>>>>>>>>>*)
status_5.0:=NOT(axisdata[5].Axis_InAb);
status_5.1:=axisdata[5].Axis_Error;
status_5.2:=NOT(dw_brake_5.0);
IF r_temp_motor5>120 THEN
status_5.3:=1;
b_power_FI:=FALSE;
b_enable_FI_5:=FALSE;
ELSE
status_5.3:=0;
END_IF
IF r_current_5>5 THEN
status_5.4:=1;
ELSE
status_5.4:=0;
END_IF

status_5.8:=NOT(b_gearinpos_5_done);

IF (b_scc_goto=TRUE AND (b_goto_Az_done=FALSE OR b_goto_El_done=FALSE OR b_goto_FI_done=FALSE)) OR (b_track_on=TRUE AND i_num_stack_left<>0) THEN
status_5.9:=1;
END_IF;
IF (b_goto_Az_done=TRUE AND b_goto_El_done=TRUE AND b_goto_FI_done=TRUE) OR i_num_stack_left=0 THEN
status_5.9:=0;
END_IF;

status_5.10:=NOT(b_track_on);
IF ABS(r_track_error[3])<0.0034 THEN
	status_5.11:=0;
ELSE
	status_5.11:=1;
END_IF
status_5.12:=axisdata[5].Axis_Error;
IF ABS(r_following_5)>0.5 THEN
status_5.13:=1;
ELSE
status_5.13:=0;
END_IF

IF r_pos_FI<-89 THEN
	status_5.14:=1;
ELSE
	status_5.14:=0;
END_IF

IF r_pos_FI>89 THEN
	status_5.15:=1;
ELSE
	status_5.15:=0;
END_IF
status_5.16:=b_limit_ccw_FI;
status_5.17:=b_limit_cw_FI;
status_5.18:=b_limit_final_FI;
status_5.19:=b_track_overspeed_FI;
*)

(*<<<<<<<<<<<<<<<<<<<<<<<<<<<<<concatenate STR_GSTAT>>>>>>>>>>>>>>>>>>>>>>>>>>>>>>>>>>>>>>>>>>>>>>>>>>>>>>>*)
str_concat[1]:=CONCAT(' ',DWORD_TO_STRING(status_1));
str_concat[2]:=CONCAT(' ',LREAL_TO_STRING(F_reduce_to_1_bit(LREAL_TO_STRING(r_current_1))));
str_concat[3]:=CONCAT(' ',LREAL_TO_STRING(r_temp_motor1));
str_concat[4]:=CONCAT(' ',LREAL_TO_STRING(i_speed_1));
str_concat[5]:=CONCAT(' ',LREAL_TO_STRING(F_reduce_to_1_bit(LREAL_TO_STRING(r_motorencoder_1))));


str_concat[6]:=CONCAT(' ',DWORD_TO_STRING(status_2));
str_concat[7]:=CONCAT(' ',LREAL_TO_STRING(F_reduce_to_1_bit(LREAL_TO_STRING(r_current_2))));
str_concat[8]:=CONCAT(' ',LREAL_TO_STRING(r_temp_motor2));
str_concat[9]:=CONCAT(' ',LREAL_TO_STRING(i_speed_2));
str_concat[10]:=CONCAT(' ',LREAL_TO_STRING(F_reduce_to_1_bit(LREAL_TO_STRING(r_motorencoder_2))));

str_concat[11]:=CONCAT(' ',DWORD_TO_STRING(status_3));
str_concat[12]:=CONCAT(' ',LREAL_TO_STRING(F_reduce_to_1_bit(LREAL_TO_STRING(r_current_3))));
str_concat[13]:=CONCAT(' ',LREAL_TO_STRING(r_temp_motor3));
str_concat[14]:=CONCAT(' ',LREAL_TO_STRING(i_speed_3));
str_concat[15]:=CONCAT(' ',LREAL_TO_STRING(F_reduce_to_1_bit(LREAL_TO_STRING(r_motorencoder_3))));

str_concat[16]:=CONCAT(' ',DWORD_TO_STRING(status_4));
str_concat[17]:=CONCAT(' ',LREAL_TO_STRING(F_reduce_to_1_bit(LREAL_TO_STRING(r_current_4))));
str_concat[18]:=CONCAT(' ',LREAL_TO_STRING(r_temp_motor4));
str_concat[19]:=CONCAT(' ',LREAL_TO_STRING(i_speed_4));
str_concat[20]:=CONCAT(' ',LREAL_TO_STRING(F_reduce_to_1_bit(LREAL_TO_STRING(r_motorencoder_4))));

str_concat[21]:=CONCAT(' ',DWORD_TO_STRING(status_5));
str_concat[22]:=CONCAT(' ',LREAL_TO_STRING(F_reduce_to_1_bit(LREAL_TO_STRING(r_current_5))));
str_concat[23]:=CONCAT(' ',LREAL_TO_STRING(r_temp_motor5));
str_concat[24]:=CONCAT(' ',LREAL_TO_STRING(i_speed_5));
str_concat[25]:=CONCAT(' ',LREAL_TO_STRING(F_reduce_to_1_bit(LREAL_TO_STRING(r_motorencoder_5))));

str_concat[26]:=CONCAT(' ',DWORD_TO_STRING(status_6));
str_concat[27]:=CONCAT(' ',LREAL_TO_STRING(F_reduce_to_1_bit(LREAL_TO_STRING(r_current_6))));
str_concat[28]:=CONCAT(' ',LREAL_TO_STRING(r_temp_motor6));
str_concat[29]:=CONCAT(' ',LREAL_TO_STRING(i_speed_6));
str_concat[30]:=CONCAT(' ',LREAL_TO_STRING(F_reduce_to_1_bit(LREAL_TO_STRING(r_motorencoder_6))));

str_concat[31]:=CONCAT(' ',last_command);
str_concat[32]:=CONCAT(' ',INT_TO_STRING(i_receive_cmd));
str_concat[33]:=CONCAT(' ',INT_TO_STRING(i_excute_cmd));
(*
str_concat[31]:=CONCAT(' ',REAL_TO_STRING(F_reduce_to_4_bit(REAL_TO_STRING(r_test1))));
str_concat[32]:=CONCAT(' ',REAL_TO_STRING(F_reduce_to_4_bit(REAL_TO_STRING(r_test2))));
str_concat[33]:=CONCAT(' ',REAL_TO_STRING(F_reduce_to_4_bit(REAL_TO_STRING(r_test3))));
*)
STR_GSTAT_M:='';(*for语句格式*)
				FOR Counter:=1 TO 33 BY 1 DO
					STR_GSTAT_M:=CONCAT(STR_GSTAT_M,str_concat[Counter]);
				END_FOR;



(*
STR_GSTAT:=CONCAT(STR_GSTAT,CONCAT(' ',DWORD_TO_STRING(status_1)));
STR_GSTAT:=CONCAT(STR_GSTAT,CONCAT(' ',REAL_TO_STRING(r_current_1)));
STR_GSTAT:=CONCAT(STR_GSTAT,CONCAT(' ',REAL_TO_STRING(r_temp_motor1)));
STR_GSTAT:=CONCAT(STR_GSTAT,CONCAT(' ',REAL_TO_STRING(i_speed_1)));
*)


(*
STR_GSTAT:=CONCAT(STR_GSTAT,CONCAT(' ',DWORD_TO_STRING(status_2)));
STR_GSTAT:=CONCAT(STR_GSTAT,CONCAT(' ',REAL_TO_STRING(r_current_2)));
STR_GSTAT:=CONCAT(STR_GSTAT,CONCAT(' ',REAL_TO_STRING(r_temp_motor2)));
STR_GSTAT:=CONCAT(STR_GSTAT,CONCAT(' ',REAL_TO_STRING(i_speed_1)));

STR_GSTAT:=CONCAT(STR_GSTAT,CONCAT(' ',DWORD_TO_STRING(status_3)));
STR_GSTAT:=CONCAT(STR_GSTAT,CONCAT(' ',REAL_TO_STRING(r_current_3)));
STR_GSTAT:=CONCAT(STR_GSTAT,CONCAT(' ',REAL_TO_STRING(r_temp_motor3)));
STR_GSTAT:=CONCAT(STR_GSTAT,CONCAT(' ',REAL_TO_STRING(i_speed_3)));

STR_GSTAT:=CONCAT(STR_GSTAT,CONCAT(' ',DWORD_TO_STRING(status_4)));
STR_GSTAT:=CONCAT(STR_GSTAT,CONCAT(' ',REAL_TO_STRING(r_current_4)));
STR_GSTAT:=CONCAT(STR_GSTAT,CONCAT(' ',REAL_TO_STRING(r_temp_motor4)));
STR_GSTAT:=CONCAT(STR_GSTAT,CONCAT(' ',REAL_TO_STRING(i_speed_3)));

STR_GSTAT:=CONCAT(STR_GSTAT,CONCAT(' ',DWORD_TO_STRING(status_5)));
STR_GSTAT:=CONCAT(STR_GSTAT,CONCAT(' ',REAL_TO_STRING(r_current_5)));
STR_GSTAT:=CONCAT(STR_GSTAT,CONCAT(' ',REAL_TO_STRING(r_temp_motor5)));
STR_GSTAT:=CONCAT(STR_GSTAT,CONCAT(' ',REAL_TO_STRING(i_speed_5)));

STR_GSTAT:=CONCAT(STR_GSTAT,CONCAT(' ',DWORD_TO_STRING(status_6)));
STR_GSTAT:=CONCAT(STR_GSTAT,CONCAT(' ',REAL_TO_STRING(r_current_6)));
STR_GSTAT:=CONCAT(STR_GSTAT,CONCAT(' ',REAL_TO_STRING(r_temp_motor6)));
STR_GSTAT:=CONCAT(STR_GSTAT,CONCAT(' ',REAL_TO_STRING(i_speed_5)));

STR_GSTAT:=CONCAT(STR_GSTAT,CONCAT(' ',INT_TO_STRING(i_num_stack_left)));
STR_GSTAT:=CONCAT(STR_GSTAT,CONCAT(' ',INT_TO_STRING(i_start)));
STR_GSTAT_M:=CONCAT(STR_GSTAT,CONCAT(' ',INT_TO_STRING(i_end)));

*)
(*<<<<<<<<<<<<<<<<<<<<<<<<<<<<<concatenate STR_K2STAT>>>>>>>>>>>>>>>>>>>>>>>>>>>>>>>>>>>>>>>>>>>>>>>>>>>>>>>*)
STR_K2STAT:=CONCAT('OK - ',REAL_TO_STRING(r_operation_hour/100));
STR_K2STAT:=CONCAT(STR_K2STAT,CONCAT(' ',LREAL_TO_STRING(r_temp_motor1)));
STR_K2STAT:=CONCAT(STR_K2STAT,CONCAT(' ',LREAL_TO_STRING(r_temp_motor2)));
STR_K2STAT:=CONCAT(STR_K2STAT,CONCAT(' ',LREAL_TO_STRING(r_temp_motor3)));
STR_K2STAT:=CONCAT(STR_K2STAT,CONCAT(' ',LREAL_TO_STRING(r_temp_motor4)));
STR_K2STAT:=CONCAT(STR_K2STAT,CONCAT(' ',LREAL_TO_STRING(r_temp_motor5)));
STR_K2STAT:=CONCAT(STR_K2STAT,CONCAT(' ',LREAL_TO_STRING(r_temp_amp1)));
STR_K2STAT:=CONCAT(STR_K2STAT,CONCAT(' ',LREAL_TO_STRING(r_temp_amp2)));
STR_K2STAT:=CONCAT(STR_K2STAT,CONCAT(' ',LREAL_TO_STRING(r_temp_amp3)));
STR_K2STAT:=CONCAT(STR_K2STAT,CONCAT(' ',LREAL_TO_STRING(r_temp_amp4)));
STR_K2STAT:=CONCAT(STR_K2STAT,CONCAT(' ',LREAL_TO_STRING(r_temp_amp5)));
STR_K2STAT_M:=CONCAT(STR_K2STAT,CONCAT(' ',LREAL_TO_STRING(r_temp_MLC)));
(*<<<<<<<<<<<<<<<<<<<<<<<<<<<<<concatenate STR_K4STAT>>>>>>>>>>>>>>>>>>>>>>>>>>>>>>>>>>>>>>>>>>>>>>>>>>>>>>>*)
STR_K4STAT:=CONCAT('OK - ',str_diagnose_MLC);
STR_K4STAT:=CONCAT(STR_K4STAT,CONCAT(' ',str_diagnose_1));
STR_K4STAT:=CONCAT(STR_K4STAT,CONCAT(' ',str_diagnose_2));
STR_K4STAT:=CONCAT(STR_K4STAT,CONCAT(' ',str_diagnose_3));
STR_K4STAT:=CONCAT(STR_K4STAT,CONCAT(' ',str_diagnose_4));
STR_K4STAT_M:=CONCAT(STR_K4STAT,CONCAT(' ',str_diagnose_5));

(*<<<<<<<<<<<<<<<<<<<<<<<<<<<<<concatenate STR_K5STAT>>>>>>>>>>>>>>>>>>>>>>>>>>>>>>>>>>>>>>>>>>>>>>>>>>>>>>>*)
IF i_software_limit_1=16 AND i_hardware_limit_1=3 AND i_ESTOP_1=5 THEN
	b_azimuth_limit:=TRUE;
ELSE
	b_azimuth_limit:=FALSE;
END_IF

IF i_software_limit_3=16 AND i_hardware_limit_3=3 AND i_ESTOP_3=5 THEN
	b_elevation_limit:=TRUE;
ELSE
	b_elevation_limit:=FALSE;
END_IF

IF i_software_limit_5=16 AND i_hardware_limit_5=3 AND i_ESTOP_5=5 THEN
	b_FeedIndexer_limit:=TRUE;
ELSE
	b_FeedIndexer_limit:=FALSE;
END_IF
IF b_azimuth_limit AND b_elevation_limit AND b_FeedIndexer_limit THEN
	STR_K5STAT_M:='All the axes are safe.';
ELSE
	STR_K5STAT_M:='';
	IF b_azimuth_limit=FALSE THEN
		STR_K5STAT_M:=CONCAT(STR_K5STAT_M,'Azimuth axis is unsafe. ');
	END_IF
	IF b_elevation_limit=FALSE THEN
		STR_K5STAT_M:=CONCAT(STR_K5STAT_M,'Elevation axis is unsafe. ');
	END_IF
	IF b_FeedIndexer_limit=FALSE THEN
		STR_K5STAT_M:=CONCAT(STR_K5STAT_M,'FeedIndexer axis is unsafe. ');
	END_IF
END_IF

ACTION A_Read_Parameter:
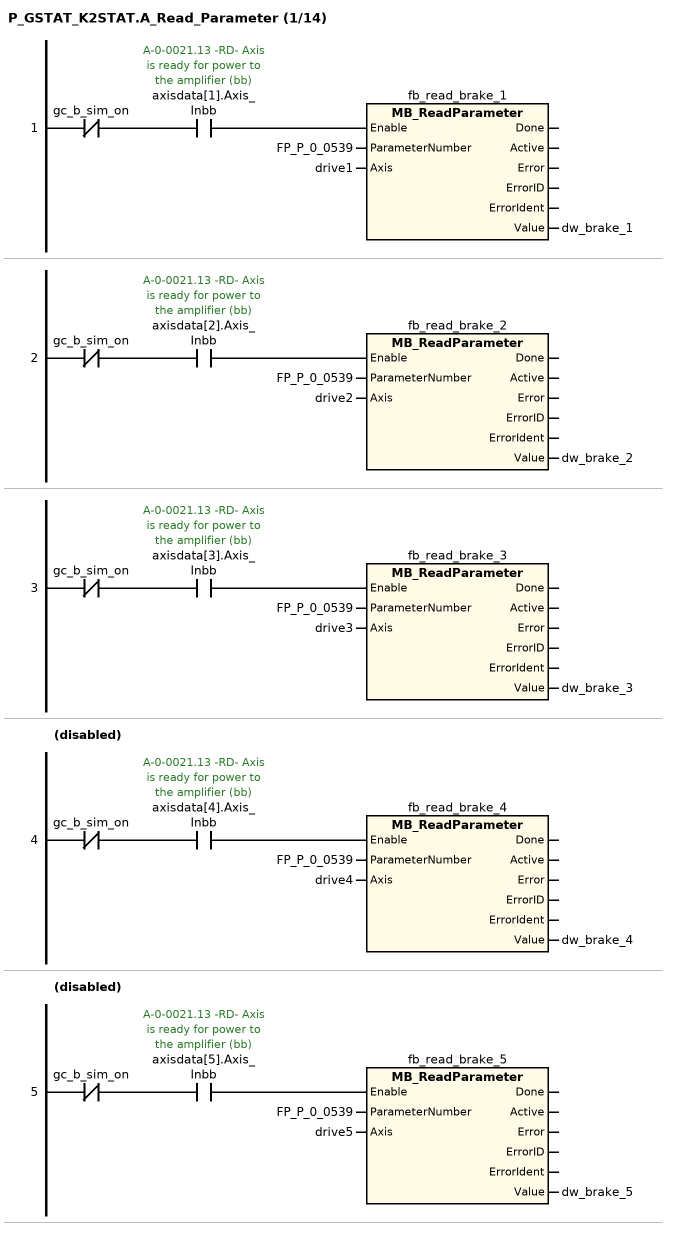
// NETWORK 1
//   fb_read_brake_1: With the function block "MB_ReadParameter" it is possible to read the current value of a parameter. The return value is DINT
//   axisdata[1].Axis_Inbb: A-0-0021.13 -RD- Axis is ready for power to the amplifier (bb)
//   FP_P_0_0539: Holding brake status word
//   drive1: Real axis "Drive1" with axis number 1
//   dw_brake_1: FP_P_0_0539,Holding brake status word
fb_read_brake_1(
    Enable := NOT gc_b_sim_on AND axisdata[1].Axis_Inbb,
    ParameterNumber := FP_P_0_0539,
    Axis := drive1,
    Value => dw_brake_1); // MB_ReadParameter

// NETWORK 2
//   axisdata[2].Axis_Inbb: A-0-0021.13 -RD- Axis is ready for power to the amplifier (bb)
//   FP_P_0_0539: Holding brake status word
//   drive2: Real axis "Drive2" with axis number 2
fb_read_brake_2(
    Enable := NOT gc_b_sim_on AND axisdata[2].Axis_Inbb,
    ParameterNumber := FP_P_0_0539,
    Axis := drive2,
    Value => dw_brake_2); // MB_ReadParameter

// NETWORK 3
//   axisdata[3].Axis_Inbb: A-0-0021.13 -RD- Axis is ready for power to the amplifier (bb)
//   FP_P_0_0539: Holding brake status word
//   drive3: Real axis "Drive3" with axis number 3
fb_read_brake_3(
    Enable := NOT gc_b_sim_on AND axisdata[3].Axis_Inbb,
    ParameterNumber := FP_P_0_0539,
    Axis := drive3,
    Value => dw_brake_3); // MB_ReadParameter

// NETWORK 4 (disabled)
//   axisdata[4].Axis_Inbb: A-0-0021.13 -RD- Axis is ready for power to the amplifier (bb)
//   FP_P_0_0539: Holding brake status word
//   drive4: Real axis "Drive4" with axis number 4
// fb_read_brake_4(
//     Enable := NOT gc_b_sim_on AND axisdata[4].Axis_Inbb,
//     ParameterNumber := FP_P_0_0539,
//     Axis := drive4,
//     Value => dw_brake_4); // MB_ReadParameter

// NETWORK 5 (disabled)
//   axisdata[5].Axis_Inbb: A-0-0021.13 -RD- Axis is ready for power to the amplifier (bb)
//   FP_P_0_0539: Holding brake status word
//   drive5: Real axis "Drive5" with axis number 5
// fb_read_brake_5(
//     Enable := NOT gc_b_sim_on AND axisdata[5].Axis_Inbb,
//     ParameterNumber := FP_P_0_0539,
//     Axis := drive5,
//     Value => dw_brake_5); // MB_ReadParameter

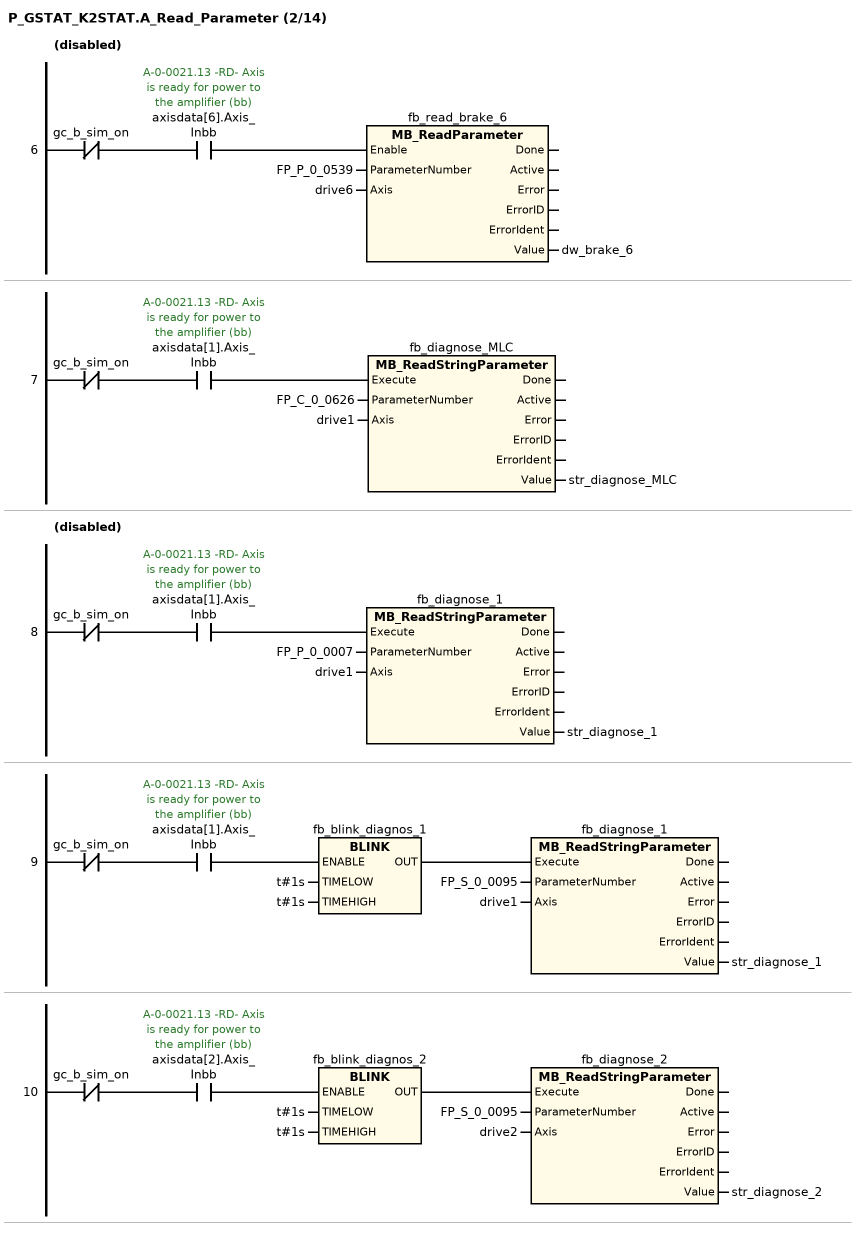
// NETWORK 6 (disabled)
//   axisdata[6].Axis_Inbb: A-0-0021.13 -RD- Axis is ready for power to the amplifier (bb)
//   FP_P_0_0539: Holding brake status word
//   drive6: Real axis "Drive6" with axis number 6
// fb_read_brake_6(
//     Enable := NOT gc_b_sim_on AND axisdata[6].Axis_Inbb,
//     ParameterNumber := FP_P_0_0539,
//     Axis := drive6,
//     Value => dw_brake_6); // MB_ReadParameter

// NETWORK 7
//   axisdata[1].Axis_Inbb: A-0-0021.13 -RD- Axis is ready for power to the amplifier (bb)
//   FP_C_0_0626: Diagnostics
//   drive1: Real axis "Drive1" with axis number 1
//   str_diagnose_MLC: FP_P_0_0007,Display text of diagnostic message
fb_diagnose_MLC(
    Execute := NOT gc_b_sim_on AND axisdata[1].Axis_Inbb,
    ParameterNumber := FP_C_0_0626,
    Axis := drive1,
    Value => str_diagnose_MLC); // MB_ReadStringParameter

// NETWORK 8 (disabled)
//   fb_diagnose_1: With the function block "MB_ReadStringParameter" it is possible to read a parameter the operating data of which has the ASCII format (string).
//   axisdata[1].Axis_Inbb: A-0-0021.13 -RD- Axis is ready for power to the amplifier (bb)
//   FP_P_0_0007: Display text of diagnostic message
//   drive1: Real axis "Drive1" with axis number 1
// fb_diagnose_1(
//     Execute := NOT gc_b_sim_on AND axisdata[1].Axis_Inbb,
//     ParameterNumber := FP_P_0_0007,
//     Axis := drive1,
//     Value => str_diagnose_1); // MB_ReadStringParameter

// NETWORK 9
//   fb_diagnose_1: With the function block "MB_ReadStringParameter" it is possible to read a parameter the operating data of which has the ASCII format (string).
//   fb_blink_diagnos_1: The function block BLINK generates a pulsating signal.The input consists of ENABLE of the type BOOL, as well as TIMELOW and TIMEHIGH of the type TIME.
//   axisdata[1].Axis_Inbb: A-0-0021.13 -RD- Axis is ready for power to the amplifier (bb)
//   FP_S_0_0095: Diagnostic message
//   drive1: Real axis "Drive1" with axis number 1
fb_blink_diagnos_1(ENABLE := NOT gc_b_sim_on AND axisdata[1].Axis_Inbb, TIMELOW := t#1s, TIMEHIGH := t#1s); // BLINK
fb_diagnose_1(
    Execute := fb_blink_diagnos_1.OUT,
    ParameterNumber := FP_S_0_0095,
    Axis := drive1,
    Value => str_diagnose_1); // MB_ReadStringParameter

// NETWORK 10
//   axisdata[2].Axis_Inbb: A-0-0021.13 -RD- Axis is ready for power to the amplifier (bb)
//   FP_S_0_0095: Diagnostic message
//   drive2: Real axis "Drive2" with axis number 2
fb_blink_diagnos_2(ENABLE := NOT gc_b_sim_on AND axisdata[2].Axis_Inbb, TIMELOW := t#1s, TIMEHIGH := t#1s); // BLINK
fb_diagnose_2(
    Execute := fb_blink_diagnos_2.OUT,
    ParameterNumber := FP_S_0_0095,
    Axis := drive2,
    Value => str_diagnose_2); // MB_ReadStringParameter

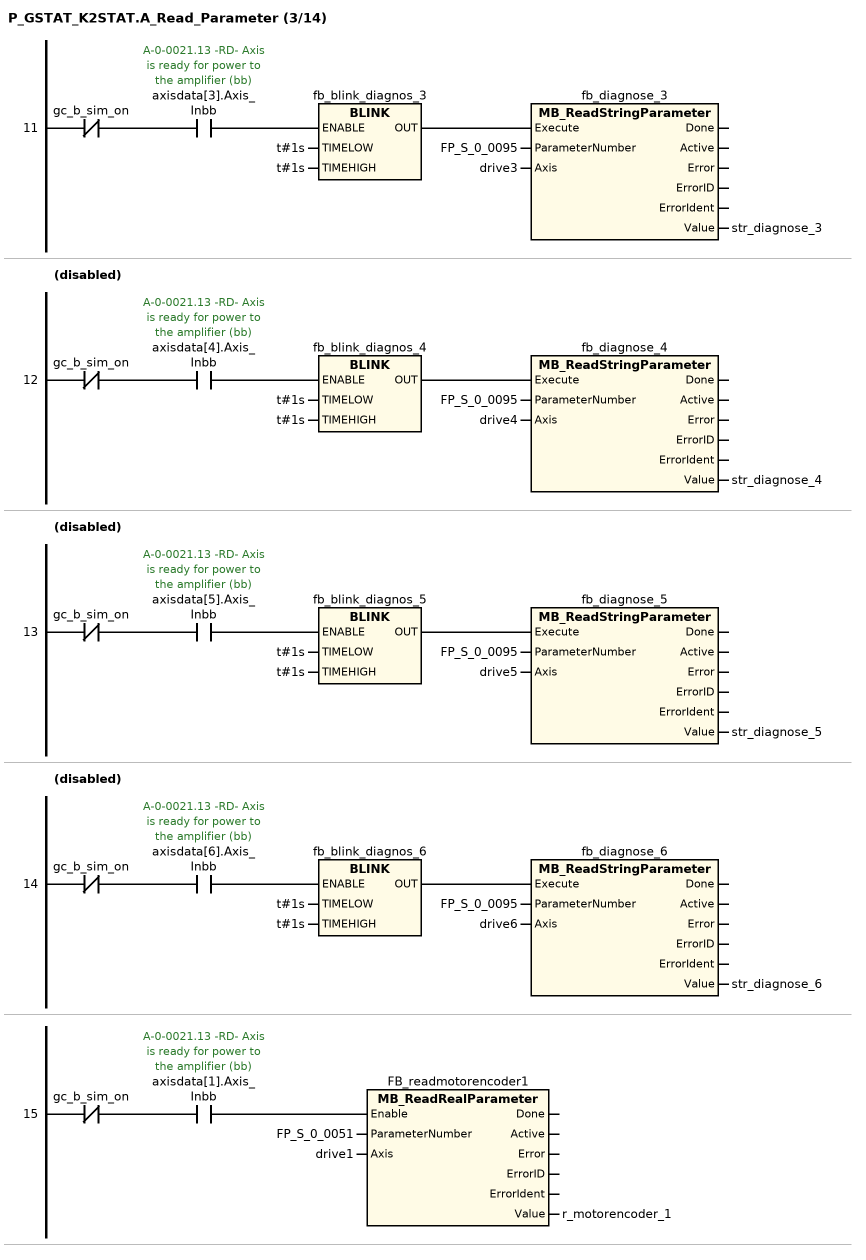
// NETWORK 11
//   axisdata[3].Axis_Inbb: A-0-0021.13 -RD- Axis is ready for power to the amplifier (bb)
//   FP_S_0_0095: Diagnostic message
//   drive3: Real axis "Drive3" with axis number 3
fb_blink_diagnos_3(ENABLE := NOT gc_b_sim_on AND axisdata[3].Axis_Inbb, TIMELOW := t#1s, TIMEHIGH := t#1s); // BLINK
fb_diagnose_3(
    Execute := fb_blink_diagnos_3.OUT,
    ParameterNumber := FP_S_0_0095,
    Axis := drive3,
    Value => str_diagnose_3); // MB_ReadStringParameter

// NETWORK 12 (disabled)
//   axisdata[4].Axis_Inbb: A-0-0021.13 -RD- Axis is ready for power to the amplifier (bb)
//   FP_S_0_0095: Diagnostic message
//   drive4: Real axis "Drive4" with axis number 4
// fb_blink_diagnos_4(ENABLE := NOT gc_b_sim_on AND axisdata[4].Axis_Inbb, TIMELOW := t#1s, TIMEHIGH := t#1s); // BLINK
// fb_diagnose_4(
//     Execute := fb_blink_diagnos_4.OUT,
//     ParameterNumber := FP_S_0_0095,
//     Axis := drive4,
//     Value => str_diagnose_4); // MB_ReadStringParameter

// NETWORK 13 (disabled)
//   axisdata[5].Axis_Inbb: A-0-0021.13 -RD- Axis is ready for power to the amplifier (bb)
//   FP_S_0_0095: Diagnostic message
//   drive5: Real axis "Drive5" with axis number 5
// fb_blink_diagnos_5(ENABLE := NOT gc_b_sim_on AND axisdata[5].Axis_Inbb, TIMELOW := t#1s, TIMEHIGH := t#1s); // BLINK
// fb_diagnose_5(
//     Execute := fb_blink_diagnos_5.OUT,
//     ParameterNumber := FP_S_0_0095,
//     Axis := drive5,
//     Value => str_diagnose_5); // MB_ReadStringParameter

